// SIMATIC STEP 7 (V5.x) project PC1_NEW_01_08_2014
// CPU: CPU 315-2 DP
// station: P_ADR_BUS
// station: Hardware
// station: SIMATIC 300 - BEC
// program: S7 Program(1)

SYMBOL_TABLE
"MAIN_POWER_DB"	DB 1	DB 1	// MAIN POWER DATA BLOCK
"HYDRAULIC_FUNCTIONS_DB"	DB 2	DB 2	// HYDRAULIC FUNCTIONS DB
"TRAVEL_DRIVE_DB"	DB 3	DB 3	// TRAVEL DRIVE DATA BLOCK
"PUSHER_RAM_DB"	DB 4	DB 4	// PUSHER RAM DRIVE MECHANISH DATA BLOCK
"LEVEL_RAM_DB"	DB 5	DB 5	// LEVELER RAM DRIVE MECHANISH DATA BLOCK
"AIR_COMPRESSOR_DB"	DB 6	DB 6	// AIR COMPRESSOR DATA BLOCK
"DOOR_AND_JAMB_DB"	DB 7	DB 7	// DOOR AND JAMB CLEANER VIBRATOR DATA BLOCK
"LEVELER_BLOWER_DB"	DB 8	DB 8	// LEVELER BLOWER DATA BLOCK
"LIFTING_PLATFORM_DB"	DB 9	DB 9	// LIFTING PLATFORM DATA BLOCK
"LEVELER_DOOR_DB"	DB 10	DB 10	// LEVELER DOOR MECHANISM DATA BLOCK
"LEVELER_MUFF_DB"	DB 11	DB 11	// LEVELER MUFF MECHANISM DATA BLOCK
"DOOR_EXTRACTOR_DB"	DB 12	DB 12	// DOOR EXTRACTOR MECHANISH DATA BLOCK
"DOOR_CLEANER_DB"	DB 13	DB 13	// DOOR CLEANER MECHANISM DATA BLOCK
"JAMB_CLEANER_DB"	DB 14	DB 14	// JAMB CLEANER MECHANISM DATA BLOCK
"COUNTER_THRUST_WEDGE_DB"	DB 15	DB 15	// COUNTER THRUST WEDGE DATA BLOCK
"COAL_SPILLAGE_SYSTEM_DB"	DB 16	DB 16	// COAL SPILLAGE SYSTEM DATA BLOCK
"TATA_COMMUNICATION_DB"	DB 17	DB 17	// TATA COMMUNICATION THROUGH PROFIBUS
"WINCC_DB"	DB 18	DB 18
"DB_FOR_FM350"	DB 19	UDT 2
"FB_TO_TATA"	DB 20	DB 20	// FEEDBACK TO TATA ONBOARD PLC THROUGH PROFIBUS
"CMD_FROM_TATA"	DB 21	DB 21	// COMMAND FROM TATA ONBOARD PLC THROUGH PROFIBUS
"INPUT_MAPPING"	FC 1	FC 1	// INPUT MAPPING TO DATA BLOCK
"OUTPUT_MAPPING"	FC 2	FC 2	// OUTPUT MAPPING FROM DATA BLOCK
"MAIN_POWER"	FC 3	FC 3	// MAIN POWER CONTROL LOGIC
"HYDRAULIC_SYSTEM"	FC 4	FC 4	// HYDRAULIC SYSTEM OPERATIONS
"LEVELLER_RAM"	FC 5	FC 5	// LEVELLER RAM MECHANISH FUNCTION
"LEVELER_DOOR"	FC 6	FC 6	// LEVELLER DOOR MECHANISM
"TRAVEL_DRIVE"	FC 7	FC 7	// TRAVEL_DRIVE_MECHANISM
"PUSHER_RAM"	FC 8	FC 8	// PUSHER RAM MECHANISM
"AIR_COMPRESSOR"	FC 9	FC 9	// AIR COMPRESSOR FUNCTION
"DOOR_AND_JAMB"	FC 10	FC 10	// DOOR AND JAMB CLEANER MECHANISM
"LEVELER_BLOWER"	FC 11	FC 11	// LEVELER BLOWER FUNCTIONS
"LIFTING_PLATFORM"	FC 12	FC 12	// LIFTING PLATFORM FUNCTIONS
"LEVELER_MUFF"	FC 13	FC 13	// LEVELER MUFF MECHANISM
"DOOR_EXTRACTOR"	FC 14	FC 14	// DOOR EXTRACTOR MECHANISM
"DOOR_CLEANER"	FC 15	FC 15	// DOOR CLEANER MECHANISM
"JAMB_CLEANER"	FC 16	FC 16	// JAMB CLEANER MECHANISM
"COUNTER_THRUST_WEDGE"	FC 17	FC 17	// COUNTER THRUST WEDGE MECHANISM
"COAL_SPILLAGE_SYSTEM"	FC 18	FC 18	// COAL SPILLAGE SYSTEM
"PROFIBUS_COMMUNICATION"	FC 19	FC 19	// PROFIBUS COMMUNICATION
"TATA_COMMUNICATION"	FC 20	FC 20	// TATA COMMUNICATION FOR AUTO POSITIONING
"Clock Generator"	FC 69	FC 69	// Clock generator
"SCALE"	FC 105	FC 105	// Scaling Values
"UNSCALE"	FC 106	FC 106	// Unscaling Values
"MAIN_PWR_RDY_FOR_ON"	I 0.0	BOOL	// MAIN POWER READY FOR ON
"MAIN_PWR_ON_PB"	I 0.1	BOOL	// MAIN POWER ON PUSH BUTTON
"MAIN_PWR_OFF_PB"	I 0.2	BOOL	// MAIN POWER OFF PUSH BUTTON
"MAIN_PWR_ON_FB"	I 0.3	BOOL	// MAIN POWER ON FEED BACK
"CTRL_PWR_ON_FB"	I 0.4	BOOL	// CONTROL POWER ON FEEDBACK
"LAMP_TEST_PB"	I 0.5	BOOL	// LAMP TEST PUSH BUTTON
"ALARM_ACK_PB"	I 0.6	BOOL	// ALARM ACKNOWLEDGE PUSH BUTTON
"TRA_ILK_BYPAS"	I 0.7	BOOL	// TRAVEL INTERLOCK BYPASS INPUT
"PUSH_RAM_ILK_BYPASS"	I 1.0	BOOL	// PUSHER RAM INTERLOCK BYPASS
"LEV_ILK_BYPASS"	I 1.1	BOOL	// LEVELER RAM INTERLOCK BYPASS INPUT
"LEV_DRV_PROF_HARD_SEL"	I 1.2	BOOL	// LEVELER DRIVE PROFIBUS / HARD WIRE CONNECTION
"LEV_DRV_ON_FB"	I 1.3	BOOL	// LEVELER DRIVE ON FEED BACK
"PUMP_1_RDY_FOR_STA"	I 1.4	BOOL	// PUMP 1 READY FOR START
"PUMP_1_RUN_FB"	I 1.5	BOOL	// PUMP 1 RUNNING FEEDBACK
"PUMP_1_OVR_LD_TRIP"	I 1.6	BOOL	// PUMP 1 OVER LOAD TRIPPED
"LEV_DRV_RDY_FOR_STA"	I 1.7	BOOL	// LEVELER DRIVE READY FOR START
"PUMP_2_RDY_FOR_STA"	I 2.0	BOOL	// PUMP 2 READY FOR START
"PUMP_2_RUN_FB"	I 2.1	BOOL	// PUMP 2 RUNNING FEEDBACK
"PUMP_2_OVR_LD_TRIP"	I 2.2	BOOL	// PUMP 2 OVER LOAD TRIPPED
"CIR_PUMP_RDY_FOR_STA"	I 2.3	BOOL	// CIRCULATION PUMP READY FOR START
"CIR_PUMP_RUN_FB"	I 2.4	BOOL	// CIRCULATION PUMP RUNNING FEEDBACK
"CIR_PUMP_OVR_LD_TRIP"	I 2.5	BOOL	// CIRCULATION PUMP OVER LOAD TRIPPED
"COLR_FAN_RDY_FOR_STA"	I 2.6	BOOL	// COOLER FAN READY FOR START
"LEV_DRV_TRP_FB"	I 2.7	BOOL	// LEVELER DRIVE TRIP FEED BACK
"COLR_FAN_RUN_FB"	I 3.0	BOOL	// COOLER FAN RUNNING FEEDBACK
"COLR_FAN_OVR_LD_TRIP"	I 3.1	BOOL	// COOLER FAN OVER LOAD TRIPPED
"CD_LCS_SS"	I 3.2	BOOL	// CONTROL DESK / LOCAL CONTROL SELECTOR SWITCH
"PUMP_1_2_SS"	I 3.3	BOOL	// PUMP 1 OR 2 SELECTOR SWITCH
"PUMP_1_STA_PB"	I 3.4	BOOL	// PUMP 1 START PUSH BUTTON
"PUMP_1_STP_PB"	I 3.5	BOOL	// PUMP 1 STOP PUSH BUTTON
"PUMP_2_STA_PB"	I 3.6	BOOL	// PUMP 2 START PUSH BUTTON
"GRV_SCRPR_2_FWD_LS"	I 3.7	BOOL	// DOOR CLEANER GROOVE SCRAPPER 2 FORWARD LIMIT SWITCH
"PUMP_2_STP_PB"	I 4.0	BOOL	// PUMP 2 STOP PUSH BUTTON
"EMERGENCY_STOP_PB_LCS_41"	I 4.1	BOOL	// EMERGENCY STOP PUSH BUTTON LCS 41
"PUMP_1_2_SS_LCS"	I 4.2	BOOL	// PUMP 1 OR 2 SELECTOR SWITCH LCS
"PUMP_1_STA_PB_LCS"	I 4.3	BOOL	// PUMP 1 START PUSH BUTTON LCS
"PUMP_1_STP_PB_LCS"	I 4.4	BOOL	// PUMP 1 STOP PUSH BUTTON LCS
"PUMP_2_STA_PB_LCS"	I 4.5	BOOL	// PUMP 2 START PUSH BUTTON LCS
"PUMP_2_STP_PB_LCS"	I 4.6	BOOL	// PUMP 2 STOP PUSH BUTTON LCS
"GRV_SCRPR_2_RET_LS"	I 4.7	BOOL	// DOOR CLEANER GROOVE SCRAPPER 2 RETRACT LIMIT SWITCH
"CIR_PUMP_STA_PB_LCS"	I 5.0	BOOL	// CIRCULATION PUMP START PUSH BUTTON LCS
"CIR_PUMP_STP_PB_LCS"	I 5.1	BOOL	// CIRCULATION PUMP STOP PUSH BUTTON LCS
"COLR_FAN_STA_PB_LCS"	I 5.2	BOOL	// COOLER FAN START PUSH BUTTON LCS
"COLR_FAN_STP_PB_LCS"	I 5.3	BOOL	// COOLER FAN STOP PUSH BUTTON LCS
"LAMP_TEST_PB_LCS_41"	I 5.4	BOOL	// LAMP TEST PUSH BUTTON LCS
"SHT_OF_VLV_LIN_1_FUL_OPN"	I 5.5	BOOL	// SHUT OFF VALVE IN LINE 1 - FULLY OPEN
"SHT_OF_VLV_LIN_2_FUL_OPN"	I 5.6	BOOL	// SHUT OFF VALVE IN LINE 2 - FULLY OPEN
"DOOR_FIX_LOC_FB_PR_SWT"	I 5.7	BOOL	// DOOR FIX LOCKED FEEDBACK PRESSURE SWITCH
"LOW_OIL_TEMP"	I 6.0	BOOL	// LOW OIL TEMPERATURE - THERMOSTAT
"HIGH_OIL_TEMP"	I 6.1	BOOL	// HIGH OIL TEMPERATURE - THERMOSTAT
"MAX_OIL_TEMP"	I 6.2	BOOL	// MAXIMUM OIL TEMPERATURE - THERMOSTAT
"LOW_OIL_LEVEL"	I 6.3	BOOL	// LOW OIL LEVEL - FLOAT SWITCH
"MIN_OIL_LEVEL"	I 6.4	BOOL	// MINIMUM OIL LEVEL - FLOAT SWITCH
"RET_LIN_FLTR_CKD"	I 6.5	BOOL	// RETURN LINE FILTER CHOKED
"LOW_OIL_PRESS"	I 6.6	BOOL	// LOW OIL PRESSURE - PRESSURE SWITCH
"DOOR_FIX_REL_FB"	I 6.7	BOOL	// DOOR FIXRELEASED FEEDBACK
"HIGH_OIL_PRESS"	I 7.0	BOOL	// HIGH OIL PRESSURE - PRESSURE SWITCH
"EMG_ACCM_STA_PB_LCS"	I 7.1	BOOL	// EMERGENCY ACCUMULATOR START PB LCS
"EMG_ACCM_STP_PB_LCS"	I 7.2	BOOL	// EMERGENCY ACCUMULATOR STOP PB LCS
"HTR_STA_PB_LCS"	I 7.3	BOOL	// HEATER START PUSH BUTTON LCS
"HTR_STP_PB_LCS"	I 7.4	BOOL	// HEATER STOP PUSH BUTTON LCS
"TRA_GRP_1_RDY_FOR_STA"	I 7.6	BOOL	// TRAVEL GROUP 1 READY FOR START
"TATA_PUSH_PERM_BYPASS"	I 7.7	BOOL	// TATA PUSHING PERMISION BYPASS
"TRA_GRP_2_RDY_FOR_STA"	I 8.0	BOOL	// TRAVEL GROUP 2 READY FOR START
"TRA_GRP_2_RUN_FB"	I 8.1	BOOL	// TRAVEL GROUP 2 RUNNING FEEDBACK
"TRA_MTR_3_OVLD_TRIP"	I 8.2	BOOL	// TRAVEL MOTOR 3 OVER LOAD TRIP
"TRA_MTR_4_OVLD_TRIP"	I 8.3	BOOL	// TRAVEL MOTOR 4 OVER LOAD TRIP
"TRA_GRP_1_BRK_RDY_FOR_ST"	I 8.4	BOOL	// TRAVEL GROUP 1 BREAK READY FOR START
"TRA_GRP_1_BRK_ON_FB"	I 8.5	BOOL	// TRAVEL GROUP 1 BREAK ON FEEDBACK
"TRA_GRP_1_RUN_FB"	I 8.6	BOOL	// TRAVEL GROUP 1 RUNNING FEEDBACK
"USE_JOY_STICK_FOR_PUSH"	I 8.7	BOOL	// USER TRAVEL JOY STICK FOR PUSHER
"TRA_MTR_1_OVLD_TRIP"	I 9.0	BOOL	// TRAVEL MOTOR 1 OVER LOAD TRIP
"TRA_MTR_2_OVLD_TRIP"	I 9.1	BOOL	// TRAVEL MOTOR 2 OVER LOAD TRIP
"TRA_MTR_1_ISO_ON_FB"	I 9.2	BOOL	// TRAVEL MOTOR 1 ISOLATOR ON FEEDBACK
"TRA_MTR_2_ISO_ON_FB"	I 9.3	BOOL	// TRAVEL MOTOR 2 ISOLATOR ON FEEDBACK
"TRA_MTR_3_ISO_ON_FB"	I 9.4	BOOL	// TRAVEL MOTOR 3 ISOLATOR ON FEEDBACK
"TRA_MTR_4_ISO_ON_FB"	I 9.5	BOOL	// TRAVEL MOTOR 4 ISOLATOR ON FEEDBACK
"SIR_RDY_FOR_STA"	I 9.6	BOOL	// SIREN READY FOR START
"USE_JOY_STICK_FOR_LEV"	I 9.7	BOOL	// USE TRAVEL JPY STICK FOR LEVELER
"SIR_ON_FB"	I 10.0	BOOL	// SIREN ON FEED BACK
"TRA_GRP_2_BRK_RDY_FOR_ST"	I 10.1	BOOL	// TRAVEL GROUP 2 BREAK READY FOR START
"TRA_GRP_2_BRK_ON_FB"	I 10.2	BOOL	// TRAVEL GROUP 2 BREAK ON FEEDBACK
"SIR_OLR_TRIP"	I 10.3	BOOL	// SIREN ON OVER LOAD TRIP
"TRA_JOY_STK_REV_POS"	I 10.4	BOOL	// TRAVEL JOY STICK REVERSE POSITION
"TRA_JOY_STK_DED_MAN_BTN"	I 10.5	BOOL	// TRAVEL JOY DEAD MAN BUTTON
"TRA_JOY_STK_HME_POS"	I 10.6	BOOL	// TRAVEL JOY STICK HOME POSITION
"PUSH_JS_FWD_POS"	I 10.7	BOOL	// PUSHER RAM JOY STICK FORWARD POSITION
"TRA_JOY_STK_FWD_POS"	I 11.0	BOOL	// TRAVEL JOYSTICK FORWARD POSITION
"TRA_DRV_1_PROF_HARD_SS"	I 11.1	BOOL	// TRAVEL DRIVE 1 PROFIBUS/HARD WIRE SELECTRO SWITCH
"TRA_DRV_1_ON_FB"	I 11.2	BOOL	// TRAVEL DRIVE 1 ON FEEDBACK
"TRA_DRV_1_RDY_FOR_STA"	I 11.3	BOOL	// TRAVEL DRIVE 1 READY FOR START
"TRA_DRV_1_TRP_FB"	I 11.4	BOOL	// TRAVEL DRIVE 1 TRIP FEEDBACK
"TRA_DRV_2_PROF_HARD_SS"	I 11.5	BOOL	// TRAVEL DRIVE 2 PROFIBUS/HARD WIRE SELECTRO SWITCH
"TRA_DRV_2_ON_FB"	I 11.6	BOOL	// TRAVEL DRIVE 2 ON FEEDBACK
"PUSH_JS_HME_POS"	I 11.7	BOOL	// PUSHER JOY STICK HOME POSITION
"TRA_DRV_2_RDY_FOR_STA"	I 12.0	BOOL	// TRAVEL DRIVE 2 READY FOR START
"TRA_DRV_2_TRP_FB"	I 12.1	BOOL	// TRAVEL DRIVE 2 TRIP FEEDBACK
"LIMIT_SW_END_FWD_FB"	I 12.2	BOOL	// LIMIT SWITCH END FORWARD FEEDBACK
"LIMIT_SW_END_REV_FB"	I 12.4	BOOL	// LIMIT SWITCH END REVERSE FEEDBACK
"PUSH_BRK_RDY_FOR_STA"	I 12.6	BOOL	// PUSHER BRAKE READY FOR START
"PUSH_JS_REV_POS"	I 12.7	BOOL	// PUSHER JOY STICK REVERSE POSITION
"PUSH_MTR_BRK_ON_FB"	I 13.0	BOOL	// PUSHER MOTOR BRAKE ON FEEDBCAK
"PUSH_RAM_STP_PB"	I 13.1	BOOL	// PUSHER RAM STOP PUSH BUTTON
"PUSH_MAN_SS"	I 13.2	BOOL	// PUSHER MANUAL SELECTOR SWTICH
"PUSH_AUTO_SS"	I 13.3	BOOL	// PUSHER AUTO SELECTOR SWITCH
"PUSH_DRV_PROF_HDWR_SS"	I 13.4	BOOL	// PUSHER DRIVE PROFIBUS/HARDWIRE SELECTOR SWITCH
"PUSH_DRV_ON_FB"	I 13.5	BOOL	// PUSHER DRIVE ON FEED BACK
"PUSH_DRV_RDY_FOR_STA"	I 13.6	BOOL	// PUSHER DRIVE READY FOR START
"PUSH_JS_DEAD_MAN_BTN"	I 13.7	BOOL	// PUSHER JOY STICK DEAD MAN BUTTON
"PUSH_DRV_TRP_FB"	I 14.0	BOOL	// PUSHER DRIVE TRIP FEED BACK
"PUSH_RLS_OVN_FACE_RCHD"	I 14.1	BOOL	// PUSHER RLS OVEN FACE REACHED
"PUSH_RLS_GUIDE_ENT"	I 14.2	BOOL	// PUSHER RLS GUIDE ENTRY
"PUSH_RLS_FWD_END"	I 14.3	BOOL	// PUSHER RLS FORWARD END
"PUSH_RLS_STND_PIPE"	I 14.4	BOOL	// PUSHER RLS STAND PIPE
"PUSH_RLS_REV_END"	I 14.5	BOOL	// PUSHER RLS REVERSE END
"AUTO_POS_ACK"	I 14.6	BOOL	// AUTO PISITION ACKNOWLEDGE
"TRA_MODE_AUTO_MAN_SS"	I 14.7	BOOL	// TRAVEL MODE AUTO MANUAL SELECTOR SWITCH
"CDL_EMERGENCY_PB"	I 15.0	BOOL	// CONTROL DESK LEFT EMERGENCY PUSH BUTTON
"LIFT_LDT_TMR_SS"	I 15.1	BOOL	// LIFTING LDT TIMER SELECTOR
"RAM_EMG_DRV_DIS_ENG"	I 15.2	BOOL	// RAM EMERGENCY DRIVE DISENGAGE
"RAM_END_FWD_LS"	I 15.3	BOOL	// RAM END FORWARD LIMIT SWITCH
"RAM_END_RET_LS"	I 15.4	BOOL	// RAM END RETRACT LIMIT SWITCH
"LEV_BRK_RDY_FOR_STA"	I 15.5	BOOL	// LEVELER BRAKE READY FOR START
"MTR_BRK_ON_FB"	I 15.6	BOOL	// MOTOR BRAKE ON FEED BACK
"LEV_STP_PB"	I 16.0	BOOL	// LEVELER BRAKE STOP PUSH BUTTON
"MANUAL_SS"	I 16.1	BOOL	// MANUAL SELECTOR SWITCH
"AUTO_SS"	I 16.2	BOOL	// AUTOMATIC SELECTOR SWITCH
"LEV_JS_FWD_POS"	I 16.3	BOOL	// LEVELER JOYSTICK FORWARD POSITION
"LEV_JS_HME_POS"	I 16.4	BOOL	// LEVELER JOYSTICK HOME POSITION
"LEV_JS_REV_POS"	I 16.5	BOOL	// LEVELER JOY STICK REVERSE POSITION
"LEV_JS_DEAD_MAN_BUTTON"	I 16.6	BOOL	// LEVELER JOY STICK DEAD MAN BUTTON
"LEV_RLS_OVN_FAC_RCHD"	I 17.4	BOOL	// LEVELER RLS OVEN FACE REACHED
"LEV_RLS_FWD_END"	I 17.5	BOOL	// LEVELER RLS FORWARD END
"LEV_RLS_REV_STK_FB"	I 17.6	BOOL	// LEVELER RLS REVERSE STROKE FEED BACK
"LEV_RLS_REV_END"	I 18.0	BOOL	// LEVELER RLS REVERSE END
"EMG_PB_LCS_16"	I 18.1	BOOL	// EMERGENCY PUSH BUTTON LCS 16
"LEV_EM_DRV_ENG_LCS"	I 18.2	BOOL	// LEVELER EMERGENCY DRIVE ENGAGE LCS
"LEV_EM_DRV_DIS_ENG_LCS"	I 18.3	BOOL	// LEVELER EMERGENCY DRIVE DISENGAGE LCS
"LEV_EM_DRV_DIS_ENG"	I 18.4	BOOL	// LEVELER EMERGENCY DRIVE DISENGAGE
"LEV_END_FWD_LS"	I 18.5	BOOL	// LEVELER END FORWARD LIMIT SWITCH
"LEV_END_RET_LS"	I 18.6	BOOL	// LEVELER END RETRACT LIMIT SWITCH
"SPRING_PRESS"	I 19.1	BOOL	// SPRING PRESS
"LEV_BLOW_RDY_FOR_STA"	I 19.2	BOOL	// LEVELER BLOWER READY FOR START
"LEV_BLOW_RUN_FB"	I 19.3	BOOL	// LEVELER BLOWER RUNNING FEED BACK
"LEV_BLOW_OLR_TRP"	I 19.4	BOOL	// LEVELER BLOWER TRIP FEED BACK
"LEV_BLOW_STA_PB"	I 19.5	BOOL	// LEVELER BLOWER START PUSH BUTTON
"LEV_BLOW_STP_PB"	I 19.6	BOOL	// LEVELER BLOWER STOP PUSH BUTTON
"LEV_BLOW_STA_PB_LCS"	I 20.0	BOOL	// LEVELER BLOWER START PUSH BUTTON LCS
"LEV_BLOW_STP_PB_LCS"	I 20.1	BOOL	// LEVELER BLOWER STOP PUSH BUTTON LCS
"LIFT_PF_RDY_FOR_STA"	I 20.2	BOOL	// LIFT PLATFORM READY FOR START
"LIFT_PF_UP_ON_FB"	I 20.3	BOOL	// LIFT PLATFORM UP ON FEEDBCAK
"LIFT_PF_DN_ON_FB"	I 20.4	BOOL	// LIFT PLATFORM DOWN ON FEEDBCAK
"LIFT_MTR_OLR_TRP"	I 20.5	BOOL	// LIFT MOTOR OVERLOAD TRIP
"LIFT_PF_UP_PB"	I 20.6	BOOL	// LIFT PLATFORM UP PUSH BUTTON
"LIFT_PF_DN_PB"	I 21.0	BOOL	// LIFT PLATFORM DOWN PUSH BUTTON
"EMERGENCY_PB_LCS_19"	I 21.2	BOOL	// LCS-19 EMERGENCY PUSH BUTTON
"LIFT_PF_UP_LS"	I 21.3	BOOL	// LIFT PLATFORM UP LIMIT SWITCH
"LIFT_PF_DN_LS"	I 21.4	BOOL	// LIFT PLATFORM DOWN LIMIT SWITCH
"LEV_DOOR_LOCAL_SS"	I 22.3	BOOL	// LEVELER DOOR LOCAL SELECTOR SWITCH
"LEV_DOOR_MAN_SS"	I 22.4	BOOL	// LEVELER DOOR MANUAL SELECTOR SWITCH
"LEV_DOOR_AUTO_SS"	I 22.5	BOOL	// LEVELER DOOR AUTO SELECTOR SWITCH
"LEV_DOOR_STP_PB"	I 22.6	BOOL	// LEVELER DOOR STOP PUSH BUTTON
"ACT_GRP_FWD_STA_PB"	I 23.0	BOOL	// ACTUATING GRIP FORWARD START PUSH BUTTON
"ACT_GRP_RET_STA_PB"	I 23.1	BOOL	// ACTUATING GRIP RETRACT START PUSH BUTTON
"SLW_RK_SP_1_FWD_STA"	I 23.2	BOOL	// SLEAVING RACK STEP 1 FORWARD START PUSH BUTTON
"SLW_RK_SP_1_RET_STA"	I 23.3	BOOL	// SLEAVING RACK STEP 1 RETRACT START PUSH BUTTON
"SLW_RK_SP_2_FWD_STA"	I 23.4	BOOL	// SLEAVING RACK STEP 2 FORWARD START PUSH BUTTON
"SLW_RK_SP_2_RET_STA"	I 23.5	BOOL	// SLEAVING RACK STEP 2 RETRACT START PUSH BUTTON
"LEV_WN_FM_CR_UP_STA"	I 23.6	BOOL	// LEVELER WINDOW FRAME CLEANER UP START PUSH BUTTON
"LEV_WN_FM_CR_DN_STA"	I 24.0	BOOL	// LEVELER WINDOW FRAME CLEANER DOWN START PUSH BUTTON
"SMK_SLVE_FWD_STA_PB"	I 24.1	BOOL	// SMOKE SLEEVE FORWARD START PUSH BUTTON
"SMK_SLVE_RET_STA_PB"	I 24.2	BOOL	// SMOKE SLEEVE RETRACT START PUSH BUTTON
"EMG_STOP_PB_LCS_61"	I 24.3	BOOL	// EMERGENCY STOP PUSH BUTTON LCS 61
"ACT_GRP_FWD_STA_PB_LCS"	I 24.4	BOOL	// ACTUATING GRIP FORWARD START PUSH BUTTON LCS
"ACT_GRP_RET_STA_PB_LCS"	I 24.5	BOOL	// ACTUATING GRIP RETRACT START PUSH BUTTON LCS
"SLW_RK_SP_1_FWD_STA_LCS"	I 24.6	BOOL	// SLEAVING RACK STEP 1 FORWARD START PUSH BUTTON LCS
"SLW_RK_SP_1_RET_STA_LCS"	I 25.0	BOOL	// SLEAVING RACK STEP 1 RETRACT START PUSH BUTTON LCS
"SLW_RK_SP_2_FWD_STA_LCS"	I 25.1	BOOL	// SLEAVING RACK STEP 2 FORWARD START PUSH BUTTON LCS
"SLW_RK_SP_2_RET_STA_LCS"	I 25.2	BOOL	// SLEAVING RACK STEP 2 RETRACT START PUSH BUTTON LCS
"LEV_WN_FM_CR_UP_STA_LCS"	I 25.3	BOOL	// LEVELER WINDOW FRAME CLEANER UP START PUSH BUTTON LCS
"LEV_WN_FM_CR_DN_STA_LCS"	I 25.4	BOOL	// LEVELER WINDOW FRAME CLEANER DOWN START PUSH BUTTON LCS
"SMK_SLVE_FWD_STA_PB_LCS"	I 25.5	BOOL	// SMOKE SLEEVE FORWARD START PUSH BUTTON LCS
"SMK_SLVE_RET_STA_PB_LCS"	I 25.6	BOOL	// SMOKE SLEEVE RETRACT START PUSH BUTTON LCS
"TEST_LAMP_PB_LCS_61"	I 26.0	BOOL	// TEST LAMP PUSH BUTTON LCS 61
"SLW_RK_SP_1_FWD_LS"	I 26.5	BOOL	// SLEAVING RACK STEP 1 FORWARD LIMIT SWITCH
"SLW_RK_SP_1_RET_LS"	I 26.6	BOOL	// SLEAVING RACK STEP 1 RETRACT LIMIT SWITCH
"SLW_RK_SP_2_FWD_LS"	I 27.0	BOOL	// SLEAVING RACK STEP 2 FORWARD LIMIT SWITCH
"SLW_RK_SP_2_RET_LS"	I 27.1	BOOL	// SLEAVING RACK STEP 2 RETRACT LIMIT SWITCH
"LEV_WN_FM_CR_UP_LS"	I 27.2	BOOL	// LEVELER WINDOW FRAME CLEANER UP LIMIT SWITCH
"LEV_WN_FM_CR_DN_LS"	I 27.3	BOOL	// LEVELER WINDOW FRAME CLEANER DOWN LIMIT SWITCH
"SMK_SLVE_FWD_LS"	I 27.4	BOOL	// SMOKE SLEEVE FORWARD LIMIT SWITCH
"SMK_SLVE_SLOW_FWD_LS"	I 27.5	BOOL	// SMOKE SLEEVE SLOW FORWARD LIMIT SWITCH
"SMK_SLVE_REV_LS"	I 27.6	BOOL	// SMOKE SLEEVE RETRACT LIMIT SWITCH
"VIB_JMB_CLNR_STA_PB_LCS"	I 27.7	BOOL	// VIBRATOR - JAMB CLEANER START PUSH BUTTON LCS
"ACT_GRP_FWD_LS"	I 28.0	BOOL	// ACTUATING GRIP FORWARD START LIMIT SWITCH
"ACT_GRP_RET_LS"	I 28.1	BOOL	// ACTUATING GRIP RETRACT START LIMIT SWITCH
"VIB_JMB_CLNR_STP_PB_LCS"	I 28.2	BOOL	// VIBRATOR - JAMB CLEANER STOP PUSH BUTTON LCS
"AIR_COMP_PRESSURE_SW_FB"	I 28.5	BOOL	// PRESSURE SWITCH FEEDBACK
"DOOR_EXT_LOC_SS"	I 28.6	BOOL	// DOOR EXTRACTOR LOCAL SELECTOR SWITCH
"DOOR_EXT_MAN_SS"	I 29.0	BOOL	// DOOR EXTRACTOR MANUAL SELECTOR SWITCH
"DOOR_EXT_AUTO_SS"	I 29.1	BOOL	// DOOR EXTRACTOR AUTO SELECTOR SWITCH
"DOOR_EXT_STP_PB"	I 29.2	BOOL	// DOOR EXTRACTOR STOP PUSH BUTTON
"SLEW_FWD_STA_PB"	I 29.3	BOOL	// SLEW FORWARD START PUSH BUTTON
"SLEW_RET_STA_PB"	I 29.4	BOOL	// SLEW RETRACT START
"VER_COMP_FWD_STA"	I 29.5	BOOL	// VERTICAL COMPENSATION FORWARD START PUSHBUTTON
"VER_COMP_RET_STA"	I 29.6	BOOL	// VERTICAL COMPENSATION RETRACT START PUSHBUTTON
"TRA_FWD_STA"	I 30.0	BOOL	// TRAVEL FORWARD START PUSHBUTTON
"TRA_RET_STA"	I 30.1	BOOL	// TRAVEL RETRACT START PUSHBUTTON
"MAN_STK_UP_STA_PB"	I 30.2	BOOL	// MAIN STROKE UP START PUSH BUTTON
"MAN_STK_UP_DN_PB"	I 30.3	BOOL	// MAIN STROKE DOWN START PUSH BUTTON
"FNL_STK_UP_STA_PB"	I 30.4	BOOL	// FINAL STROKE UP START PUSH BUTTON
"FNL_STK_UP_DN_PB"	I 30.5	BOOL	// FINAL STROKE DOWN START PUSH BUTTON
"PRE_STK_UP_STA_PB"	I 30.6	BOOL	// PRE STROKE UP START PUSH BUTTON
"PRE_STK_UP_DN_PB"	I 31.0	BOOL	// PRE STROKE DOWN START PUSH BUTTON
"DOOR_SPRG_PRS_STA_PB"	I 31.1	BOOL	// DOOR SPRING PRESS START PUSH BUTTON
"DOOR_SPRG_RLES_STA_PB"	I 31.2	BOOL	// DOOR SPRING RELEASE START PUSH BUTTON
"DOOR_LCH_TURN_LOCK"	I 31.3	BOOL	// DOOR LATCH TURNING LOCK
"DOOR_LCH_TURN_UNLOC"	I 31.4	BOOL	// DOOR LATCH TURNING UNLOCK
"EMERGENCY_PB_LCS_73"	I 31.5	BOOL	// EMERGENCY PUSHBUTTON LCS-73
"SLEW_FWD_STA_LCS"	I 31.6	BOOL	// SLEW_FORWARD_START_PUSHBUTTON_LCS
"SLEW_RET_STA_LCS"	I 32.0	BOOL	// SLEW_RETRACT_START_PUSHBUTTON_LCS
"VER_COMP_FWD_STA_LCS"	I 32.1	BOOL	// VERTICAL COMPENSATION FORWARD START LCS PUSH BUTTON
"VER_COMP_RET_STA_LCS"	I 32.2	BOOL	// VERTICAL COMPENSATION RETRACT START LCS PUSH BUTTON
"TRA_FWD_STA_LCS"	I 32.3	BOOL	// TRAVEL FORWARD START LCS  PUSH BUTTON
"TRA_BACK_STA_LCS"	I 32.4	BOOL	// TRAVEL BACK START LCS  PUSH BUTTON
"MAIN_STK_UP_STA_LCS"	I 32.5	BOOL	// MAIN STROKE UP START LCS PUSH BUTTON
"MAIN_STK_DN_STA_LCS"	I 32.6	BOOL	// MAIN STROKE DN START LCS PUSH BUTTON
"FNL_STK_UP_STA_LCS"	I 33.0	BOOL	// FINAL STROKE UP START LCS  PUSH BUTTON
"FNL_STK_DN_STA_LCS"	I 33.1	BOOL	// FINAL STROKE DOWN START LCS PUSH BUTTON
"PRE_STK_UP_STA_LCS"	I 33.2	BOOL	// PREE STROKE UP START LCS PUSH BUTTON
"PRE_STK_DN_STA_LCS"	I 33.3	BOOL	// PREE STROKE DN START LCS PUSH BUTTON
"DOOR_SPRG_PRS_LK_STA_LCS"	I 33.4	BOOL	// DOOR SPRING LOCK START PUSH BUTTON LCS
"DOOR_SPRG_RLES_UNLSTA_LC"	I 33.5	BOOL	// DOOR SPRING UNLOCK  START PUSH BUTTON LCS
"LAMP_TEST_PB_LCS_73"	I 34.1	BOOL	// LAMP_TEST_PUSHBUTTON_LCS-73
"SLEW_SLOW_FWD_LS"	I 34.2	BOOL	// SLEW SLOW FORWARD LIMIT SWITCH
"SLEW_SLOW_RET_LS"	I 34.3	BOOL	// SLEW SLOW RETRACT LIMIT SWITCH
"SLEW_NOR_FWD_LS"	I 34.4	BOOL	// SLEW NORMAL FORWARD LIMIT SWITCH
"SLEW_NOR_RET_LS"	I 34.5	BOOL	// SLEW NORMAL RETRACT LIMIT SWITCH
"TRA_SLOW_FWD_LS"	I 34.6	BOOL	// TRAVEL SLOW FORWARD LIMIT  SWITCH
"TRA_SLOW_RET_LS"	I 35.0	BOOL	// TRAVEL SLOW RETRACT LIMIT  SWITCH
"TRA_FWD_LS"	I 35.1	BOOL	// TRAVEL FORWARD LIMIT SWIITCH
"TRA_RET_LS"	I 35.2	BOOL	// TRAVEL RETRACT LIMIT SWIITCH
"FOR_LS_TRAVEL"	I 35.3	BOOL	// FORWARD LIMIT SWITCH TRAVEL
"DOOR_ON_HOOK_LS"	I 35.4	BOOL	// DOOR ON HOOK LIMITSWTCH
"DOOR_LAT_TUR_UP_LS"	I 36.0	BOOL	// DOOR_LATCH_TURNING_UP_LIMIT SWICH
"DOOR_LAT_TUR_DN_LS"	I 36.1	BOOL	// DOOR_LATCH_TURNING_DN_LIMIT SWICH
"DOOR_LAT_LOCK_PB_LCS"	I 36.4	BOOL	// DOOR LATCH LOCK PUSHBUTTON LCS
"DOOR_LAT_UNLOCK_PB_LCS1"	I 36.5	BOOL	// DOOR LATCH UNLOCK PUSHBUTTON LCS
"DOOR_LAT_HOME_PB_LCS"	I 36.6	BOOL	// DOOR LATCH HOME PUSHBUTTON LCS
"LOCAL_SEL_SW"	I 37.0	BOOL	// DOOR CLEANER LOCAL SELECTOR SWITCH
"MAN_SEL_SW"	I 37.1	BOOL	// DOOR CLEANER MANUAL SELECTOR SWITCH
"AUTO_SEL_SW1"	I 37.2	BOOL	// DOOR CLEANER AUTO SELECTOR SWITCH
"STOP_PB"	I 37.3	BOOL	// DOOR CLEANER STOP PUSH BUTTON
"CAR_TRV_FWD_STA_PB"	I 37.4	BOOL	// DOOR CLEANER CARRIAGE TRAVEL FORWARD START PUSH BUTTON
"CAR_TRV_RET_STA_PB"	I 37.5	BOOL	// DOOR CLEANER CARRIAGE TRAVEL RETURN START PUSH BUTTON
"VER_CLNR_UP_STA_PB"	I 37.6	BOOL	// DOOR CLEANER VERTICAL CLEANER UP START PUSH BUTTON
"VER_CLNR_DOWN_STA_PB"	I 38.0	BOOL	// DOOR CLEANER VERTICAL CLEANER DOWN START PUSH BUTTON
"GRV_SCRP_FWD_STA"	I 38.1	BOOL	// DOOR CLEANER GROOVE SCRAPPER FORWARD START PUSH BUTTON
"GRV_SCRP_RET_STA"	I 38.2	BOOL	// DOOR CLEANER GROOVE SCRAPPER REVERSE START PUSH BUTTON
"TOP_SCRP_FWD_STA"	I 38.3	BOOL	// DOOR CLEANER TOP SCRAPPER FORWARD START PUSH BUTTON
"TOP_SCRP_REV_STA"	I 38.4	BOOL	// DOOR CLEANER TOP SCRAPPER REVERSE START PUSH BUTTON
"BTM_SCRP_FWD_STA"	I 38.5	BOOL	// DOOR CLEANER BOTTOM SCRAPPER FORWARD START PUSH BUTTON
"BTM_SCRP_REV_STA"	I 38.6	BOOL	// DOOR CLEANER BOTTOM SCRAPPER REVERSE START PUSH BUTTON
"GRV_SCRPR_ON_LCS"	I 38.7	BOOL	// DOOR CLEANER GROOVE SCRAPPER ON PUSH BUTTON LCS
"LCS_85_EMG_STP"	I 39.0	BOOL	// DOOR CLEANER LCS_85 EMERGENCY STOP PUSH BUTTON
"CAR_TRV_FWD_STA_PB_LCS"	I 39.1	BOOL	// DOOR CLEANER CARRIAGE TRAVEL FORWARD START PUSH BUTTON IN LCS
"CAR_TRV_RET_STA_PB_LCS"	I 39.2	BOOL	// DOOR CLEANER CARRIAGE TRAVEL RETURN START PUSH BUTTON IN LCS
"VER_CLNR_UP_STA_PB_LCS"	I 39.3	BOOL	// DOOR CLEANER VERTICAL CLEANER UP START PUSH BUTTON IN LCS
"VER_CLR_DWN_STA_PB_LCS"	I 39.4	BOOL	// DOOR CLEANER VERTICAL CLEANER DOWN START PUSH BUTTON IN LCS
"BTM_BRK_HLDR_FWD_STA_LCS"	I 39.5	BOOL	// DOOR CLEANER BOTTOM BRICK HOLDER FORWARD START PUSH BUTTON IN LCS
"BTM_BRK_HLDR_REV_STA_LCS"	I 39.6	BOOL	// DOOR CLEANER BOTTOM BRICK HOLDER REVERSE START PUSH BUTTON IN LCS
"LAMP_TEST"	I 39.7	BOOL	// DOOR CLEANER LAMP TEST PB IN LCS
"TOP_SCRPR_FWD_STA_LCS"	I 40.0	BOOL	// DOOR CLEANER TOP SCRAPPER FORWARD START PUSH BUTTON IN LCS
"TOP_SCRPR_REV_STA_LCS"	I 40.1	BOOL	// DOOR CLEANER TOP SCRAPPER REVERSE START PUSH BUTTON IN LCS
"BTM_SCRPR_FWD_STA_LCS"	I 40.2	BOOL	// DOOR CLEANER BOTTOM SCRAPPER FORWARD START PUSH BUTTON IN LCS
"BTM_SCRPR_REV_STA_LCS"	I 40.3	BOOL	// DOOR CLEANER BOTTOM SCRAPPER REVERSE START PUSH BUTTON IN LCS
"CAR_TRV_FWD_LS"	I 40.4	BOOL	// DOOR CLEANER CARRIAGE TRAVEL FORWARD LIMIT SWITCH
"CAR_TRV_RET_LS"	I 40.5	BOOL	// DOOR CLEANER CARRIAGE TRAVEL RETURN LIMIT SWITCH
"VER_CLNR_UP_LS"	I 40.6	BOOL	// DOOR CLEANER VERTICAL CLEANER UP LIMIT SWITCH
"GRV_SCRPR_OFF_LCS"	I 40.7	BOOL	// DOOR CLEANER GROOVE SCRAPPER OFF PUSH BUTTON LCS
"VER_CLNR_DOWN_LS"	I 41.0	BOOL	// DOOR CLEANER VERTICAL CLEANER DOWN LIMIT SWITCH
"GRV_SCRPR_1_FWD_LS"	I 41.1	BOOL	// DOOR CLEANER GROOVE SCRAPPER 1 FORWARD LIMIT SWITCH
"GRV_SCRPR_1_RET_LS"	I 41.2	BOOL	// DOOR CLEANER GROOVE SCRAPPER 1 REVERSE LIMIT SWITCH
"TOP_SCRP_FWD_LS"	I 41.3	BOOL	// DOOR CLEANER TOP SCRAPPER FORWARD LIMIT SWITCH
"TOP_SCRP_REV_LS"	I 41.4	BOOL	// DOOR CLEANER TOP SCRAPPER REVERSE LIMIT SWITCH
"BTM_SCRP_FWD_LS"	I 41.5	BOOL	// DOOR CLEANER BOTTOM SCRAPPER FORWARD LIMIT SWITCH
"BTM_SCRP_REV_LS"	I 41.6	BOOL	// DOOR CLEANER BOTTOM SCRAPPER REVERSE LIMIT SWITCH
"JC_LOC_SS"	I 42.0	BOOL	// JAMP CLEANER LOCAL SELECTOR SWITCH
"JC_MAN_SS"	I 42.1	BOOL	// JAMP CLEANER MANUAL SELECTOR SWITCH
"JC_AUTO_SS"	I 42.2	BOOL	// JAMP CLEANER AUTO SELECTOR SWITCH
"JC_STOP_PB"	I 42.3	BOOL	// JAMP CLEANER STOP PUSH BUTTON
"JC_SLEW_FWD_STA_PB"	I 42.4	BOOL	// JAMP CLEANER SLEW FORWARD START PUSH BUTTON
"JC_SLEW_RET_STA_PB"	I 42.5	BOOL	// JAMP CLEANER SLEW RETRACT START PUSH BUTTON
"TRA_FWD_STA_PB"	I 42.6	BOOL	// TRAVEL FORWARD START PUSH BUTTON
"TRA_RET_STA_PB"	I 43.0	BOOL	// TRAVEL RETRACT START PUSH BUTTON
"VER_CLE_UP_STA_PB"	I 43.1	BOOL	// VERTICAL CLEANER UP  START PUSH BUTTON
"VER_CLE_DN_STA_PB"	I 43.2	BOOL	// VERTICAL CLEANER DN START PUSH BUTTON
"LCS_90_EMERGENCY_PB"	I 43.3	BOOL	// LCS-90 EMERGENCY PUSH BUTTON
"SLEW_FWD_STA_PB_LCS"	I 43.4	BOOL	// SLEW FORWARD START PUSH BUTTON LCS
"SLEW_RET_STA_PB_LCS"	I 43.5	BOOL	// SLEW RETRACT START PUSH BUTTON LCS
"TRA_FWD_STA_PB_LCS"	I 43.6	BOOL	// TRAVEL FORWARD START PUSH BUTTON LCS
"TRA_RET_STA_PB_LCS"	I 44.0	BOOL	// TRAVEL RETRACT START PUSH BUTTON LCS
"VER_CLE_UP_STA_PB_LCS"	I 44.1	BOOL	// VERTICAL CLEANER UP  START PUSH BUTTON LCS
"VER_CLE_DN_STA_PB_LCS"	I 44.2	BOOL	// VERTICAL CLEANER DN START PUSH BUTTON LCS
"LCS_90_EMERGENCY_TEST_PB"	I 44.3	BOOL	// LCS-90 EMERGENCY TEST PUSH BUTTON
"JC_SLEW_SLOW_FWD_LS"	I 44.4	BOOL	// JAMP CLEANER SLEW SLOW FORWARD LIMIT SWITCH
"JC_SLEW_SLOW_RET_LS"	I 44.5	BOOL	// JAMP CLEANER  SLEW SLOW RETRACT LIMIT SWITCH
"SLEW_NORMAL_FWD_LS"	I 44.6	BOOL	// SLEW NORMAL FORWARD LIMIT SWITCH
"SLEW_NORMAL_RET_LS"	I 45.0	BOOL	// SLEW NORMAL RETRACT LIMIT SWITCH
"JC_TRA_SLOW_FWD_LS"	I 45.1	BOOL	// JAMP CLEANER TRAVEL SLOW FORWARD LIMIT  SWITCH
"JC_TRA_SLOW_RET_LS"	I 45.2	BOOL	// JAMP CLEANER TRAVEL SLOW RETRACT LIMIT  SWITCH
"TRA_NORMAL_FWD_LS"	I 45.3	BOOL	// TRAVEL NORMAL FORWARD LIMIT  SWITCH
"TRA_NORMAL_RET_LS"	I 45.4	BOOL	// TRAVEL NORMAL RETRACT LIMIT  SWITCH
"VER_CLE_UP_LS"	I 45.5	BOOL	// VERTICAL CLEANER UP LIMIIT SWITCH
"VER_CLE_DN_LS"	I 45.6	BOOL	// VERTICAL CLEANER DN LIMIIT SWITCH
"CNT_TH_WED_LOC_SS"	I 46.0	BOOL	// COUNTER  THRUST WEDGE LOCAL SELECTOR SWITCH
"CNT_TH_WED_MAN_SS"	I 46.1	BOOL	// COUNTER  THRUST WEDGE MAUAL SELECTOR SWITCH
"CNT_TH_WED_AUTO_SS"	I 46.2	BOOL	// COUNTER  THRUST WEDGE AUTO SELECTOR SWITCH
"CNT_TH_WED_STOP_PB"	I 46.3	BOOL	// COUNTER  THRUST WEDGE STOP PUSH BUTTON
"CNT_TH_WED_DN_STA_PB"	I 46.4	BOOL	// COUNTER  THRUST WEDGE DOWN START PUSH BUTTON
"CNT_TH_WED_UP_STA_PB"	I 46.5	BOOL	// COUNTER  THRUST WEDGE UP START PUSH BUTTON
"CNT_TH_WED_DN_STA_PB_LCS"	I 46.6	BOOL	// COUNTER  THRUST WEDGE DN START PUSH BUTTON LCS
"CNT_TH_WED_UP_STA_PB_LCS"	I 47.0	BOOL	// COUNTER  THRUST WEDGE UP START PUSH BUTTON LCS
"EMEG_STOP_PB_LCS_72"	I 47.1	BOOL	// EMERGENCY STOP PUSH BUTTON LCS-72
"CNT_TH_WED1_DN_STA_LS"	I 47.2	BOOL	// COUNTER  THRUST WEDGE-1 DN START LIMIT SWITCH
"CNT_TH_WED1_UP_STA_LS"	I 47.3	BOOL	// COUNTER  THRUST WEDGE-1 UP START LIMIT SWITCH
"CNT_TH_WED2_DN_STA_LS"	I 47.4	BOOL	// COUNTER  THRUST WEDGE-2 DN START LIMIT SWITCH
"CNT_TH_WED2_UP_STA_LS"	I 47.5	BOOL	// COUNTER  THRUST WEDGE-2 UP START LIMIT SWITCH
"CO_SPI_CHU_DN_STA"	I 47.6	BOOL	// COAL SPILLAGE CHUTE DOWN START
"CO_SPI_CHU_UP_STA"	I 48.0	BOOL	// COAL SPILLAGE CHUTE UP START
"CO_SPI_CHU_DN_STA_LCS"	I 48.1	BOOL	// COAL SPILLAGE CHUTE DOWN START LCS
"CO_SPI_CHU_UP_STA_LCS"	I 48.2	BOOL	// COAL SPILLAGE CHUTE UP START LCS
"CO_SPI_HOP_GT_OP_STA_LCS"	I 48.3	BOOL	// COAL SPILLAGE HOPPER GATE OPEN START LCS
"CO_SPI_HOP_GT_CL_STA_LCS"	I 48.4	BOOL	// COAL SPILLAGE HOPPER GATE CLOSE START LCS
"CO_SP_CHT_DN_LS"	I 48.5	BOOL	// COAL SPILLAGE CHUTE DOWN LIMIT SWITCH
"CO_SP_CHT_UP_LS"	I 48.6	BOOL	// COAL SPILLAGE CHUTE UP LIMIT SWITCH
"CO_SPI_HOP_GT_OP_LS"	I 49.0	BOOL	// COAL SPILLAGE HOPPER GATE OPEN LIMIT SWITCH
"CO_SPI_HOP_GT_CL_LS"	I 49.1	BOOL	// COAL SPILLAGE HOPPER GATE CLOSE LIMIT SWITCH
"CTRL_SELECTION_CD"	I 49.3	BOOL	// CONTROL SELECTRION CD
"PREP_DOOR_FUNC_STA"	I 49.4	BOOL	// COUNTER THRUST WEDGE PREPARE DOOR FUNCTION START PUSH BITTON
"PREP_DOOR_FUNC_STP"	I 49.5	BOOL	// COUNTER THRUST WEDGE PREPARE DOOR FUNCTION STO
"FIN_DOOR_FUNC_STA"	I 49.6	BOOL	// COUNTER THRUST WEDGE FINISH DOOR FUNCTION START
"EXT_OVEN_DOR_AUTO_STA_PB"	I 50.0	BOOL	// EXTRACT OVEN DOOR AUTO START PUSH BUTTON
"DR_EXT_RPL_AUTO_STP_PB"	I 50.1	BOOL	// DOOR EXTRACT/REPLACE OVEN DOOR AUTO STOP PUSH BUTTON
"RPL_OVEN_DOR_AUTO_STA_PB"	I 50.2	BOOL	// REPLACE OVEN DOOR AUTO START PUSH BUTTON
"CLEAN_OVN_DR_STA"	I 50.3	BOOL	// CLEAN OVEN DOOR START PUSH BUTTON
"CLEAN_OVN_DR_STP"	I 50.4	BOOL	// CLEAN OVEN DOOR STOP PUSH BUTTON
"PUSH_AUTO_STA_PB"	I 50.5	BOOL	// PUSHER RAM AUTO START PUSH BUTTON
"PUSH_AUTO_STP_RET_PB"	I 50.6	BOOL	// PUSHER RAM AUTO STOP AND RETRACT PUSH BUTTON
"JAMB_CLNR_AUTO_STA_PB"	I 51.0	BOOL	// CLEAN OVEN DOOR AUTO START PUSH BUTTON
"JAMB_CLNR_AUTO_STP_PB"	I 51.1	BOOL	// CLEAN OVEN DOOR AUTO STOP PUSH BUTTON
"PREP_FOR_LEV_STA_PB"	I 51.2	BOOL	// PREPARE FOR LEVELING START PUSH BUTTON
"PREP_FOR_LEV_STP_PB"	I 51.3	BOOL	// PREPARE FOR LEVELING STOP PUSH BUTTON
"FIN_LEV_DOOR_OPER_STA"	I 51.4	BOOL	// FINISH LEVELING OPERATION START PUSH BUTTON
"LEV_AUTO_STA_PB"	I 51.5	BOOL	// LEVELER AUTO START PUSH BUTTON
"LEV_AUTO_STP_RET_PB"	I 51.6	BOOL	// LEVELER AUTO STOP AND RETRACT PUSH BUTTON
"TRA_SIREN_ON_PB"	I 52.0	BOOL	// TRAVEL SIREN ON PUSH BUTTON
"EMERGENCY_LCS_15"	I 52.1	BOOL	// LCS-15 EMERGENCY PUSH BUTTON
"RAM_EM_DRV_ENG_LCS_15"	I 52.2	BOOL	// RAM EMERGENCY DRIVE ENGAGE LCS-15
"RAM_EM_DRV_DENG_LCS_15"	I 52.3	BOOL	// RAM EMERGENCY DRIVE DISENGAGE LCS - 15
"EMERGENCY_PB_LCS_16"	I 52.4	BOOL	// LCS-16 EMERGENCY PUSH BUTTON
"LEV_EM_DRV_ENG_LCS_16"	I 52.5	BOOL	// LEVELER EMERGENCY DRIVE ENGAGE LCS-16
"COK_SP_SH_SLE_FWD_STA_PB"	I 52.6	BOOL	// COKE SPILLAGE SHOVEL  SLEW FORWARD START PUSH BUTTON
"VIB_DOR_CLNR_RDY_FOR_STA"	I 53.0	BOOL	// VIBRATOR - DOOR CLEANER READY FOR START
"VIB_DOR_CLNR_RUN_FB"	I 53.1	BOOL	// VIBRATOR - DOOR CLEANER RUN FEEDBACK
"VIB_DOR_CLNR_OLR_TRP"	I 53.2	BOOL	// VIBRATOR - DOOR CLEANER OVERLOAD TRIP
"VIB_JMB_CLNR_RDY_FOR_STA"	I 53.3	BOOL	// VIBRATOR - JAMB CLEANER READY FOR START
"VIB_JMB_CLNR_RUN_FB"	I 53.4	BOOL	// VIBRATOR - JAMB CLEANER RUN FEEDBACK
"VIB_JMB_CLNR_OLR_TRP"	I 53.5	BOOL	// VIBRATOR - JAMB CLEANER OVERLOAD TRIP
"VIB_DOR_CLNR_STA_PB"	I 53.6	BOOL	// VIBRATOR - DOOR CLEANER START PUSH BUTTON
"COK_SP_SH_SLE_RET_STA_PB"	I 53.7	BOOL	// COKE SPILLAGE SHOVEL  SLEW RETRACT START PUSH BUTTON
"DR_CL_SP_SH_SL_FWD_LCS"	I 54.0	BOOL	// DOOR CLEANER SPILLAGE SHOWEL SLEW FORWARD START LCS
"DR_CL_SP_SH_SL_RET_LCS"	I 54.1	BOOL	// DOOR CLEANER SPILLAGE SHOWEL SLEW RETRACT START LCS
"DR_CL_SP_HO_FWD_STA_LCS"	I 54.2	BOOL	// DOOR  CLEANER SPILLAGE HOPPER FORWARD START LCS
"DR_CL_SP_HO_RET_STA_LCS"	I 54.3	BOOL	// DOOR  CLEANER SPILLAGE HOPPER RETRACT START LCS
"VIB_DOR_CLNR_STP_PB"	I 54.4	BOOL	// VIBRATOR - DOOR CLEANER STOP PUSH BUTTON
"VIB_JMB_CLNR_STA_PB"	I 54.5	BOOL	// VIBRATOR - JAMB CLEANER START PUSH BUTTON
"VIB_JMB_CLNR_STP_PB"	I 54.6	BOOL	// VIBRATOR - JAMB CLEANER STOP PUSH BUTTON
"MRT_1_RDY_FOR_STA"	I 55.0	BOOL	// MOTOR 1 READY FOR START
"MTR_1_RUN_FB"	I 55.1	BOOL	// MOTOR 1 RUN FEEDBACK
"MTR_1_OLR_TRP"	I 55.2	BOOL	// MOTOR 1 OVER LOAD TRIP
"MRT_2_RDY_FOR_STA"	I 55.3	BOOL	// MOTOR 2 READY FOR START
"MTR_2_RUN_FB"	I 55.4	BOOL	// MOTOR 2 RUN FEEDBACK
"MTR_2_OLR_TRP"	I 55.5	BOOL	// MOTOR 2 OVER LOAD TRIP
"CD_LCS_SS_AIR_COMP"	I 55.6	BOOL	// CONTROL DESK/LOCAL CONTROL SELECTOR SWITCH
"MTR_1_2_SS"	I 56.0	BOOL	// MOTOR 1/2 SELECTION
"MTR_1_STA_PB"	I 56.1	BOOL	// MOTOR 1 START PUSH BUTTON
"MTR_1_STP_PB"	I 56.2	BOOL	// MOTOR 1 STOP PUSH BUTTON
"MTR_2_STA_PB"	I 56.3	BOOL	// MOTOR 2 START PUSH BUTTON
"MTR_2_STP_PB"	I 56.4	BOOL	// MOTOR 2 STOP PUSH BUTTON
"MTR_1_2_SS_LCS"	I 56.5	BOOL	// MOTOR 1/2 SELECTION LCS
"MTR_1_STA_PB_LCS"	I 56.6	BOOL	// MOTOR 1 START PUSH BUTTON LCS
"MTR_1_STP_PB_LCS"	I 57.0	BOOL	// MOTOR 1 STOP PUSH BUTTON LCS
"MTR_2_STA_PB_LCS"	I 57.1	BOOL	// MOTOR 2 START PUSH BUTTON LCS
"MTR_2_STP_PB_LCS"	I 57.2	BOOL	// MOTOR 2 STOP PUSH BUTTON LCS
"LCS_24_EMERGENCY_STOP_PB"	I 57.3	BOOL	// LCS-24 EMERGENCY STOP PUSH BUTTON
"CK_SPI_SH_SL_RT_STA_PB"	I 57.4	BOOL	// COKE SPILLAGE SHOVEL  SLEW RETRACT START PUSH BUTTON LCS
"VIB_DOR_CLNR_STA_PB_LCS"	I 57.5	BOOL	// VIBRATOR - DOOR CLEANER START PUSH BUTTON LCS
"VIB_DOR_CLNR_STP_PB_LCS"	I 57.6	BOOL	// VIBRATOR - DOOR CLEANER STOP PUSH BUTTON LCS
"LEV_EM_DRV_DENG_LCS_16"	I 58.0	BOOL	// LEVELER EMERGENCY DRIVE DISENGAGE LCS-16
"COK_SP_SH_SLE_FWD_STA_LC"	I 58.1	BOOL	// COKE SPILLAGE SHOVEL  SLEW FORWARD START PUSH BUTTON LCS
"COK_SP_SH_SLE_RET_STA_LC"	I 58.2	BOOL	// COKE SPILLAGE SHOVEL  SLEW RETRACT START PUSH BUTTON LCS
"COK_SP_SH_SLE_FWD_ST_LCS"	I 58.3	BOOL	// COKE SPILLAGE SHOVEL  SLEW FORWARD START PUSH BUTTON LCS1
"COK_SP_SH_SLE_RET_ST_LCS"	I 58.4	BOOL	// COKE SPILLAGE SHOVEL  SLEW RETRACT START PUSH BUTTON LCS1
"DR_CL_SP_SH_SL_FWD_STA"	I 58.5	BOOL	// DOOR CLEANER SPILLAGE SHOWEL SLEW FORWARD START
"DR_CL_SP_SH_SL_RET_STA"	I 58.6	BOOL	// DOOR CLEANER SPILLAGE SHOWEL SLEW RETRACT START
"DR_CL_SP_SH_SL_FWD_FB"	I 59.0	BOOL	// DOOR CLEANER SPILLAGE SHOWEL SLEW FORWARD FEED BACK
"DR_CL_SP_SH_SL_RET_FB"	I 59.1	BOOL	// DOOR CLEANER SPILLAGE SHOWEL SLEW RETRACT FEED BACK
"DR_CL_SP_HO_FWD_FB"	I 59.2	BOOL	// DOOR  CLEANER SPILLAGE HOPPER FORWARD FEED BACK
"DR_CL_SP_HO_RET_FB"	I 59.3	BOOL	// DOOR  CLEANER SPILLAGE HOPPER RETRACT FEED BACK
"ALWAYS_OFF"	M 0.0	BOOL	// THIS BIT WILL BE ALWAYS OFF
"ALWAYS_ON"	M 0.1	BOOL	// THIS BIT WILL BE ALWAYS ON
"HALF_SECOND_PULSE_TRAIN"	M 0.2	BOOL	// ONE SECOND PULSE - THIS BIT WILL BE ON FOR 500MS AND OFF FOR 500MS
"ONE_SECOND_PULSE"	M 0.3	BOOL	// ONE RAINSING EGDGE PULE WILL BE GENERATED PER SECOND
"EMERGENCY"	M 0.4	BOOL	// EMERGENCY PUSH BUTTON PRESSED
"PULSE_GENERATION_BIT"	M 0.5	BOOL	// PULSE GENERATION BIT
"TEST_FWD_LEV"	M 11.0	BOOL	// TEST FORWARD LEVELER
"TEST_REV_LEV"	M 11.1	BOOL	// TEST REVERSE LEVELER
"TEST_HOME_LEV"	M 11.2	BOOL	// TEST HOME BIT LEVELER
"TEST_DEAD_MAN_LEV"	M 11.3	BOOL	// TEST DEAD MAN PUSH BUTTON LEVELER
"TEST_FWD_PUSH"	M 11.4	BOOL	// TEST FORWARD PUSHER
"TEST_REV_PUSH"	M 11.5	BOOL	// TEST REVERSE PUSHER
"TEST_HOME_PUSH"	M 11.6	BOOL	// TEST HOME BIT PUSHER
"TEST_DEAD_MAN_PUSH"	M 11.7	BOOL	// TEST DEAD MAN PUSH BUTTON PUSHER
"TEST_SPEED_LEV"	MW 10	INT	// TEST SPEED LEVELER
"TEST_SPEED_PUSH"	MW 12	INT	// TEST SPEED PUSHER
"MAIN_PROGRAM"	OB 1	OB 1	// MAIN ROUTINE
"I/O_FLT1"	OB 82	OB 82	// I/O Point Fault 1
"OBNL_FLT"	OB 85	OB 85	// OB Not Loaded Fault
"RACK_FLT"	OB 86	OB 86	// Loss of Rack Fault
"PROG_ERR"	OB 121	OB 121	// Programming Error
"MOD_ERR"	OB 122	OB 122	// Module Access Error
"LEV_ENC_POS"	PID 288	DINT	// LEVELER ENCODER POSITION THROUGH PROFIBUS
"PUSH_ENC_POS"	PID 292	DINT	// PUSHER ENCODER POSITION FEEDBACK THROUGH PROFIBUS
"TRA_DRV_JS_SPD_REF"	PIW 254	INT	// TRAVEL DRIVE SPEED REFERENCE INPUT FROM JOY STICK
"PUSH_DRV_JS_SPD_REF_1"	PIW 256	WORD	// PUSHER DRIVE JOY STICK SPEED REFERENCE
"PUSH_DRV_JS_SPD_REF"	PIW 258	INT	// PUSHER DRIVE JOY STICK SPEED REFERENCE
"LEV_DRV_JS_SPD_REF"	PIW 260	WORD
"VER_COMP_LDT_IN"	PIW 262	INT	// VERTICAL COMPENSATION LDT INPUT VALUE
"DR_LIFT_LDT_VAL_IN"	PIW 264	INT	// DOOR LIFTING LDT VALUE INPUT
"TRA_DRV_1_SPD_REF"	PQW 258	WORD	// TRAVEL DRIVE 1 SPEED REFERENCE
"TRA_DRV_2_SPD_REF"	PQW 260	WORD	// TRAVEL DRIVE 2 SPEED REFERENCE
"LEV_DRV_SPD_REF"	PQW 264	INT	// LEVELER DRIVE SPEED REFERENCE OUTPUT
"LEV_ENC_CTRL_WORD"	PQW 266	INT	// LEVELER ENCODER CONTROL WORD
"PUSH_ENC_CTRL_WORD"	PQW 288	INT	// PUSHER ENCODER CONTROL WORD
"MAIN_PWR_ON_CMD"	Q 0.0	BOOL	// MAIN POWER ON COMMAND
"MAIN_PWR_ON_IND"	Q 0.1	BOOL	// MAIN POWER ON INDICATOR
"CTRL_PWR_ON_IND"	Q 0.2	BOOL	// CONTROL POWER ON INDICATOR
"PUMP_1_ON_CMD"	Q 0.3	BOOL	// PUMP 1 ON COMMAND
"PUMP_2_ON_CMD"	Q 0.4	BOOL	// PUMP 2 ON COMMAND
"CIR_PUMP_ON_CMD"	Q 0.5	BOOL	// CIRCULATION PUMP ON COMMAND
"CLR_FAN_ON_CMD"	Q 0.6	BOOL	// COOLER FAN ON COMMAND
"SYSTEM_RDY_IND"	Q 1.0	BOOL	// SYSTEM READY INDICATOR
"PUMP_1_ON_IND"	Q 1.1	BOOL	// PUMP 1 ON INDICATOR
"PUMP_2_ON_IND"	Q 1.2	BOOL	// PUMP 2 ON INDICATOR LCS
"LCS_41_ON_IND_LCS"	Q 1.3	BOOL	// LCS 41 ON INDICATOR
"PUMP_1_ON_IND_LCS"	Q 1.4	BOOL	// PUMP 1 ON INDICATOR LCS
"PUMP_2_ON_IND_LCS"	Q 1.5	BOOL	// PUMP 2 ON INDICATOR LCS
"CIR_PUMP_ON_IND_LCS"	Q 1.6	BOOL	// CIRCULATION PUMP ON INDICATOR LCS
"CLR_FAN_ON_IND_LCS"	Q 2.0	BOOL	// COOLER FAN ON INDICATOR LCS
"LOW_OIL_LEVEL_IND_LCS"	Q 2.1	BOOL	// LOW OIL LEVEL INDICATOR LCS
"HIGH_OIL_TEMP_IND_LCS"	Q 2.2	BOOL	// HIGH OIL TEMPERATURE INDICATOR LCS
"LOW_OIL_TEMP_IND_LCS"	Q 2.3	BOOL	// LOW OIL TEMPERATURE INDICATOR LCS
"FLTR_CHK_IND_LCS"	Q 2.4	BOOL	// FILTER CHOKE INDICATOR LCS
"ACCM_IN_OPER_IND_LCS"	Q 2.5	BOOL	// ACCUMULATOR IN OPERATION INDICATOR
"HTR_ON_IND_LCS"	Q 2.6	BOOL	// HEATER ON INDICATOR LCS
"DR_CL_SP_SH_SL_FWD_CMD"	Q 2.7	BOOL	// DOOR CLEANER SPILLAGE SHOWEL SLEW FORWARD COMMAND
"TRA_GRP_1_ON_CMD"	Q 3.0	BOOL	// TRAVEL GROUP 1 ON COMMAND
"TRA_GRP_2_ON_CMD"	Q 3.1	BOOL	// TRAVEL GROUP 2 ON COMMAND
"TRA_GRP_1_BRK_ON_CMD"	Q 3.2	BOOL	// TRAVEL GROUP 1 BRAKE ON COMMAND
"SIREN_ON_CMD"	Q 3.3	BOOL	// SIREN ON COMMAND
"TRA_GRP_2_BRK_ON_CMD"	Q 3.4	BOOL	// TRAVEL GROUP 2 BRAKE ON COMMAND
"FLASHER_ON_CMD"	Q 3.5	BOOL	// FLASHER ON COMMAND
"TRA_PER_IND"	Q 3.6	BOOL	// TRAVEL PERMISSION INDICATOR
"PUSH_RAM_BRK_ON_CMD"	Q 4.2	BOOL	// PUSHER RAM BREAK ON COMMAND
"PREP_FOR_PUSH_IND"	Q 4.3	BOOL	// PREPARE FOR PUSHING INDICATOR
"LEV_LOC_IND_LCS_16"	Q 4.4	BOOL	// LEVELER LOCAL SELECTION INDICATION LCS-16
"TRA_DRV_1_FWD_CMD"	Q 4.5	BOOL	// TRAVEL DRIVE 1 FORWARD COMMAND
"DR_CL_SP_HO_FWD_COM"	Q 4.6	BOOL	// DOOR  CLEANER SPILLAGE HOPPER FORWARD COMMAND
"PRESS_REL_VLV_1_ON_CMD"	Q 4.7	BOOL	// PRESSURE RELIEF VALVE 1 ON COMMAND
"LEV_RAM_BRK_ON_CMD"	Q 5.2	BOOL	// LEVELER RAM BRAKE ON COMMAND
"LEV_PERM_IND"	Q 5.3	BOOL	// LEVELING PERMISSION INDICATION
"DR_CL_SP_HO_RET_COM"	Q 5.4	BOOL	// DOOR  CLEANER SPILLAGE HOPPER RETRACT COMMAND
"PUSH_RAM_DE_CARB_VALVE"	Q 5.5	BOOL	// PSUHER RAM DE CARBONISING VALVE
"PUSH_RAM_RACK_TEETH_VLV"	Q 5.6	BOOL	// PUSHER RAM RACK TEETH VALVE
"PRESS_REL_VLV_2_ON_CMD"	Q 5.7	BOOL	// PRESSURE RELIEF VALVE 2 ON COMMAND
"MTR_1_ON_CMD"	Q 6.0	BOOL	// MOTOR 1 ON COMMAND
"MTR_2_ON_CMD"	Q 6.1	BOOL	// MOTOR 2 ON COMMAND
"MTR_1_ON_IND"	Q 6.2	BOOL	// MOTOR 1 ON INDICATOR
"MTR_2_ON_IND"	Q 6.3	BOOL	// MOTOR 2 ON INDICATOR
"MTR_1_ON_IND_LCS"	Q 6.4	BOOL	// MOTOR 1 ON INDICATOR LCS
"MTR_2_ON_IND_LCS"	Q 6.5	BOOL	// MOTOR 2 ON INDICATOR LCS
"LCS_24_ON_IND_LCS"	Q 6.6	BOOL	// LCS-24 ON INDICATOR LCS
"VIB_DOR_CLNR_ON_CMD"	Q 7.0	BOOL	// VIBRATOR - DOOR CLEANER ON COMMAND
"VIB_JMB_CLNR_ON_CMD"	Q 7.1	BOOL	// VIBRATOR - JAMB CLEANER ON COMMAND
"VIB_DOR_CLNR_ON_IND"	Q 7.2	BOOL	// VIBRATOR - DOOR CLEANER ON INDICATOR
"VIB_JMB_CLNR_ON_IND"	Q 7.3	BOOL	// VIBRATOR - JAMB CLEANER ON INDICATOR
"VIB_DOR_CLNR_ON_IND_LCS"	Q 7.4	BOOL	// VIBRATOR - DOOR CLEANER ON INDICATOR LCS
"VIB_JMB_CLNR_ON_IND_LCS"	Q 7.5	BOOL	// VIBRATOR - JAMB CLEANER ON INDICATOR LCS
"LEV_BLOW_MTR_ON_CMD"	Q 7.6	BOOL	// LEVELER BLOWER MOTOR ON COMMAND
"DE_TRA_RELIVE_CMD"	Q 7.7	BOOL	// DOOR EXTRACTOR TRAVEL RELEVE VALVE
"LEV_BLOW_MTR_ON_IND"	Q 8.0	BOOL	// LEVELER BLOWER MOTOR ON INDICATOR
"LEV_BLOW_MTR_ON_IND_LCS"	Q 8.1	BOOL	// LEVELER BLOWER MOTOR ON INDICATOR
"LIFT_PF_UP_ON_CMD"	Q 8.2	BOOL	// LIFT PLATFORM UP ON COMMAND
"LIFT_PF_DN_ON_CMD"	Q 8.3	BOOL	// LIFT PLATFORM DOWN ON COMMAND
"DOOR_FIX_LOCK_IND"	Q 8.4	BOOL	// DOOR FIX LOCK INDICATOR
"DOOR_FIX_UNLK_IND"	Q 8.5	BOOL	// DOOR FIX UNLOCK INDICATOR
"DOOR_FIX_UNLK_IND1"	Q 8.6	BOOL	// DOOR FIX UNLOCK INDICATOR
"TRA_DRV_1_REV_CMD"	Q 8.7	BOOL	// TRAVEL DRIVE 1 REVERSE COMMAND
"ACT_GRP_FWD_CMD"	Q 9.0	BOOL	// ACTUATING GRIP FORWARD START COMMAND
"ACT_GRP_RET_CMD"	Q 9.1	BOOL	// ACTUATING GRIP RETRACT START COMMAND
"SLW_RK_SP_1_FWD_CMD"	Q 9.2	BOOL	// SLEAVING RACK STEP 1 FORWARD COMMAND
"SLW_RK_SP_1_RET_CMD"	Q 9.3	BOOL	// SLEAVING RACK STEP 1 RETRACT COMMAND
"SLW_RK_SP_2_FWD_CMD"	Q 9.4	BOOL	// SLEAVING RACK STEP 2 FORWARD COMMAND
"SLW_RK_SP_2_RET_CMD"	Q 9.5	BOOL	// SLEAVING RACK STEP 2 RETRACT COMMAND
"LEV_WN_FM_CR_UP_CMD"	Q 9.6	BOOL	// LEVELER WINDOW FRAME CLEANER UP COMMAND
"TRA_DRV_2_FWD_CMD"	Q 9.7	BOOL	// TRAVEL DRIVE 2 FORWARD COMMAND
"LEV_WN_FM_CR_DN_CMD"	Q 10.0	BOOL	// LEVELER WINDOW FRAME CLEANER DOWN COMMAND
"SMK_SLVE_SLOW_FWD_CMD"	Q 10.1	BOOL	// SMOKE SLEEVE SLOW FORWARD COMMAND
"SMK_SLVE_SLOW_RET_CMD"	Q 10.2	BOOL	// SMOKE SLEEVE SLOW RETRACT COMMAND
"SMK_SLVE_NORM_FWD_CMD"	Q 10.3	BOOL	// SMOKE SLEEVE NORMAL FORWARD COMMAND
"SMK_SLVE_NORM_REV_CMD"	Q 10.4	BOOL	// SMOKE SLEEVE NORMAL RETRACT COMMAND
"ACT_GRP_FWD_IND"	Q 10.5	BOOL	// ACTUATING GRIP FORWARD INDICATOR
"ACT_GRP_RET_IND"	Q 10.6	BOOL	// ACTUATING GRIP RETRACT INDICATOR
"TRA_DRV_2_REV_CMD"	Q 10.7	BOOL	// TRAVEL DRIVE 2 REVERSE COMMAND
"ACT_GRP_DOOR_ON_HOOK"	Q 11.0	BOOL	// ACTUATOR GRIP DOOR ON HOOK
"SLW_RK_SP_1_FWD_IND"	Q 11.1	BOOL	// SLEAVING RACK STEP 1 FORWARD INDICATOR
"SLW_RK_SP_1_RET_IND"	Q 11.2	BOOL	// SLEAVING RACK STEP 1 RETRACT INDICATOR
"SLW_RK_SP_2_FWD_IND"	Q 11.3	BOOL	// SLEAVING RACK STEP 2 FORWARD INDICATOR
"SLW_RK_SP_2_RET_IND"	Q 11.4	BOOL	// SLEAVING RACK STEP 2 RETRACT INDICATOR
"LEV_WN_FM_CR_UP_IND"	Q 11.5	BOOL	// LEVELER WINDOW FRAME CLEANER UP INDICATOR
"LEV_WN_FM_CR_DN_IND"	Q 11.6	BOOL	// LEVELER WINDOW FRAME CLEANER DOWN INDICATOR
"PUSH_RAM_FWD_CMD"	Q 11.7	BOOL	// PUSHER RAM FORWARD ON COMMAND
"SMK_SLVE_FWD_IND"	Q 12.0	BOOL	// SMOKE SLEEVE FORWARD INDICATOR
"SMK_SLVE_RET_IND"	Q 12.1	BOOL	// SMOKE SLEEVE RETRACT INDICATOR
"ACT_GRP_FWD_IND_LCS"	Q 12.2	BOOL	// ACTUATING GRIP FORWARD INDICATOR LCS
"ACT_GRP_RET_IND_LCS"	Q 12.3	BOOL	// ACTUATING GRIP RETRACT INDICATOR LCS
"ACT_GRP_DOOR_ON_HOOK_LCS"	Q 12.4	BOOL	// ACTUATOR GRIP DOOR ON HOOK LCS
"SLW_RK_SP_1_FWD_IND_LCS"	Q 12.5	BOOL	// SLEAVING RACK STEP 1 FORWARD INDICATOR LCS
"SLW_RK_SP_1_RET_IND_LCS"	Q 12.6	BOOL	// SLEAVING RACK STEP 1 RETRACT INDICATOR LCS
"PUSH_RAM_REV_CMD"	Q 12.7	BOOL	// PUSHER RAM REVERSE COMMAND
"SLW_RK_SP_2_FWD_IND_LCS"	Q 13.0	BOOL	// SLEAVING RACK STEP 2 FORWARD INDICATOR LCS
"SLW_RK_SP_2_RET_IND_LCS"	Q 13.1	BOOL	// SLEAVING RACK STEP 2 RETRACT INDICATOR LCS
"LEV_WN_FM_CR_UP_IND_LCS"	Q 13.2	BOOL	// LEVELER WINDOW FRAME CLEANER UP INDICATOR LCS
"LEV_WN_FM_CR_DN_IND_LCS"	Q 13.3	BOOL	// LEVELER WINDOW FRAME CLEANER DOWN INDICATOR LCS
"SMK_SLVE_FWD_IND_LCS"	Q 13.4	BOOL	// SMOKE SLEEVE FORWARD INDICATOR LCS
"SMK_SLVE_RET_IND_LCS"	Q 13.5	BOOL	// SMOKE SLEEVE RETRACT INDICATOR LCS
"LCS_61_ON_INDICATOR"	Q 13.6	BOOL	// LCS 61 ON INDICATOR
"LEV_DRV_FWD_CMD"	Q 13.7	BOOL	// LEVELER DRIVE FORWARD COMMAND
"LEV_DRV_ENG_UP_CMD"	Q 14.0	BOOL	// LEVELER PNEUMATIC EMERGENCY DRIVE LEVEL UP COMMAND
"LEV_ENG_DRV_DN_CMD"	Q 14.1	BOOL	// LEVELER EMERGENCY PNEUMATIC DRIVE LEVEL DOWN COMMAND
"RAMU_ENG_DRV_UP_CMD"	Q 14.2	BOOL	// RAM PNEUMATIC EMERGENCY DRIVE UP COMMAND
"RAM_ENG_DRV_DN_CMD"	Q 14.3	BOOL	// RAM PNEUMATIC EMERGENCY DRIVE DOWN COMMAND
"LEV_EM_DRV_ENG_IND_LC_15"	Q 14.4	BOOL	// LEVELER EMERGENCY DRIVE ENGAGE INDICATOR LCS-15
"COK_SPI_SH_SL_RET_CMD"	Q 14.5	BOOL	// COKE SPILLAGE SHOVEL SLEW RETRACT COMMAND
"COK_SPI_SH_SL_FWD_IND"	Q 14.6	BOOL	// COKE SPILLAGE SHOVEL SLEW FORWARD INDICATOR
"LEV_DRV_REV_CMD"	Q 14.7	BOOL	// LEVELER DRIVE REVERSE COMMAND
"TRA_SIR_ON_CMD"	Q 15.0	BOOL	// TRAVEL SIREN ON COMMAND
"PUSH_RAM_HOOT"	Q 15.1	BOOL	// PUSHER_RAM_HOOTER
"SLEW_NOR_FWD_COMMAND"	Q 15.2	BOOL	// SLEW NORMAL FORWARD COMMAND
"SLEW_NOR_RET_COMMAND"	Q 15.3	BOOL	// SLEW NORMAL RETRACT COMMAND
"VER_COMP_FWD_CMD"	Q 15.4	BOOL	// VERTICAL COMPENSATION FORWARD COMMAND
"VER_COMP_RET_CMD"	Q 15.5	BOOL	// VERTICAL COMPENSATION RETRACT COMMAND
"VER_COMP_RELIVE_CMD"	Q 15.6	BOOL	// VERTICAL COMPENSTAION RELIVE  COOMMAND
"DR_CL_SP_SH_SL_RET_CMD"	Q 15.7	BOOL	// DOOR CLEANER SPILLAGE SHOWEL SLEW RETRACT COMMAND
"TRA_SLOW_FWD_CMD"	Q 16.0	BOOL	// TRAVEL SLOW FORWARD COMMAND
"TRA_SLOW_RET_CMD"	Q 16.1	BOOL	// TRAVEL SLOW RETRACT COMMAND
"TRA_NORM_FWD_CMD"	Q 16.2	BOOL	// TRAVEL NORMAL FORWARD COMMAND
"TRA_NORM_RET_CMD"	Q 16.3	BOOL	// TRAVEL NORMAL RETRACT COMMAND
"MAN_FNL_STK_UP_CMD"	Q 16.4	BOOL	// MANUAL AND FINAL STROKE  UP COMMAND
"MAN_FNL_STK_DN_CMD"	Q 16.5	BOOL	// MANUAL AND FINAL STROKE  DN COMMAND
"PRE_STK_UP_CMD"	Q 16.6	BOOL	// PRE STROKE  UP COMMAND
"AUTO_POS_ON"	Q 16.7	BOOL	// AUTO POSITION ON
"PRE_STK_DN_CMD"	Q 17.0	BOOL	// PRE STROKE  DN COMMAND
"DOOR_SPRG_PRS_LOCK_CMD"	Q 17.1	BOOL	// DOOR SPRING PRESS LOCK COMMAND
"DOOR_SPRG_PRS_UNLK_CMD"	Q 17.2	BOOL	// DOOR SPRING PRESS UNLOCK COMMAND
"DOOR_LCH_TURN_UP_CMD"	Q 17.3	BOOL	// DOOR LATCH TURNING UP COMMAND
"DOOR_LCH_TURN_DOWN_CMD"	Q 17.4	BOOL	// DOOR LATCH TURNING DOWN COMMADN
"DE_SLEW_FWD_IND"	Q 17.5	BOOL	// SLEW FORWARD INDICATOR
"SLEW_SLOW_RET_IND"	Q 17.6	BOOL	// SLEW SLOW RETRACT INDICATOR
"SLEW_SLOW_FWD_IND"	Q 17.7	BOOL	// SLEW SLOW FORWARD INDICATOR
"VER_COMP_FWD_IND"	Q 18.0	BOOL	// VERTICAL COMPENSATION FORWARD INDICATOR
"VER_COMP_RET_IND"	Q 18.1	BOOL	// VERTICAL COMPENSATION RETRACT INDICATOR
"TRA_FWD_IND"	Q 18.2	BOOL	// TRAVEL FORWARD INDICATOR
"TRA_BACK_IND"	Q 18.3	BOOL	// TRAVEL BACK INDICATOR
"MAN_STK_UP_IND"	Q 18.4	BOOL	// FINAL STROKE  UP INDICATION
"MAN_STK_DN_IND"	Q 18.5	BOOL	// FINAL STROKE  DOWN  INDICATOR
"FNL_STK_UP_IND"	Q 18.6	BOOL	// FINAL STROKE  UP INDICATOR
"FNL_STK_DN_IND"	Q 19.0	BOOL	// FINAL STROKE  DOWN INDICATOR
"PRE_STK_UP_IND"	Q 19.1	BOOL	// PRE STROKE  UP INDICATION
"PRE_STK_DN_IND"	Q 19.2	BOOL	// PRE STROKE  DOWN INDICATOR
"DOOR_SPRG_PRS_LOCK_IND"	Q 19.3	BOOL	// DOOR SPRING PRESS LOCK INDICATOR
"DOOR_SPRG_PRS_UNLK_IND"	Q 19.4	BOOL	// DOOR SPRING PRESS UNLOCK INDICATOR
"DR_CL_SP_SH_SL_FWD_IND_L"	Q 19.5	BOOL	// DOOR CLEANER SPILLAGE SHOWEL SLEW FORWARD INDICATOR LCS
"DR_CL_SP_SH_SL_RET_IND_L"	Q 19.6	BOOL	// DOOR CLEANER SPILLAGE SHOWEL SLEW RETRACT INDICATOR LCS
"LCS_73_ON_IND"	Q 20.0	BOOL	// LCS-73_ON_INDICATOR
"SLEW_SLOW_FWD_IND_LCS"	Q 20.1	BOOL	// SLEW SLOW FORWARD INDICATOR LCS
"SLEW_SLOW_RET_IND_LCS"	Q 20.2	BOOL	// SLEW SLOW RETRACT INDICATOR LCS
"VER_COMP_FWD_IND_LCS"	Q 20.3	BOOL	// VERTICAL COMPENSATION FORWARD INDICATOR LCS
"VER_COMP_RET_IND_LCS"	Q 20.4	BOOL	// VERTICAL COMPENSATION RETRACT INDICATOR LCS
"TRA_FWD_IND_LCS"	Q 20.5	BOOL	// TRAVEL FORWARD INDICATOR
"TRA_BACK_IND_LCS"	Q 20.6	BOOL	// TRAVEL BACK INDICATOR LCS
"MAN_STK_UP_IND_LCS"	Q 21.0	BOOL	// FINAL STROKE  UP INDICATION LCS
"MAN_STK_DN_IND_LCS"	Q 21.1	BOOL	// FINAL STROKE  DOWN  INDICATOR LCS
"FNL_STK_UP_IND_LCS"	Q 21.2	BOOL	// FINAL STROKE  UP INDICATOR LCS
"FNL_STK_DN_IND_LCS"	Q 21.3	BOOL	// FINAL STROKE  DOWN INDICATOR LCS
"PRE_STK_UP_IND_LCS"	Q 21.4	BOOL	// PRE STROKE  UP INDICATION LCS
"PRE_STK_DN_IND_LCS"	Q 21.5	BOOL	// PRE STROKE  DOWN INDICATOR LCS
"DR_CL_SP_HO_FWD_IND_LCS"	Q 21.6	BOOL	// DOOR  CLEANER SPILLAGE HOPPER FORWARD INDICATOR
"DOOR_LAT_TUR_DN_IND_LCS"	Q 22.0	BOOL	// DOOR LATCH TURNING  DOWN  INDICATOR LCS
"DOOR_LAT_TUR_UP_IND_LCS"	Q 22.1	BOOL	// DOOR LATCH TURNING  UP INDICATOR LCS
"DR_CL_SP_HO_RET_IND_LCS"	Q 22.2	BOOL	// DOOR  CLEANER SPILLAGE HOPPER RETRACT INDICATOR
"DOOR_LAT_HOME"	Q 22.3	BOOL	// DOOR LATCH  HOME
"DR_SPNG_LK_IND_LCS"	Q 22.4	BOOL	// DOOR SPRING PRESSURE LOCK INDICATOR LCS
"DR_SPNG_UNLK_IND_LCS"	Q 22.5	BOOL	// DOOR SPRING PRESSURE UNLOCK INDICATOR LCS
"CAR_TRA_FWD_CMD"	Q 23.0	BOOL	// DOOR CLEANER CARRIAGE FORWARD TRAVEL COMMAND
"CAR_TRA_RET_CMD"	Q 23.1	BOOL	// DOOR CLEANER CARRIAGE RETRACT TRAVEL COMMAND
"VER_CLNR_UP_CMD"	Q 23.2	BOOL	// DOOR CLEANER VERTICAL CLEANER UP COMMAND
"VER_CLNR_DOWN_CMD"	Q 23.3	BOOL	// DOOR CLEANER VERTICAL CLEANER DOWN COMMAND
"GRV_SCRPR_1_FWD_CMD"	Q 23.4	BOOL	// DOOR CLEANER GROOVE SCRAPPER 1 FWD COMMAND
"GRV_SCRPR_1_RET_CMD"	Q 23.5	BOOL	// DOOR CLEANER GROOVE SCRAPPER 1 RET COMMAND
"TOP_SCRP_FWD_CMD"	Q 23.6	BOOL	// DOOR CLEANER TOP SCRAPPER FORWARD COMMAND
"TOP_SCRP_REV_CMD"	Q 24.0	BOOL	// DOOR CLEANER TOP SCRAPPER REVERSE COMMAND
"BTM_SCRP_FWD_CMD"	Q 24.1	BOOL	// DOOR CLEANER BOTTOM SCRAPPER FORWARD COMMAND
"BTM_SCRP_REV_CMD"	Q 24.2	BOOL	// DOOR CLEANER BOTTOM SCRAPPER REVERSE COMMAND
"CAR_TRA_FWD_IND_CD"	Q 24.3	BOOL	// DOOR CLEANER CARRIAGE FORWARD TRAVEL INDICATOR CONTROL DESK
"CAR_TRA_RET_IND_CD"	Q 24.4	BOOL	// DOOR CLEANER CARRIAGE RETRACT TRAVEL INDICATOR CONTROL DESK
"VER_CLNR_UP_IND_CD"	Q 24.5	BOOL	// DOOR CLEANER VERTICAL CLEANER UP INDICATOR CONTROL DESK
"VER_CLNR_DOWN_IND_CD"	Q 24.6	BOOL	// DOOR CLEANER VERTICAL CLEANER DOWN INDICATOR CONTROL DESK
"GRV_SRPR_FWD_IND_CD"	Q 25.0	BOOL	// DOOR CLEANER GROOVE SCRAPPER FORWARD INDICATOR CONTROL DESK
"GRV_SRPR_RET_IND_CD"	Q 25.1	BOOL	// DOOR CLEANER GROOVE SCRAPPER REVERSE INDICATOR CONTROL DESK
"TOP_SCRP_FWD_IND_CD"	Q 25.2	BOOL	// DOOR CLEANER TOP SCRAPPER FORWARD INDICATOR CONTROL DESK
"TOP_SCRP_REV_IND_CD"	Q 25.3	BOOL	// DOOR CLEANER TOP SCRAPPER REVERSE INDICATOR CONTROL DESK
"BTM_SCRP_FWD_IND_CD"	Q 25.4	BOOL	// DOOR CLEANER BOTTOM SCRAPPER FORWARD INDICATOR CONTROL DESK
"BTM_SCRP_REV_IND_CD"	Q 25.5	BOOL	// DOOR CLEANER BOTTOM SCRAPPER REVERSE INDICATOR CONTROL DESK
"CAR_TRA_FWD_IND_LCS"	Q 25.6	BOOL	// DOOR CLEANER CARRIAGE FORWARD TRAVEL INDICATOR LOCAL CONTROL PANEL
"CAR_TRA_RET_IND_LCS"	Q 26.0	BOOL	// DOOR CLEANER CARRIAGE RETRACT TRAVEL INDICATOR LOCAL CONTROL PANEL
"VER_CLNR_UP_IND_LCS"	Q 26.1	BOOL	// DOOR CLEANER VERTICAL CLEANER UP INDICATOR LOCAL CONTROL PANEL
"VER_CLNR_DOWN_IND_LCS"	Q 26.2	BOOL	// DOOR CLEANER VERTICAL CLEANER DOWN INDICATOR LOCAL CONTROL PANEL
"BRK_HLDR_FWD_IND_LCS"	Q 26.3	BOOL	// DOOR CLEANER BRICK HOLDER FORWARD INDICATOR LOCAL CONTROL PANEL
"BRK_HLDR_REV_IND_LCS"	Q 26.4	BOOL	// DOOR CLEANER BRICK HOLDER REVERSE INDICATOR LOCAL CONTROL PANEL
"TOP_SCRP_FWD_IND_LCS"	Q 26.5	BOOL	// DOOR CLEANER TOP SCRAPPER FORWARD INDICATOR LOCAL CONTROL PANEL
"TOP_SCRP_REV_IND_LCS"	Q 26.6	BOOL	// DOOR CLEANER TOP SCRAPPER REVERSE INDICATOR LOCAL CONTROL PANEL
"BTM_SCRP_FWD_IND_LCS"	Q 27.0	BOOL	// DOOR CLEANER BOTTOM SCRAPPER FORWARD INDICATOR LOCAL CONTROL PANEL
"BTM_SCRP_REV_IND_LCS"	Q 27.1	BOOL	// DOOR CLEANER BOTTOM SCRAPPER REVERSE INDICATOR LOCAL CONTROL PANEL
"LCS_85_ON_IND"	Q 27.2	BOOL	// LCS 85 ON INDICATION
"GRV_SCRPR_ON_IND"	Q 27.3	BOOL	// DOOR CLEANER GROOVE SCRAPPER ON INDICATOR LCS
"GRV_SCRPR_OFF_IND"	Q 27.4	BOOL	// DOOR CLEANER GROOVE SCRAPPER OFF INDICATOR LCS
"GRV_SCRPR_2_FWD_CMD"	Q 27.5	BOOL	// DOOR CLEANER GROOVE SCRAPPER 2 FWD COMMAND
"GRV_SCRPR_2_RET_CMD"	Q 27.6	BOOL	// DOOR CLEANER GROOVE SCRAPPER 2 RET COMMAND
"SLEW_NORMAL_RET_CMD"	Q 28.0	BOOL	// SLEW NORMAL RETRACT COMMAND
"JC_TRA_SLOW_FWD_CMD"	Q 28.1	BOOL	// JAMP CLEANER TRAVEL SLOW FORWARD COMMAND
"JC_TRA_SLOW_RET_CMD"	Q 28.2	BOOL	// JAMP CLEANER TRAVEL SLOW RETRACT COMMAND
"TRA_NORMAL_FWD_CMD"	Q 28.3	BOOL	// TRAVEL NORMAL FORWARD COMMAND
"TRA_NORMAL_RET_CMD"	Q 28.4	BOOL	// TRAVEL NORMAL RETRACT COMMAND
"VER_CLE_UP_CMD"	Q 28.5	BOOL	// VERTICAL CLEANER UP COMMAND
"VER_CLE_DN_CMD"	Q 28.6	BOOL	// VERTICAL CLEANER DN COMMAND
"JC_SLEW_FWD_IND"	Q 29.0	BOOL	// SLEW FORWARD INDICATOR
"SLEW_RET_IND"	Q 29.1	BOOL	// SLEW RETRACT INDICATOR
"JC_TRA_FWD_IND"	Q 29.2	BOOL	// TRAVEL FORWARD INDICATOR
"TRA_RET_IND"	Q 29.3	BOOL	// TRAVEL RETRACT INDICATOR
"VER_CLE_UP_IND"	Q 29.4	BOOL	// VERTICAL CLEANER UP INDICATOR
"VER_CLE_DN_IND"	Q 29.5	BOOL	// VERTICAL CLEANER DN INDICATOR
"SLEW_FWD_IND_LCS"	Q 29.7	BOOL	// SLEW FORWARD INDICATOR LCS
"SLEW_RET_IND_LCS"	Q 30.0	BOOL	// SLEW RETRACT INDICATOR LCS
"JC_TRA_FWD_IND_LCS"	Q 30.1	BOOL	// TRAVEL FORWARD INDICATOR LCS
"TRA_RET_IND_LCS"	Q 30.2	BOOL	// TRAVEL RETRACT INDICATOR LCS
"VER_CLE_UP_IND_LCS"	Q 30.3	BOOL	// VERTICAL CLEANER UP INDICATOR LCS
"VER_CLE_DN_IND_LCS"	Q 30.4	BOOL	// VERTICAL CLEANER DN INDICATOR
"LCS_90_ON_IND"	Q 30.5	BOOL	// LCS-90 ON INDICATOR
"SLEW_NORMAL_FWD_CMD"	Q 30.6	BOOL	// SLEW NORMAL FORWARD COMMAND
"CNT_TH_WED_UP_CMD"	Q 31.0	BOOL	// COUNTER  THRUST WEDGE UP COMMAND
"CNT_TH_WED_DN_CMD"	Q 31.1	BOOL	// COUNTER  THRUST WEDGE DN COMMAND
"CNT_TH_WED_UP_IND"	Q 31.2	BOOL	// COUNTER  THRUST WEDGE UP INDICATOR
"CNT_TH_WED_DN_IND"	Q 31.3	BOOL	// COUNTER  THRUST WEDGE DN INDICATOR
"CNT_TH_WED_UP_IND_LCS"	Q 31.4	BOOL	// COUNTER  THRUST WEDGE UP INDICATOR LCS
"CNT_TH_WED_DN_IND_LCS"	Q 31.5	BOOL	// COUNTER  THRUST WEDGE DN INDICATOR LCS
"CNT_WED_LOC_IND_LCS"	Q 31.6	BOOL	// COUNTER  THRUST WEDGE LOCAL INDICATOR LCS
"CO_SPI_CHU_UP_CMD"	Q 32.0	BOOL	// COAL SPILLAGE CHUTE UP COMMAND
"CO_SPI_CHU_DN_CMD"	Q 32.1	BOOL	// COAL SPILLAGE CHUTE DOWN COMMAND
"CO_SP_CHT_HO_GT_OP_CMD"	Q 32.2	BOOL	// COAL SPILLAGE CHUTE HOPPER GATE OPEN COMMAND
"CO_SP_CHT_HO_GT_CL_CMD"	Q 32.3	BOOL	// COAL SPILLAGE CHUTE HOPPER GATE CLOSE COMMAND
"CO_SP_CHT_UP_IND"	Q 32.4	BOOL	// COAL SPILLAGE CHUTE UP INDICATOR
"CO_SP_CHT_DN_IND"	Q 32.5	BOOL	// COAL SPILLAGE CHUTE DOWN INDICATOR
"CO_SP_CHT_DN_IND_LCS"	Q 32.6	BOOL	// COAL SPILLAGE CHUTE DOWN INDICATOR LCS
"CO_SP_CHT_UP_IND_LCS"	Q 33.0	BOOL	// COAL SPILLAGE CHUTE UP INDICATOR LCS
"CO_SPI_HOP_GT_OP_IND_LCS"	Q 33.1	BOOL	// COAL SPILLAGE HOPPER GATE OPEN INDICATOR LCS
"CO_SPI_HOP_GT_CL_IND_LCS"	Q 33.2	BOOL	// COAL SPILLAGE HOPPER GATE CLOSE INDICATOR LCS
"PREP_DOOR_FUNC_IND"	Q 33.3	BOOL	// PREPARE DOOR FUNCTION INDICATOR
"FIN_DOOR_FUNC_IND"	Q 33.4	BOOL	// FINISH DOOR FUNCTION INDICATOR
"EXT_OVEN_DOR_IND"	Q 33.5	BOOL	// EXTRACT OVEN DOOR INDICATOR
"RPL_OVEN_DOR_IND"	Q 33.6	BOOL	// REPLACE OVEN DOOR INDICATOR
"CLEAN_OVN_DR_IND"	Q 34.0	BOOL	// CLEAN OVEN DOOR AUTO INDICATION
"STA_PUSH_IND"	Q 34.1	BOOL	// START PUSHING INDICATION
"CLEAN_OVN_DOOR_IND"	Q 34.2	BOOL	// CLEAN OVEN DOOR INDICATION
"PREP_FOR_LEV_IND"	Q 34.3	BOOL	// PREPARE FOR LEVELING INDICATION
"FIN_LEV_PERM_IND"	Q 34.4	BOOL	// FINISH LEVELING PERMISION INDICATOR
"STA_LEV_IND"	Q 34.5	BOOL	// START LEVELING INDICATION
"PUSH_RAM_REV_END_IND"	Q 34.6	BOOL	// PUSHER RAM FULLY BACK INDICATION
"LEV_RAM_REV_END_IND"	Q 35.0	BOOL	// LEVELER BAR FULLY BACK INDICATOR
"COK_SPI_SH_SL_FWD_CMD"	Q 35.1	BOOL	// COKE SPILLAGE SHOVEL SLEW FORWARD COMMAND
"DR_CL_SP_SH_SL_FWD_IND"	Q 35.2	BOOL	// DOOR CLEANER SPILLAGE SHOWEL SLEW FORWARD INDICATOR
"DR_CL_SP_SH_SL_RET_IND"	Q 35.3	BOOL	// DOOR CLEANER SPILLAGE SHOWEL SLEW RETRACT INDICATOR
"COK_SPI_SH_SL_RET_IND"	Q 35.4	BOOL	// COKE SPILLAGE SHOVEL SLEW RETRACT INDICATOR
"COK_SPI_SH_SL_FWD_IND_LC"	Q 35.5	BOOL	// COKE SPILLAGE SHOVEL SLEW FORWARD INDICATOR LCS
"COK_SPI_SH_SL_RET_IND_L"	Q 35.6	BOOL	// COKE SPILLAGE SHOVEL SLEW RETRACT INDICATOR LCS
"EMG_ACCM_ON_CMD"	Q 36.5	BOOL	// EMERGENCY ACCUMULLATOR ON COMMAND
"PUSH_DRV_REV_CMD"	Q 37.1	BOOL	// PUSHER DRIVE REVERSE COMMAND
"DPRD_DAT"	SFC 14	SFC 14	// Read Consistent Data of a Standard DP Slave
"DPWR_DAT"	SFC 15	SFC 15	// Write Consistent Data to a Standard DP Slave
"PRE_STK_UP_CMD_TMR"	T 50	TIMER	// PRE STROKE UP COMMAND TIMER
"PRE_STK_DN_CMD_TMR"	T 51	TIMER	// PRE STROKE DOWN COMMAND TIMER
"MAIN_STK_UP_CMD_TMR"	T 52	TIMER	// MAIN STROKE UP COMMAND TIMER
"MAIN_STK_DN_CMD_TMR"	T 53	TIMER	// MAIN STROKE DOWN COMMAND TIMER
"FIN_STK_UP_CMD_TMR"	T 54	TIMER	// FINAL STROKE UP COMMAND TIMER
"FIN_STK_DN_CMD_TMR"	T 55	TIMER	// FINAL STROKE DOWN COMMAND TIMER
"COUNTER_MODULE_DATA_TYPE"	UDT 2	UDT 2
"ANALOG_VALUE"	VAT 1	
END_SYMBOL_TABLE

FUNCTION "INPUT_MAPPING" : VOID	// FC 1
AUTHOR : Kamillas
VERSION : 0.1
BEGIN
// (block stored without names or comments; labels and parameter names are numbered)
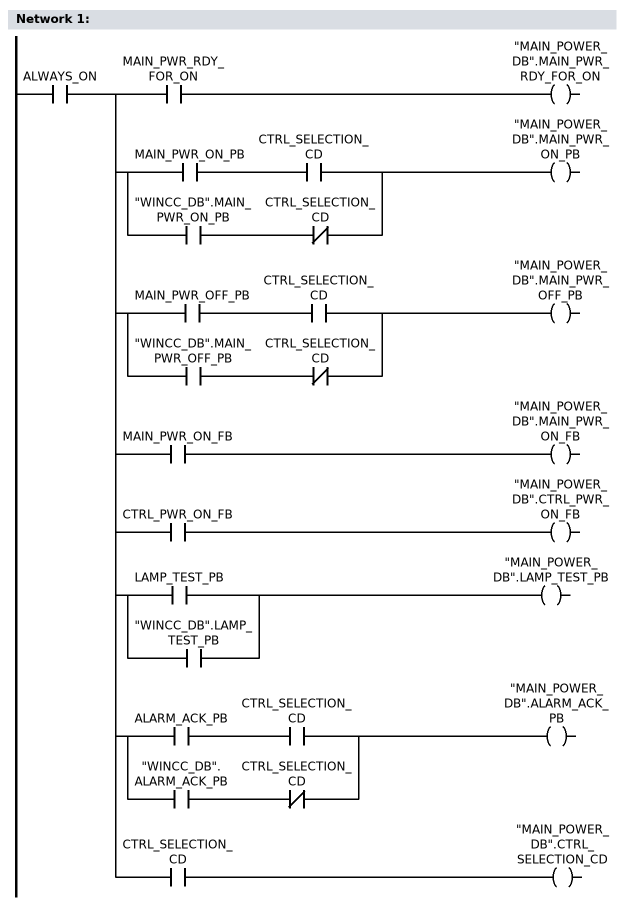
NETWORK
TITLE =
      A     "ALWAYS_ON";
      =     L 0.0;
      A     L 0.0;
      A     "MAIN_PWR_RDY_FOR_ON";
      =     "MAIN_POWER_DB".MAIN_PWR_RDY_FOR_ON;
      A     L 0.0;
      A(;
      A     "MAIN_PWR_ON_PB";
      A     "CTRL_SELECTION_CD";
      O;
      A     "WINCC_DB".MAIN_PWR_ON_PB;
      AN    "CTRL_SELECTION_CD";
      );
      =     "MAIN_POWER_DB".MAIN_PWR_ON_PB;
      A     L 0.0;
      A(;
      A     "MAIN_PWR_OFF_PB";
      A     "CTRL_SELECTION_CD";
      O;
      A     "WINCC_DB".MAIN_PWR_OFF_PB;
      AN    "CTRL_SELECTION_CD";
      );
      =     "MAIN_POWER_DB".MAIN_PWR_OFF_PB;
      A     L 0.0;
      A     "MAIN_PWR_ON_FB";
      =     "MAIN_POWER_DB".MAIN_PWR_ON_FB;
      A     L 0.0;
      A     "CTRL_PWR_ON_FB";
      =     "MAIN_POWER_DB".CTRL_PWR_ON_FB;
      A     L 0.0;
      A(;
      O     "LAMP_TEST_PB";
      O     "WINCC_DB".LAMP_TEST_PB;
      );
      =     "MAIN_POWER_DB".LAMP_TEST_PB;
      A     L 0.0;
      A(;
      A     "ALARM_ACK_PB";
      A     "CTRL_SELECTION_CD";
      O;
      A     "WINCC_DB".ALARM_ACK_PB;
      AN    "CTRL_SELECTION_CD";
      );
      =     "MAIN_POWER_DB".ALARM_ACK_PB;
      A     L 0.0;
      A     "CTRL_SELECTION_CD";
      =     "MAIN_POWER_DB".CTRL_SELECTION_CD;
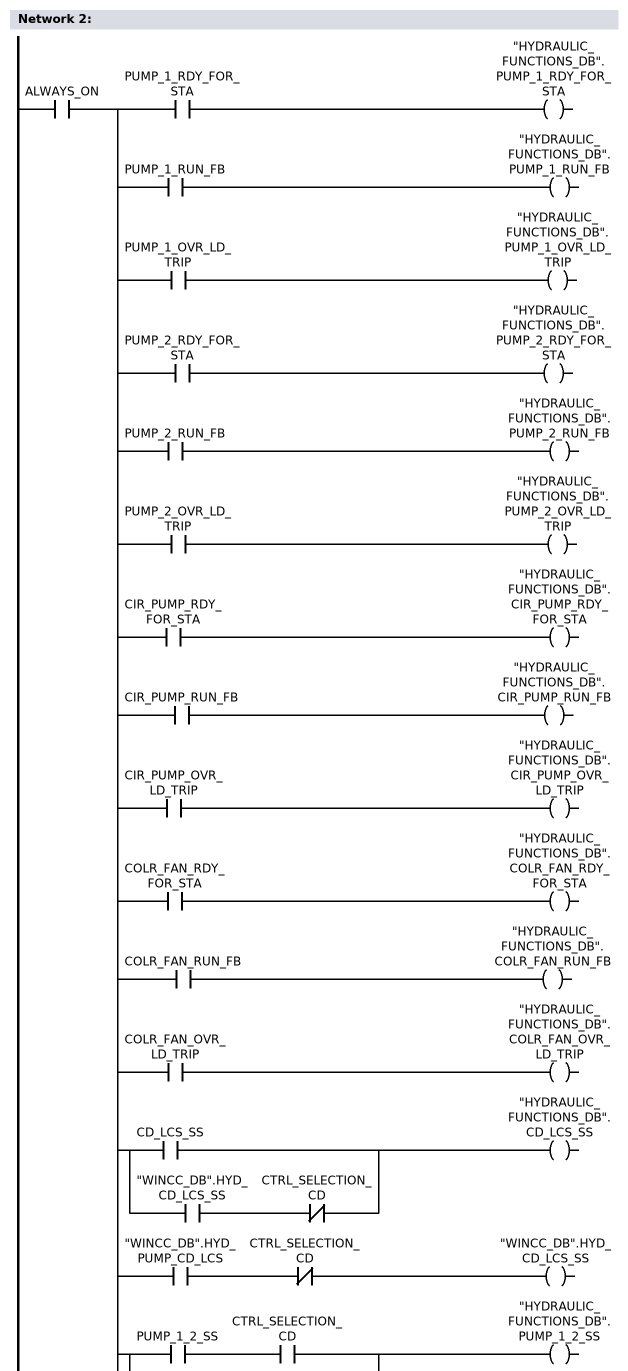
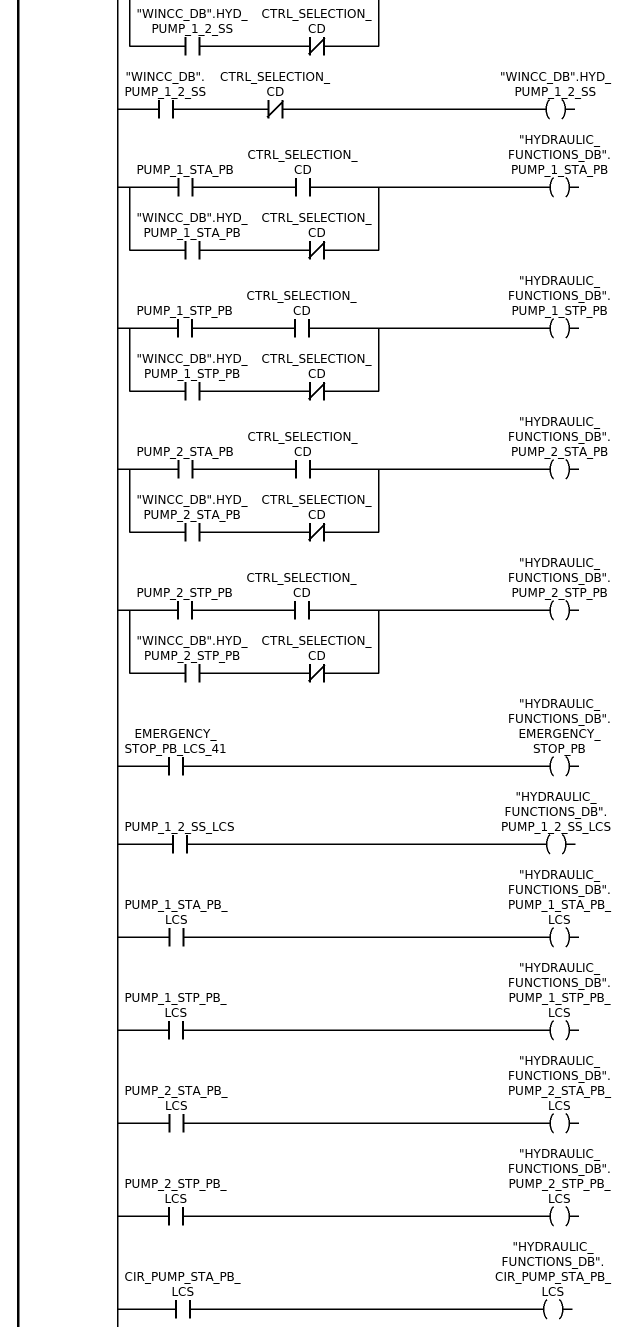
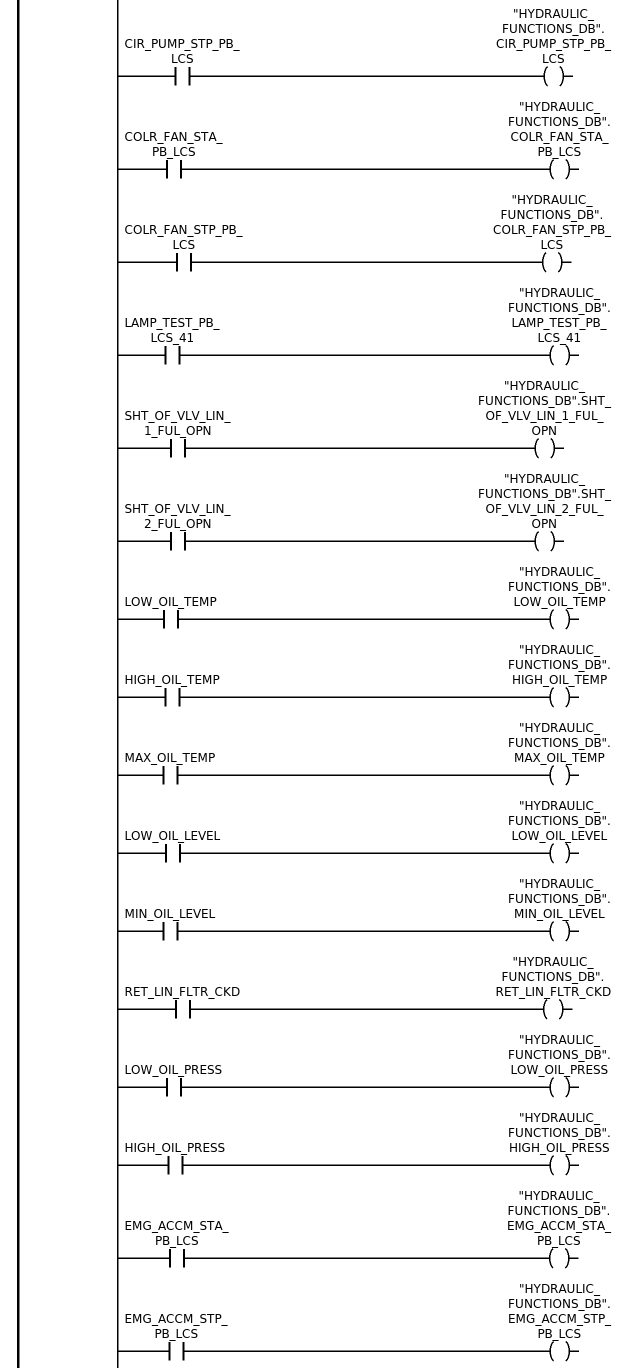
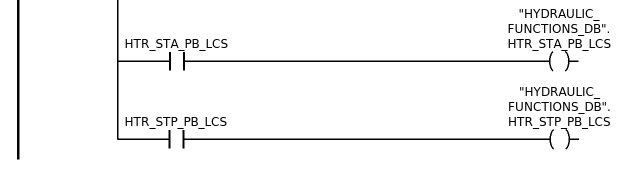
NETWORK
TITLE =
      A     "ALWAYS_ON";
      =     L 0.0;
      A     L 0.0;
      A     "PUMP_1_RDY_FOR_STA";
      =     "HYDRAULIC_FUNCTIONS_DB".PUMP_1_RDY_FOR_STA;
      A     L 0.0;
      A     "PUMP_1_RUN_FB";
      =     "HYDRAULIC_FUNCTIONS_DB".PUMP_1_RUN_FB;
      A     L 0.0;
      A     "PUMP_1_OVR_LD_TRIP";
      =     "HYDRAULIC_FUNCTIONS_DB".PUMP_1_OVR_LD_TRIP;
      A     L 0.0;
      A     "PUMP_2_RDY_FOR_STA";
      =     "HYDRAULIC_FUNCTIONS_DB".PUMP_2_RDY_FOR_STA;
      A     L 0.0;
      A     "PUMP_2_RUN_FB";
      =     "HYDRAULIC_FUNCTIONS_DB".PUMP_2_RUN_FB;
      A     L 0.0;
      A     "PUMP_2_OVR_LD_TRIP";
      =     "HYDRAULIC_FUNCTIONS_DB".PUMP_2_OVR_LD_TRIP;
      A     L 0.0;
      A     "CIR_PUMP_RDY_FOR_STA";
      =     "HYDRAULIC_FUNCTIONS_DB".CIR_PUMP_RDY_FOR_STA;
      A     L 0.0;
      A     "CIR_PUMP_RUN_FB";
      =     "HYDRAULIC_FUNCTIONS_DB".CIR_PUMP_RUN_FB;
      A     L 0.0;
      A     "CIR_PUMP_OVR_LD_TRIP";
      =     "HYDRAULIC_FUNCTIONS_DB".CIR_PUMP_OVR_LD_TRIP;
      A     L 0.0;
      A     "COLR_FAN_RDY_FOR_STA";
      =     "HYDRAULIC_FUNCTIONS_DB".COLR_FAN_RDY_FOR_STA;
      A     L 0.0;
      A     "COLR_FAN_RUN_FB";
      =     "HYDRAULIC_FUNCTIONS_DB".COLR_FAN_RUN_FB;
      A     L 0.0;
      A     "COLR_FAN_OVR_LD_TRIP";
      =     "HYDRAULIC_FUNCTIONS_DB".COLR_FAN_OVR_LD_TRIP;
      A     L 0.0;
      A(;
      O     "CD_LCS_SS";
      O;
      A     "WINCC_DB".HYD_CD_LCS_SS;
      AN    "CTRL_SELECTION_CD";
      );
      =     "HYDRAULIC_FUNCTIONS_DB".CD_LCS_SS;
      A     L 0.0;
      A     "WINCC_DB".HYD_PUMP_CD_LCS;
      AN    "CTRL_SELECTION_CD";
      =     "WINCC_DB".HYD_CD_LCS_SS;
      A     L 0.0;
      A(;
      A     "PUMP_1_2_SS";
      A     "CTRL_SELECTION_CD";
      O;
      A     "WINCC_DB".HYD_PUMP_1_2_SS;
      AN    "CTRL_SELECTION_CD";
      );
      =     "HYDRAULIC_FUNCTIONS_DB".PUMP_1_2_SS;
      A     L 0.0;
      A     "WINCC_DB".PUMP_1_2_SS;
      AN    "CTRL_SELECTION_CD";
      =     "WINCC_DB".HYD_PUMP_1_2_SS;
      A     L 0.0;
      A(;
      A     "PUMP_1_STA_PB";
      A     "CTRL_SELECTION_CD";
      O;
      A     "WINCC_DB".HYD_PUMP_1_STA_PB;
      AN    "CTRL_SELECTION_CD";
      );
      =     "HYDRAULIC_FUNCTIONS_DB".PUMP_1_STA_PB;
      A     L 0.0;
      A(;
      A     "PUMP_1_STP_PB";
      A     "CTRL_SELECTION_CD";
      O;
      A     "WINCC_DB".HYD_PUMP_1_STP_PB;
      AN    "CTRL_SELECTION_CD";
      );
      =     "HYDRAULIC_FUNCTIONS_DB".PUMP_1_STP_PB;
      A     L 0.0;
      A(;
      A     "PUMP_2_STA_PB";
      A     "CTRL_SELECTION_CD";
      O;
      A     "WINCC_DB".HYD_PUMP_2_STA_PB;
      AN    "CTRL_SELECTION_CD";
      );
      =     "HYDRAULIC_FUNCTIONS_DB".PUMP_2_STA_PB;
      A     L 0.0;
      A(;
      A     "PUMP_2_STP_PB";
      A     "CTRL_SELECTION_CD";
      O;
      A     "WINCC_DB".HYD_PUMP_2_STP_PB;
      AN    "CTRL_SELECTION_CD";
      );
      =     "HYDRAULIC_FUNCTIONS_DB".PUMP_2_STP_PB;
      A     L 0.0;
      A     "EMERGENCY_STOP_PB_LCS_41";
      =     "HYDRAULIC_FUNCTIONS_DB".EMERGENCY_STOP_PB;
      A     L 0.0;
      A     "PUMP_1_2_SS_LCS";
      =     "HYDRAULIC_FUNCTIONS_DB".PUMP_1_2_SS_LCS;
      A     L 0.0;
      A     "PUMP_1_STA_PB_LCS";
      =     "HYDRAULIC_FUNCTIONS_DB".PUMP_1_STA_PB_LCS;
      A     L 0.0;
      A     "PUMP_1_STP_PB_LCS";
      =     "HYDRAULIC_FUNCTIONS_DB".PUMP_1_STP_PB_LCS;
      A     L 0.0;
      A     "PUMP_2_STA_PB_LCS";
      =     "HYDRAULIC_FUNCTIONS_DB".PUMP_2_STA_PB_LCS;
      A     L 0.0;
      A     "PUMP_2_STP_PB_LCS";
      =     "HYDRAULIC_FUNCTIONS_DB".PUMP_2_STP_PB_LCS;
      A     L 0.0;
      A     "CIR_PUMP_STA_PB_LCS";
      =     "HYDRAULIC_FUNCTIONS_DB".CIR_PUMP_STA_PB_LCS;
      A     L 0.0;
      A     "CIR_PUMP_STP_PB_LCS";
      =     "HYDRAULIC_FUNCTIONS_DB".CIR_PUMP_STP_PB_LCS;
      A     L 0.0;
      A     "COLR_FAN_STA_PB_LCS";
      =     "HYDRAULIC_FUNCTIONS_DB".COLR_FAN_STA_PB_LCS;
      A     L 0.0;
      A     "COLR_FAN_STP_PB_LCS";
      =     "HYDRAULIC_FUNCTIONS_DB".COLR_FAN_STP_PB_LCS;
      A     L 0.0;
      A     "LAMP_TEST_PB_LCS_41";
      =     "HYDRAULIC_FUNCTIONS_DB".LAMP_TEST_PB_LCS_41;
      A     L 0.0;
      A     "SHT_OF_VLV_LIN_1_FUL_OPN";
      =     "HYDRAULIC_FUNCTIONS_DB".SHT_OF_VLV_LIN_1_FUL_OPN;
      A     L 0.0;
      A     "SHT_OF_VLV_LIN_2_FUL_OPN";
      =     "HYDRAULIC_FUNCTIONS_DB".SHT_OF_VLV_LIN_2_FUL_OPN;
      A     L 0.0;
      A     "LOW_OIL_TEMP";
      =     "HYDRAULIC_FUNCTIONS_DB".LOW_OIL_TEMP;
      A     L 0.0;
      A     "HIGH_OIL_TEMP";
      =     "HYDRAULIC_FUNCTIONS_DB".HIGH_OIL_TEMP;
      A     L 0.0;
      A     "MAX_OIL_TEMP";
      =     "HYDRAULIC_FUNCTIONS_DB".MAX_OIL_TEMP;
      A     L 0.0;
      A     "LOW_OIL_LEVEL";
      =     "HYDRAULIC_FUNCTIONS_DB".LOW_OIL_LEVEL;
      A     L 0.0;
      A     "MIN_OIL_LEVEL";
      =     "HYDRAULIC_FUNCTIONS_DB".MIN_OIL_LEVEL;
      A     L 0.0;
      A     "RET_LIN_FLTR_CKD";
      =     "HYDRAULIC_FUNCTIONS_DB".RET_LIN_FLTR_CKD;
      A     L 0.0;
      A     "LOW_OIL_PRESS";
      =     "HYDRAULIC_FUNCTIONS_DB".LOW_OIL_PRESS;
      A     L 0.0;
      A     "HIGH_OIL_PRESS";
      =     "HYDRAULIC_FUNCTIONS_DB".HIGH_OIL_PRESS;
      A     L 0.0;
      A     "EMG_ACCM_STA_PB_LCS";
      =     "HYDRAULIC_FUNCTIONS_DB".EMG_ACCM_STA_PB_LCS;
      A     L 0.0;
      A     "EMG_ACCM_STP_PB_LCS";
      =     "HYDRAULIC_FUNCTIONS_DB".EMG_ACCM_STP_PB_LCS;
      A     L 0.0;
      A     "HTR_STA_PB_LCS";
      =     "HYDRAULIC_FUNCTIONS_DB".HTR_STA_PB_LCS;
      A     L 0.0;
      A     "HTR_STP_PB_LCS";
      =     "HYDRAULIC_FUNCTIONS_DB".HTR_STP_PB_LCS;
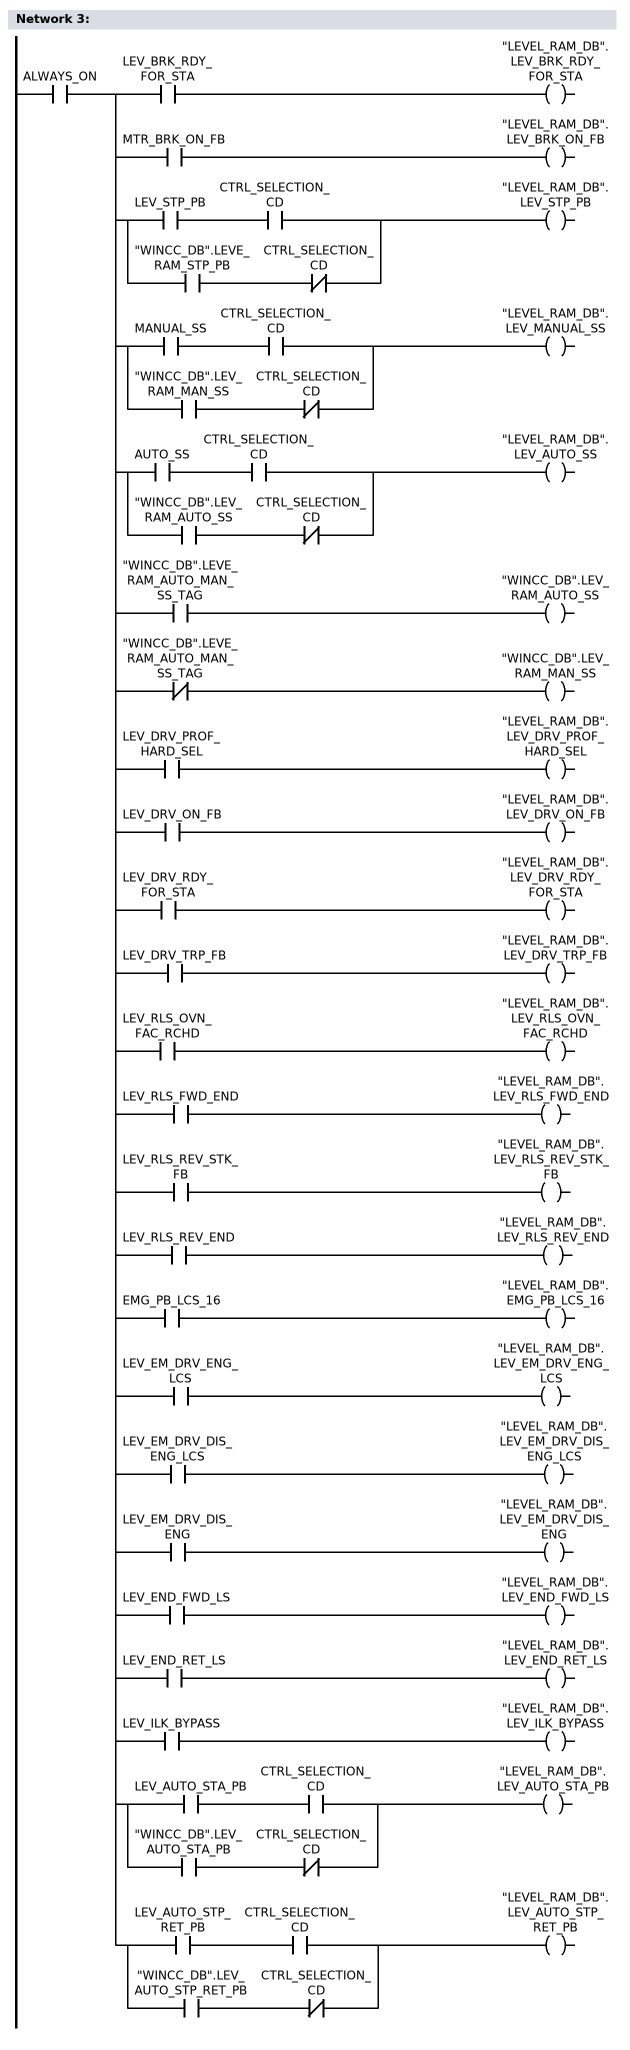
NETWORK
TITLE =
      A     "ALWAYS_ON";
      =     L 0.0;
      A     L 0.0;
      A     "LEV_BRK_RDY_FOR_STA";
      =     "LEVEL_RAM_DB".LEV_BRK_RDY_FOR_STA;
      A     L 0.0;
      A     "MTR_BRK_ON_FB";
      =     "LEVEL_RAM_DB".LEV_BRK_ON_FB;
      A     L 0.0;
      A(;
      A     "LEV_STP_PB";
      A     "CTRL_SELECTION_CD";
      O;
      A     "WINCC_DB".LEVE_RAM_STP_PB;
      AN    "CTRL_SELECTION_CD";
      );
      =     "LEVEL_RAM_DB".LEV_STP_PB;
      A     L 0.0;
      A(;
      A     "MANUAL_SS";
      A     "CTRL_SELECTION_CD";
      O;
      A     "WINCC_DB".LEV_RAM_MAN_SS;
      AN    "CTRL_SELECTION_CD";
      );
      =     "LEVEL_RAM_DB".LEV_MANUAL_SS;
      A     L 0.0;
      A(;
      A     "AUTO_SS";
      A     "CTRL_SELECTION_CD";
      O;
      A     "WINCC_DB".LEV_RAM_AUTO_SS;
      AN    "CTRL_SELECTION_CD";
      );
      =     "LEVEL_RAM_DB".LEV_AUTO_SS;
      A     L 0.0;
      A     "WINCC_DB".LEVE_RAM_AUTO_MAN_SS_TAG;
      =     "WINCC_DB".LEV_RAM_AUTO_SS;
      A     L 0.0;
      AN    "WINCC_DB".LEVE_RAM_AUTO_MAN_SS_TAG;
      =     "WINCC_DB".LEV_RAM_MAN_SS;
      A     L 0.0;
      A     "LEV_DRV_PROF_HARD_SEL";
      =     "LEVEL_RAM_DB".LEV_DRV_PROF_HARD_SEL;
      A     L 0.0;
      A     "LEV_DRV_ON_FB";
      =     "LEVEL_RAM_DB".LEV_DRV_ON_FB;
      A     L 0.0;
      A     "LEV_DRV_RDY_FOR_STA";
      =     "LEVEL_RAM_DB".LEV_DRV_RDY_FOR_STA;
      A     L 0.0;
      A     "LEV_DRV_TRP_FB";
      =     "LEVEL_RAM_DB".LEV_DRV_TRP_FB;
      A     L 0.0;
      A     "LEV_RLS_OVN_FAC_RCHD";
      =     "LEVEL_RAM_DB".LEV_RLS_OVN_FAC_RCHD;
      A     L 0.0;
      A     "LEV_RLS_FWD_END";
      =     "LEVEL_RAM_DB".LEV_RLS_FWD_END;
      A     L 0.0;
      A     "LEV_RLS_REV_STK_FB";
      =     "LEVEL_RAM_DB".LEV_RLS_REV_STK_FB;
      A     L 0.0;
      A     "LEV_RLS_REV_END";
      =     "LEVEL_RAM_DB".LEV_RLS_REV_END;
      A     L 0.0;
      A     "EMG_PB_LCS_16";
      =     "LEVEL_RAM_DB".EMG_PB_LCS_16;
      A     L 0.0;
      A     "LEV_EM_DRV_ENG_LCS";
      =     "LEVEL_RAM_DB".LEV_EM_DRV_ENG_LCS;
      A     L 0.0;
      A     "LEV_EM_DRV_DIS_ENG_LCS";
      =     "LEVEL_RAM_DB".LEV_EM_DRV_DIS_ENG_LCS;
      A     L 0.0;
      A     "LEV_EM_DRV_DIS_ENG";
      =     "LEVEL_RAM_DB".LEV_EM_DRV_DIS_ENG;
      A     L 0.0;
      A     "LEV_END_FWD_LS";
      =     "LEVEL_RAM_DB".LEV_END_FWD_LS;
      A     L 0.0;
      A     "LEV_END_RET_LS";
      =     "LEVEL_RAM_DB".LEV_END_RET_LS;
      A     L 0.0;
      A     "LEV_ILK_BYPASS";
      =     "LEVEL_RAM_DB".LEV_ILK_BYPASS;
      A     L 0.0;
      A(;
      A     "LEV_AUTO_STA_PB";
      A     "CTRL_SELECTION_CD";
      O;
      A     "WINCC_DB".LEV_AUTO_STA_PB;
      AN    "CTRL_SELECTION_CD";
      );
      =     "LEVEL_RAM_DB".LEV_AUTO_STA_PB;
      A     L 0.0;
      A(;
      A     "LEV_AUTO_STP_RET_PB";
      A     "CTRL_SELECTION_CD";
      O;
      A     "WINCC_DB".LEV_AUTO_STP_RET_PB;
      AN    "CTRL_SELECTION_CD";
      );
      =     "LEVEL_RAM_DB".LEV_AUTO_STP_RET_PB;
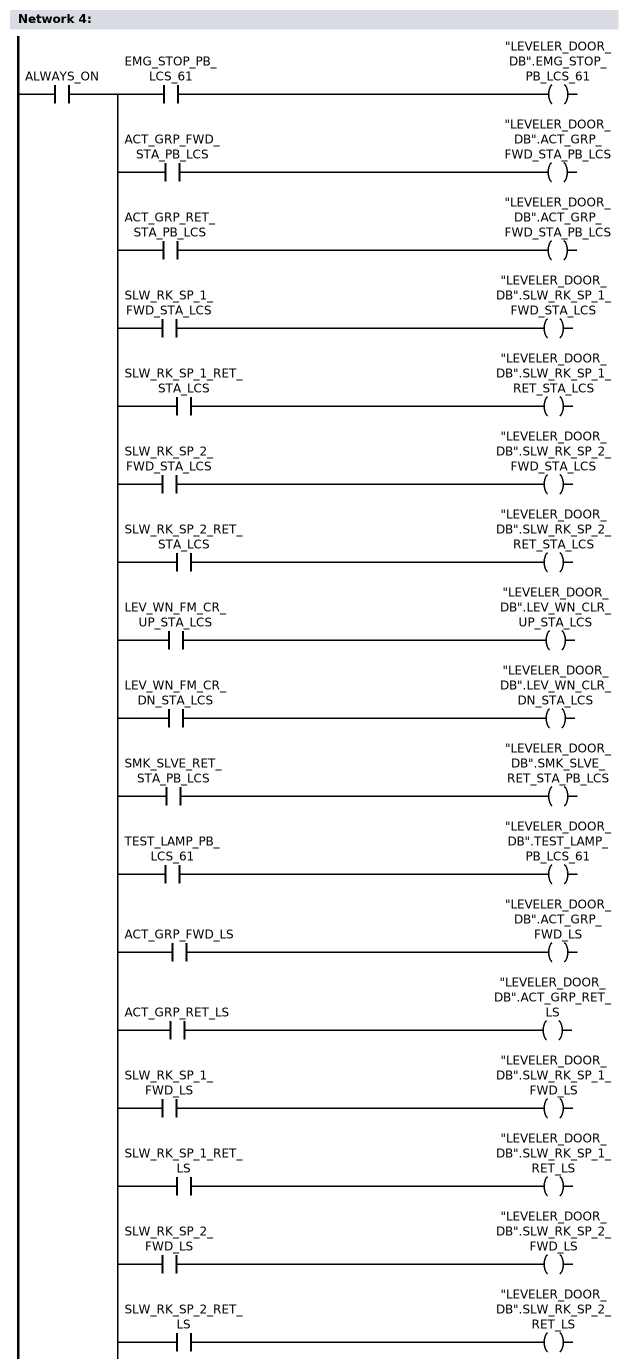
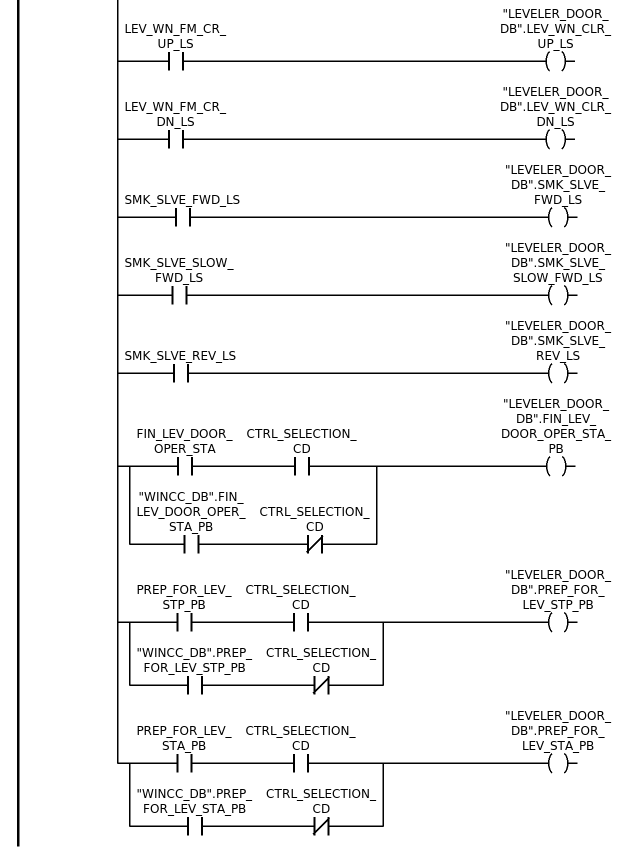
NETWORK
TITLE =
      A     "ALWAYS_ON";
      =     L 0.0;
      A     L 0.0;
      A     "EMG_STOP_PB_LCS_61";
      =     "LEVELER_DOOR_DB".EMG_STOP_PB_LCS_61;
      A     L 0.0;
      A     "ACT_GRP_FWD_STA_PB_LCS";
      =     "LEVELER_DOOR_DB".ACT_GRP_FWD_STA_PB_LCS;
      A     L 0.0;
      A     "ACT_GRP_RET_STA_PB_LCS";
      =     "LEVELER_DOOR_DB".ACT_GRP_FWD_STA_PB_LCS;
      A     L 0.0;
      A     "SLW_RK_SP_1_FWD_STA_LCS";
      =     "LEVELER_DOOR_DB".SLW_RK_SP_1_FWD_STA_LCS;
      A     L 0.0;
      A     "SLW_RK_SP_1_RET_STA_LCS";
      =     "LEVELER_DOOR_DB".SLW_RK_SP_1_RET_STA_LCS;
      A     L 0.0;
      A     "SLW_RK_SP_2_FWD_STA_LCS";
      =     "LEVELER_DOOR_DB".SLW_RK_SP_2_FWD_STA_LCS;
      A     L 0.0;
      A     "SLW_RK_SP_2_RET_STA_LCS";
      =     "LEVELER_DOOR_DB".SLW_RK_SP_2_RET_STA_LCS;
      A     L 0.0;
      A     "LEV_WN_FM_CR_UP_STA_LCS";
      =     "LEVELER_DOOR_DB".LEV_WN_CLR_UP_STA_LCS;
      A     L 0.0;
      A     "LEV_WN_FM_CR_DN_STA_LCS";
      =     "LEVELER_DOOR_DB".LEV_WN_CLR_DN_STA_LCS;
      A     L 0.0;
      A     "SMK_SLVE_RET_STA_PB_LCS";
      =     "LEVELER_DOOR_DB".SMK_SLVE_RET_STA_PB_LCS;
      A     L 0.0;
      A     "TEST_LAMP_PB_LCS_61";
      =     "LEVELER_DOOR_DB".TEST_LAMP_PB_LCS_61;
      A     L 0.0;
      A     "ACT_GRP_FWD_LS";
      =     "LEVELER_DOOR_DB".ACT_GRP_FWD_LS;
      A     L 0.0;
      A     "ACT_GRP_RET_LS";
      =     "LEVELER_DOOR_DB".ACT_GRP_RET_LS;
      A     L 0.0;
      A     "SLW_RK_SP_1_FWD_LS";
      =     "LEVELER_DOOR_DB".SLW_RK_SP_1_FWD_LS;
      A     L 0.0;
      A     "SLW_RK_SP_1_RET_LS";
      =     "LEVELER_DOOR_DB".SLW_RK_SP_1_RET_LS;
      A     L 0.0;
      A     "SLW_RK_SP_2_FWD_LS";
      =     "LEVELER_DOOR_DB".SLW_RK_SP_2_FWD_LS;
      A     L 0.0;
      A     "SLW_RK_SP_2_RET_LS";
      =     "LEVELER_DOOR_DB".SLW_RK_SP_2_RET_LS;
      A     L 0.0;
      A     "LEV_WN_FM_CR_UP_LS";
      =     "LEVELER_DOOR_DB".LEV_WN_CLR_UP_LS;
      A     L 0.0;
      A     "LEV_WN_FM_CR_DN_LS";
      =     "LEVELER_DOOR_DB".LEV_WN_CLR_DN_LS;
      A     L 0.0;
      A     "SMK_SLVE_FWD_LS";
      =     "LEVELER_DOOR_DB".SMK_SLVE_FWD_LS;
      A     L 0.0;
      A     "SMK_SLVE_SLOW_FWD_LS";
      =     "LEVELER_DOOR_DB".SMK_SLVE_SLOW_FWD_LS;
      A     L 0.0;
      A     "SMK_SLVE_REV_LS";
      =     "LEVELER_DOOR_DB".SMK_SLVE_REV_LS;
      A     L 0.0;
      A(;
      A     "FIN_LEV_DOOR_OPER_STA";
      A     "CTRL_SELECTION_CD";
      O;
      A     "WINCC_DB".FIN_LEV_DOOR_OPER_STA_PB;
      AN    "CTRL_SELECTION_CD";
      );
      =     "LEVELER_DOOR_DB".FIN_LEV_DOOR_OPER_STA_PB;
      A     L 0.0;
      A(;
      A     "PREP_FOR_LEV_STP_PB";
      A     "CTRL_SELECTION_CD";
      O;
      A     "WINCC_DB".PREP_FOR_LEV_STP_PB;
      AN    "CTRL_SELECTION_CD";
      );
      =     "LEVELER_DOOR_DB".PREP_FOR_LEV_STP_PB;
      A     L 0.0;
      A(;
      A     "PREP_FOR_LEV_STA_PB";
      A     "CTRL_SELECTION_CD";
      O;
      A     "WINCC_DB".PREP_FOR_LEV_STA_PB;
      AN    "CTRL_SELECTION_CD";
      );
      =     "LEVELER_DOOR_DB".PREP_FOR_LEV_STA_PB;
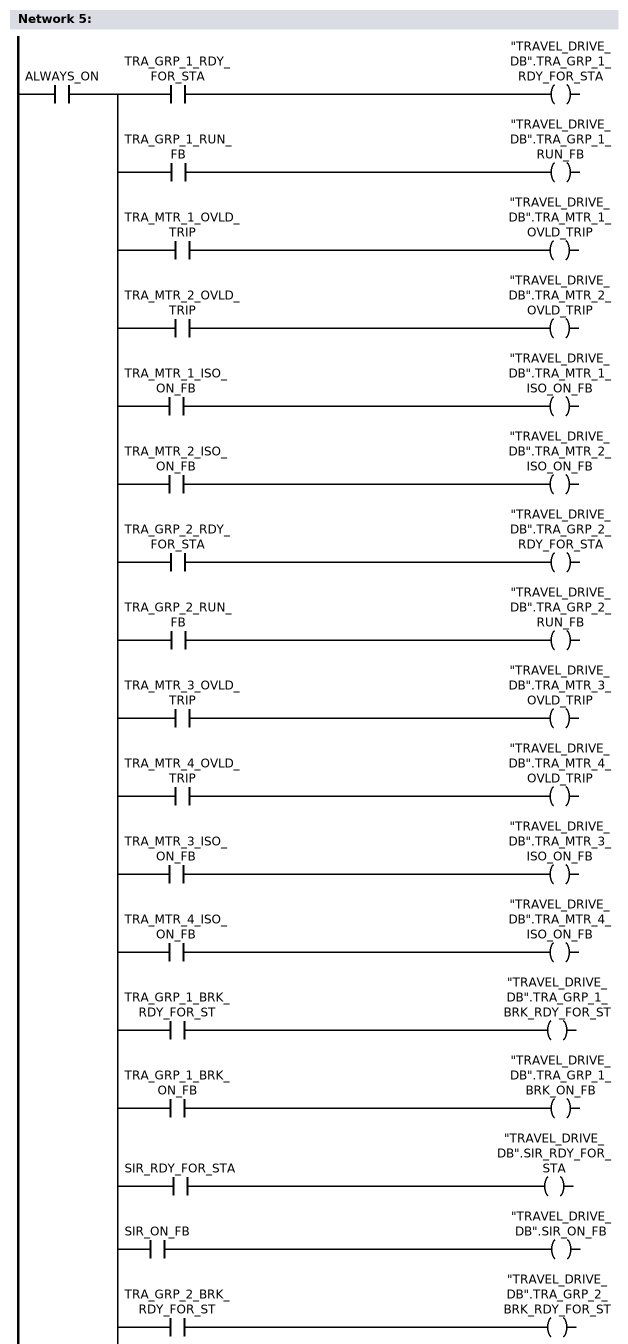
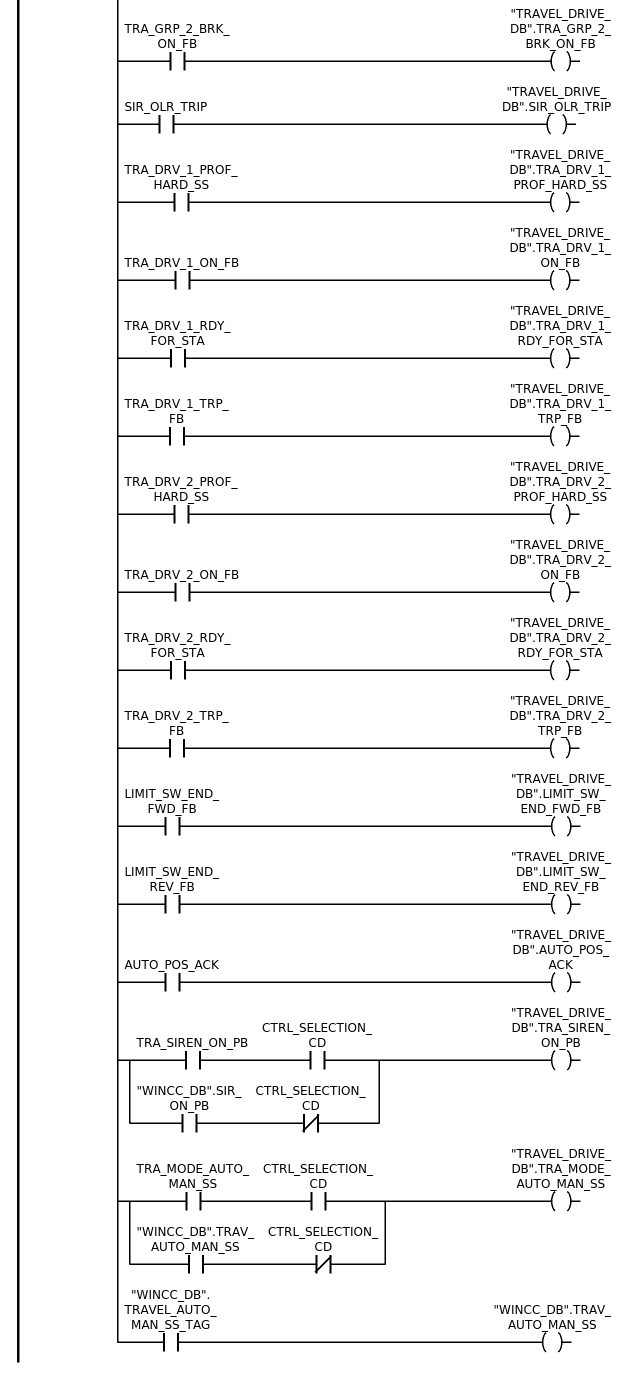
NETWORK
TITLE =
      A     "ALWAYS_ON";
      =     L 0.0;
      A     L 0.0;
      A     "TRA_GRP_1_RDY_FOR_STA";
      =     "TRAVEL_DRIVE_DB".TRA_GRP_1_RDY_FOR_STA;
      A     L 0.0;
      A     "TRA_GRP_1_RUN_FB";
      =     "TRAVEL_DRIVE_DB".TRA_GRP_1_RUN_FB;
      A     L 0.0;
      A     "TRA_MTR_1_OVLD_TRIP";
      =     "TRAVEL_DRIVE_DB".TRA_MTR_1_OVLD_TRIP;
      A     L 0.0;
      A     "TRA_MTR_2_OVLD_TRIP";
      =     "TRAVEL_DRIVE_DB".TRA_MTR_2_OVLD_TRIP;
      A     L 0.0;
      A     "TRA_MTR_1_ISO_ON_FB";
      =     "TRAVEL_DRIVE_DB".TRA_MTR_1_ISO_ON_FB;
      A     L 0.0;
      A     "TRA_MTR_2_ISO_ON_FB";
      =     "TRAVEL_DRIVE_DB".TRA_MTR_2_ISO_ON_FB;
      A     L 0.0;
      A     "TRA_GRP_2_RDY_FOR_STA";
      =     "TRAVEL_DRIVE_DB".TRA_GRP_2_RDY_FOR_STA;
      A     L 0.0;
      A     "TRA_GRP_2_RUN_FB";
      =     "TRAVEL_DRIVE_DB".TRA_GRP_2_RUN_FB;
      A     L 0.0;
      A     "TRA_MTR_3_OVLD_TRIP";
      =     "TRAVEL_DRIVE_DB".TRA_MTR_3_OVLD_TRIP;
      A     L 0.0;
      A     "TRA_MTR_4_OVLD_TRIP";
      =     "TRAVEL_DRIVE_DB".TRA_MTR_4_OVLD_TRIP;
      A     L 0.0;
      A     "TRA_MTR_3_ISO_ON_FB";
      =     "TRAVEL_DRIVE_DB".TRA_MTR_3_ISO_ON_FB;
      A     L 0.0;
      A     "TRA_MTR_4_ISO_ON_FB";
      =     "TRAVEL_DRIVE_DB".TRA_MTR_4_ISO_ON_FB;
      A     L 0.0;
      A     "TRA_GRP_1_BRK_RDY_FOR_ST";
      =     "TRAVEL_DRIVE_DB".TRA_GRP_1_BRK_RDY_FOR_ST;
      A     L 0.0;
      A     "TRA_GRP_1_BRK_ON_FB";
      =     "TRAVEL_DRIVE_DB".TRA_GRP_1_BRK_ON_FB;
      A     L 0.0;
      A     "SIR_RDY_FOR_STA";
      =     "TRAVEL_DRIVE_DB".SIR_RDY_FOR_STA;
      A     L 0.0;
      A     "SIR_ON_FB";
      =     "TRAVEL_DRIVE_DB".SIR_ON_FB;
      A     L 0.0;
      A     "TRA_GRP_2_BRK_RDY_FOR_ST";
      =     "TRAVEL_DRIVE_DB".TRA_GRP_2_BRK_RDY_FOR_ST;
      A     L 0.0;
      A     "TRA_GRP_2_BRK_ON_FB";
      =     "TRAVEL_DRIVE_DB".TRA_GRP_2_BRK_ON_FB;
      A     L 0.0;
      A     "SIR_OLR_TRIP";
      =     "TRAVEL_DRIVE_DB".SIR_OLR_TRIP;
      A     L 0.0;
      A     "TRA_DRV_1_PROF_HARD_SS";
      =     "TRAVEL_DRIVE_DB".TRA_DRV_1_PROF_HARD_SS;
      A     L 0.0;
      A     "TRA_DRV_1_ON_FB";
      =     "TRAVEL_DRIVE_DB".TRA_DRV_1_ON_FB;
      A     L 0.0;
      A     "TRA_DRV_1_RDY_FOR_STA";
      =     "TRAVEL_DRIVE_DB".TRA_DRV_1_RDY_FOR_STA;
      A     L 0.0;
      A     "TRA_DRV_1_TRP_FB";
      =     "TRAVEL_DRIVE_DB".TRA_DRV_1_TRP_FB;
      A     L 0.0;
      A     "TRA_DRV_2_PROF_HARD_SS";
      =     "TRAVEL_DRIVE_DB".TRA_DRV_2_PROF_HARD_SS;
      A     L 0.0;
      A     "TRA_DRV_2_ON_FB";
      =     "TRAVEL_DRIVE_DB".TRA_DRV_2_ON_FB;
      A     L 0.0;
      A     "TRA_DRV_2_RDY_FOR_STA";
      =     "TRAVEL_DRIVE_DB".TRA_DRV_2_RDY_FOR_STA;
      A     L 0.0;
      A     "TRA_DRV_2_TRP_FB";
      =     "TRAVEL_DRIVE_DB".TRA_DRV_2_TRP_FB;
      A     L 0.0;
      A     "LIMIT_SW_END_FWD_FB";
      =     "TRAVEL_DRIVE_DB".LIMIT_SW_END_FWD_FB;
      A     L 0.0;
      A     "LIMIT_SW_END_REV_FB";
      =     "TRAVEL_DRIVE_DB".LIMIT_SW_END_REV_FB;
      A     L 0.0;
      A     "AUTO_POS_ACK";
      =     "TRAVEL_DRIVE_DB".AUTO_POS_ACK;
      A     L 0.0;
      A(;
      A     "TRA_SIREN_ON_PB";
      A     "CTRL_SELECTION_CD";
      O;
      A     "WINCC_DB".SIR_ON_PB;
      AN    "CTRL_SELECTION_CD";
      );
      =     "TRAVEL_DRIVE_DB".TRA_SIREN_ON_PB;
      A     L 0.0;
      A(;
      A     "TRA_MODE_AUTO_MAN_SS";
      A     "CTRL_SELECTION_CD";
      O;
      A     "WINCC_DB".TRAV_AUTO_MAN_SS;
      AN    "CTRL_SELECTION_CD";
      );
      =     "TRAVEL_DRIVE_DB".TRA_MODE_AUTO_MAN_SS;
      A     L 0.0;
      A     "WINCC_DB".TRAVEL_AUTO_MAN_SS_TAG;
      =     "WINCC_DB".TRAV_AUTO_MAN_SS;
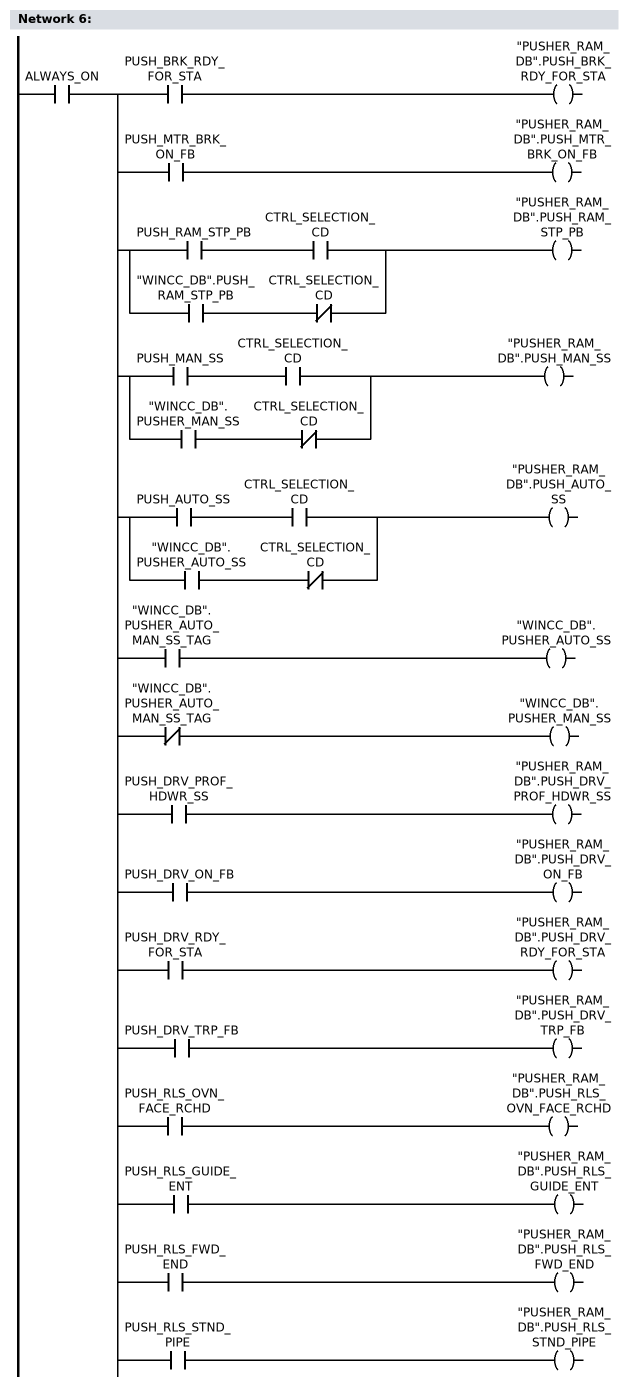
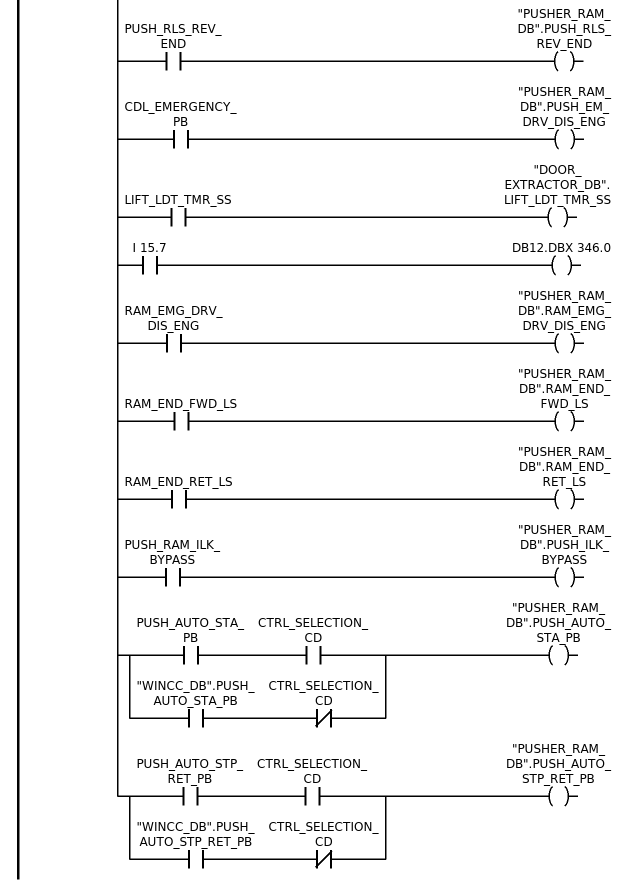
NETWORK
TITLE =
      A     "ALWAYS_ON";
      =     L 0.0;
      A     L 0.0;
      A     "PUSH_BRK_RDY_FOR_STA";
      =     "PUSHER_RAM_DB".PUSH_BRK_RDY_FOR_STA;
      A     L 0.0;
      A     "PUSH_MTR_BRK_ON_FB";
      =     "PUSHER_RAM_DB".PUSH_MTR_BRK_ON_FB;
      A     L 0.0;
      A(;
      A     "PUSH_RAM_STP_PB";
      A     "CTRL_SELECTION_CD";
      O;
      A     "WINCC_DB".PUSH_RAM_STP_PB;
      AN    "CTRL_SELECTION_CD";
      );
      =     "PUSHER_RAM_DB".PUSH_RAM_STP_PB;
      A     L 0.0;
      A(;
      A     "PUSH_MAN_SS";
      A     "CTRL_SELECTION_CD";
      O;
      A     "WINCC_DB".PUSHER_MAN_SS;
      AN    "CTRL_SELECTION_CD";
      );
      =     "PUSHER_RAM_DB".PUSH_MAN_SS;
      A     L 0.0;
      A(;
      A     "PUSH_AUTO_SS";
      A     "CTRL_SELECTION_CD";
      O;
      A     "WINCC_DB".PUSHER_AUTO_SS;
      AN    "CTRL_SELECTION_CD";
      );
      =     "PUSHER_RAM_DB".PUSH_AUTO_SS;
      A     L 0.0;
      A     "WINCC_DB".PUSHER_AUTO_MAN_SS_TAG;
      =     "WINCC_DB".PUSHER_AUTO_SS;
      A     L 0.0;
      AN    "WINCC_DB".PUSHER_AUTO_MAN_SS_TAG;
      =     "WINCC_DB".PUSHER_MAN_SS;
      A     L 0.0;
      A     "PUSH_DRV_PROF_HDWR_SS";
      =     "PUSHER_RAM_DB".PUSH_DRV_PROF_HDWR_SS;
      A     L 0.0;
      A     "PUSH_DRV_ON_FB";
      =     "PUSHER_RAM_DB".PUSH_DRV_ON_FB;
      A     L 0.0;
      A     "PUSH_DRV_RDY_FOR_STA";
      =     "PUSHER_RAM_DB".PUSH_DRV_RDY_FOR_STA;
      A     L 0.0;
      A     "PUSH_DRV_TRP_FB";
      =     "PUSHER_RAM_DB".PUSH_DRV_TRP_FB;
      A     L 0.0;
      A     "PUSH_RLS_OVN_FACE_RCHD";
      =     "PUSHER_RAM_DB".PUSH_RLS_OVN_FACE_RCHD;
      A     L 0.0;
      A     "PUSH_RLS_GUIDE_ENT";
      =     "PUSHER_RAM_DB".PUSH_RLS_GUIDE_ENT;
      A     L 0.0;
      A     "PUSH_RLS_FWD_END";
      =     "PUSHER_RAM_DB".PUSH_RLS_FWD_END;
      A     L 0.0;
      A     "PUSH_RLS_STND_PIPE";
      =     "PUSHER_RAM_DB".PUSH_RLS_STND_PIPE;
      A     L 0.0;
      A     "PUSH_RLS_REV_END";
      =     "PUSHER_RAM_DB".PUSH_RLS_REV_END;
      A     L 0.0;
      A     "CDL_EMERGENCY_PB";
      =     "PUSHER_RAM_DB".PUSH_EM_DRV_DIS_ENG;
      A     L 0.0;
      A     "LIFT_LDT_TMR_SS";
      =     "DOOR_EXTRACTOR_DB".LIFT_LDT_TMR_SS;
      A     L 0.0;
      A     I 15.7;
      =     DB12.DBX 346.0;
      A     L 0.0;
      A     "RAM_EMG_DRV_DIS_ENG";
      =     "PUSHER_RAM_DB".RAM_EMG_DRV_DIS_ENG;
      A     L 0.0;
      A     "RAM_END_FWD_LS";
      =     "PUSHER_RAM_DB".RAM_END_FWD_LS;
      A     L 0.0;
      A     "RAM_END_RET_LS";
      =     "PUSHER_RAM_DB".RAM_END_RET_LS;
      A     L 0.0;
      A     "PUSH_RAM_ILK_BYPASS";
      =     "PUSHER_RAM_DB".PUSH_ILK_BYPASS;
      A     L 0.0;
      A(;
      A     "PUSH_AUTO_STA_PB";
      A     "CTRL_SELECTION_CD";
      O;
      A     "WINCC_DB".PUSH_AUTO_STA_PB;
      AN    "CTRL_SELECTION_CD";
      );
      =     "PUSHER_RAM_DB".PUSH_AUTO_STA_PB;
      A     L 0.0;
      A(;
      A     "PUSH_AUTO_STP_RET_PB";
      A     "CTRL_SELECTION_CD";
      O;
      A     "WINCC_DB".PUSH_AUTO_STP_RET_PB;
      AN    "CTRL_SELECTION_CD";
      );
      =     "PUSHER_RAM_DB".PUSH_AUTO_STP_RET_PB;
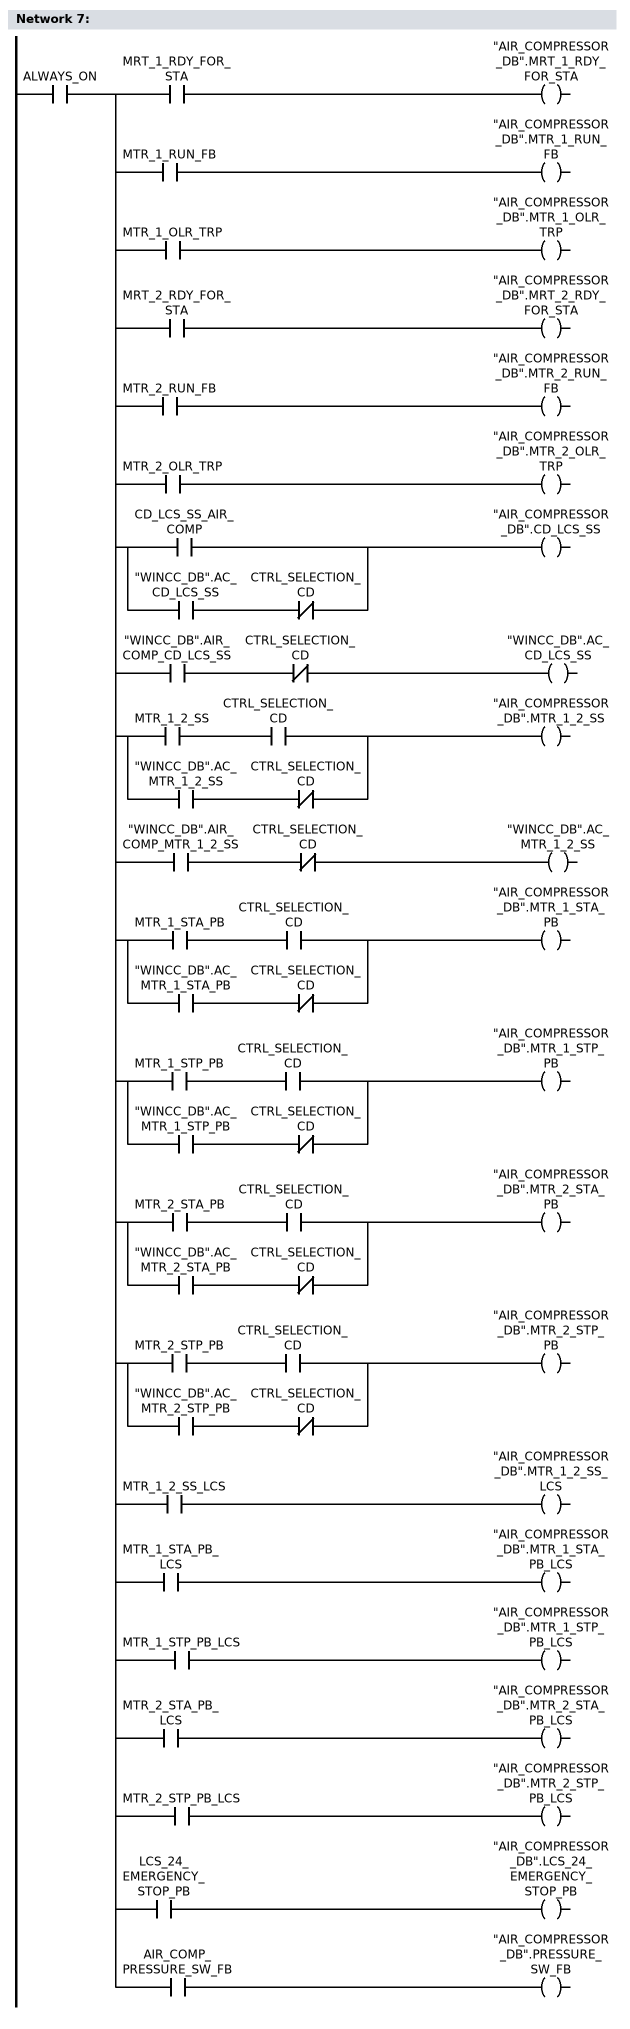
NETWORK
TITLE =
      A     "ALWAYS_ON";
      =     L 0.0;
      A     L 0.0;
      A     "MRT_1_RDY_FOR_STA";
      =     "AIR_COMPRESSOR_DB".MRT_1_RDY_FOR_STA;
      A     L 0.0;
      A     "MTR_1_RUN_FB";
      =     "AIR_COMPRESSOR_DB".MTR_1_RUN_FB;
      A     L 0.0;
      A     "MTR_1_OLR_TRP";
      =     "AIR_COMPRESSOR_DB".MTR_1_OLR_TRP;
      A     L 0.0;
      A     "MRT_2_RDY_FOR_STA";
      =     "AIR_COMPRESSOR_DB".MRT_2_RDY_FOR_STA;
      A     L 0.0;
      A     "MTR_2_RUN_FB";
      =     "AIR_COMPRESSOR_DB".MTR_2_RUN_FB;
      A     L 0.0;
      A     "MTR_2_OLR_TRP";
      =     "AIR_COMPRESSOR_DB".MTR_2_OLR_TRP;
      A     L 0.0;
      A(;
      O     "CD_LCS_SS_AIR_COMP";
      O;
      A     "WINCC_DB".AC_CD_LCS_SS;
      AN    "CTRL_SELECTION_CD";
      );
      =     "AIR_COMPRESSOR_DB".CD_LCS_SS;
      A     L 0.0;
      A     "WINCC_DB".AIR_COMP_CD_LCS_SS;
      AN    "CTRL_SELECTION_CD";
      =     "WINCC_DB".AC_CD_LCS_SS;
      A     L 0.0;
      A(;
      A     "MTR_1_2_SS";
      A     "CTRL_SELECTION_CD";
      O;
      A     "WINCC_DB".AC_MTR_1_2_SS;
      AN    "CTRL_SELECTION_CD";
      );
      =     "AIR_COMPRESSOR_DB".MTR_1_2_SS;
      A     L 0.0;
      A     "WINCC_DB".AIR_COMP_MTR_1_2_SS;
      AN    "CTRL_SELECTION_CD";
      =     "WINCC_DB".AC_MTR_1_2_SS;
      A     L 0.0;
      A(;
      A     "MTR_1_STA_PB";
      A     "CTRL_SELECTION_CD";
      O;
      A     "WINCC_DB".AC_MTR_1_STA_PB;
      AN    "CTRL_SELECTION_CD";
      );
      =     "AIR_COMPRESSOR_DB".MTR_1_STA_PB;
      A     L 0.0;
      A(;
      A     "MTR_1_STP_PB";
      A     "CTRL_SELECTION_CD";
      O;
      A     "WINCC_DB".AC_MTR_1_STP_PB;
      AN    "CTRL_SELECTION_CD";
      );
      =     "AIR_COMPRESSOR_DB".MTR_1_STP_PB;
      A     L 0.0;
      A(;
      A     "MTR_2_STA_PB";
      A     "CTRL_SELECTION_CD";
      O;
      A     "WINCC_DB".AC_MTR_2_STA_PB;
      AN    "CTRL_SELECTION_CD";
      );
      =     "AIR_COMPRESSOR_DB".MTR_2_STA_PB;
      A     L 0.0;
      A(;
      A     "MTR_2_STP_PB";
      A     "CTRL_SELECTION_CD";
      O;
      A     "WINCC_DB".AC_MTR_2_STP_PB;
      AN    "CTRL_SELECTION_CD";
      );
      =     "AIR_COMPRESSOR_DB".MTR_2_STP_PB;
      A     L 0.0;
      A     "MTR_1_2_SS_LCS";
      =     "AIR_COMPRESSOR_DB".MTR_1_2_SS_LCS;
      A     L 0.0;
      A     "MTR_1_STA_PB_LCS";
      =     "AIR_COMPRESSOR_DB".MTR_1_STA_PB_LCS;
      A     L 0.0;
      A     "MTR_1_STP_PB_LCS";
      =     "AIR_COMPRESSOR_DB".MTR_1_STP_PB_LCS;
      A     L 0.0;
      A     "MTR_2_STA_PB_LCS";
      =     "AIR_COMPRESSOR_DB".MTR_2_STA_PB_LCS;
      A     L 0.0;
      A     "MTR_2_STP_PB_LCS";
      =     "AIR_COMPRESSOR_DB".MTR_2_STP_PB_LCS;
      A     L 0.0;
      A     "LCS_24_EMERGENCY_STOP_PB";
      =     "AIR_COMPRESSOR_DB".LCS_24_EMERGENCY_STOP_PB;
      A     L 0.0;
      A     "AIR_COMP_PRESSURE_SW_FB";
      =     "AIR_COMPRESSOR_DB".PRESSURE_SW_FB;
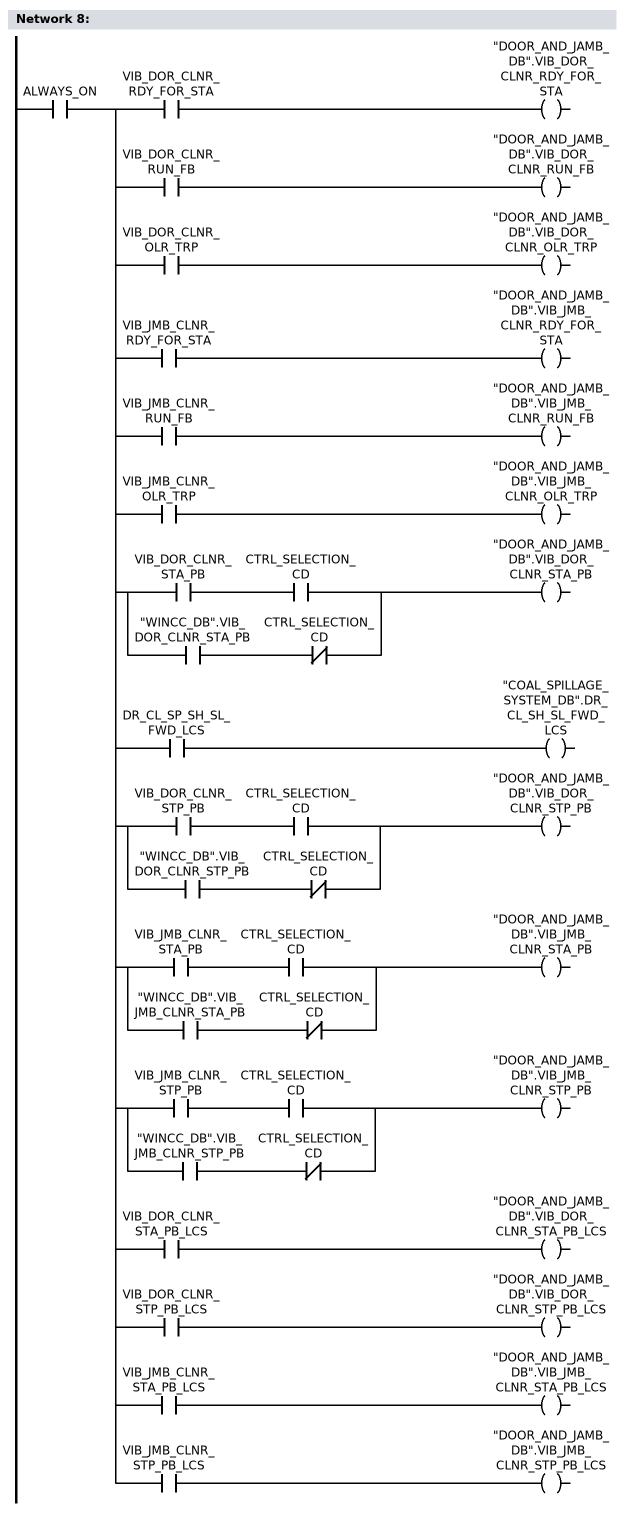
NETWORK
TITLE =
      A     "ALWAYS_ON";
      =     L 0.0;
      A     L 0.0;
      A     "VIB_DOR_CLNR_RDY_FOR_STA";
      =     "DOOR_AND_JAMB_DB".VIB_DOR_CLNR_RDY_FOR_STA;
      A     L 0.0;
      A     "VIB_DOR_CLNR_RUN_FB";
      =     "DOOR_AND_JAMB_DB".VIB_DOR_CLNR_RUN_FB;
      A     L 0.0;
      A     "VIB_DOR_CLNR_OLR_TRP";
      =     "DOOR_AND_JAMB_DB".VIB_DOR_CLNR_OLR_TRP;
      A     L 0.0;
      A     "VIB_JMB_CLNR_RDY_FOR_STA";
      =     "DOOR_AND_JAMB_DB".VIB_JMB_CLNR_RDY_FOR_STA;
      A     L 0.0;
      A     "VIB_JMB_CLNR_RUN_FB";
      =     "DOOR_AND_JAMB_DB".VIB_JMB_CLNR_RUN_FB;
      A     L 0.0;
      A     "VIB_JMB_CLNR_OLR_TRP";
      =     "DOOR_AND_JAMB_DB".VIB_JMB_CLNR_OLR_TRP;
      A     L 0.0;
      A(;
      A     "VIB_DOR_CLNR_STA_PB";
      A     "CTRL_SELECTION_CD";
      O;
      A     "WINCC_DB".VIB_DOR_CLNR_STA_PB;
      AN    "CTRL_SELECTION_CD";
      );
      =     "DOOR_AND_JAMB_DB".VIB_DOR_CLNR_STA_PB;
      A     L 0.0;
      A     "DR_CL_SP_SH_SL_FWD_LCS";
      =     "COAL_SPILLAGE_SYSTEM_DB".DR_CL_SH_SL_FWD_LCS;
      A     L 0.0;
      A(;
      A     "VIB_DOR_CLNR_STP_PB";
      A     "CTRL_SELECTION_CD";
      O;
      A     "WINCC_DB".VIB_DOR_CLNR_STP_PB;
      AN    "CTRL_SELECTION_CD";
      );
      =     "DOOR_AND_JAMB_DB".VIB_DOR_CLNR_STP_PB;
      A     L 0.0;
      A(;
      A     "VIB_JMB_CLNR_STA_PB";
      A     "CTRL_SELECTION_CD";
      O;
      A     "WINCC_DB".VIB_JMB_CLNR_STA_PB;
      AN    "CTRL_SELECTION_CD";
      );
      =     "DOOR_AND_JAMB_DB".VIB_JMB_CLNR_STA_PB;
      A     L 0.0;
      A(;
      A     "VIB_JMB_CLNR_STP_PB";
      A     "CTRL_SELECTION_CD";
      O;
      A     "WINCC_DB".VIB_JMB_CLNR_STP_PB;
      AN    "CTRL_SELECTION_CD";
      );
      =     "DOOR_AND_JAMB_DB".VIB_JMB_CLNR_STP_PB;
      A     L 0.0;
      A     "VIB_DOR_CLNR_STA_PB_LCS";
      =     "DOOR_AND_JAMB_DB".VIB_DOR_CLNR_STA_PB_LCS;
      A     L 0.0;
      A     "VIB_DOR_CLNR_STP_PB_LCS";
      =     "DOOR_AND_JAMB_DB".VIB_DOR_CLNR_STP_PB_LCS;
      A     L 0.0;
      A     "VIB_JMB_CLNR_STA_PB_LCS";
      =     "DOOR_AND_JAMB_DB".VIB_JMB_CLNR_STA_PB_LCS;
      A     L 0.0;
      A     "VIB_JMB_CLNR_STP_PB_LCS";
      =     "DOOR_AND_JAMB_DB".VIB_JMB_CLNR_STP_PB_LCS;
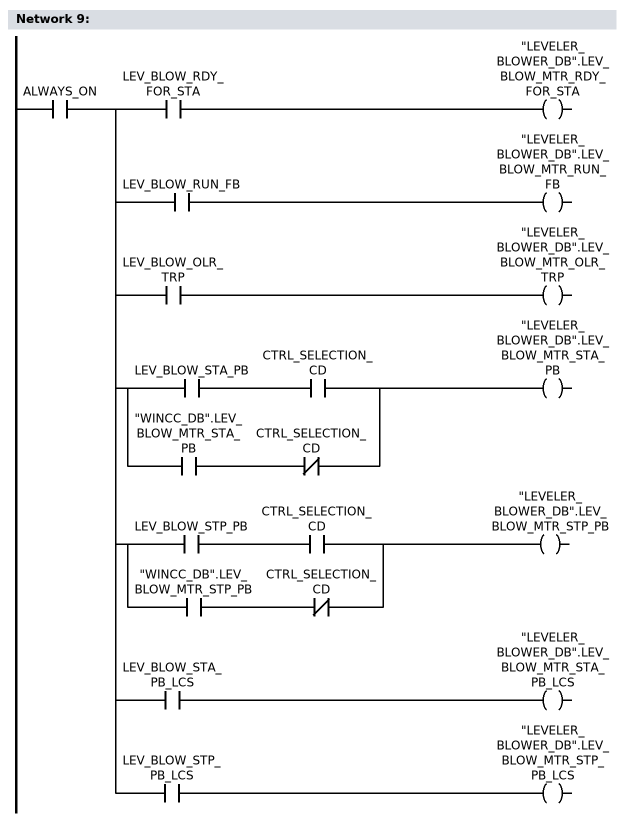
NETWORK
TITLE =
      A     "ALWAYS_ON";
      =     L 0.0;
      A     L 0.0;
      A     "LEV_BLOW_RDY_FOR_STA";
      =     "LEVELER_BLOWER_DB".LEV_BLOW_MTR_RDY_FOR_STA;
      A     L 0.0;
      A     "LEV_BLOW_RUN_FB";
      =     "LEVELER_BLOWER_DB".LEV_BLOW_MTR_RUN_FB;
      A     L 0.0;
      A     "LEV_BLOW_OLR_TRP";
      =     "LEVELER_BLOWER_DB".LEV_BLOW_MTR_OLR_TRP;
      A     L 0.0;
      A(;
      A     "LEV_BLOW_STA_PB";
      A     "CTRL_SELECTION_CD";
      O;
      A     "WINCC_DB".LEV_BLOW_MTR_STA_PB;
      AN    "CTRL_SELECTION_CD";
      );
      =     "LEVELER_BLOWER_DB".LEV_BLOW_MTR_STA_PB;
      A     L 0.0;
      A(;
      A     "LEV_BLOW_STP_PB";
      A     "CTRL_SELECTION_CD";
      O;
      A     "WINCC_DB".LEV_BLOW_MTR_STP_PB;
      AN    "CTRL_SELECTION_CD";
      );
      =     "LEVELER_BLOWER_DB".LEV_BLOW_MTR_STP_PB;
      A     L 0.0;
      A     "LEV_BLOW_STA_PB_LCS";
      =     "LEVELER_BLOWER_DB".LEV_BLOW_MTR_STA_PB_LCS;
      A     L 0.0;
      A     "LEV_BLOW_STP_PB_LCS";
      =     "LEVELER_BLOWER_DB".LEV_BLOW_MTR_STP_PB_LCS;
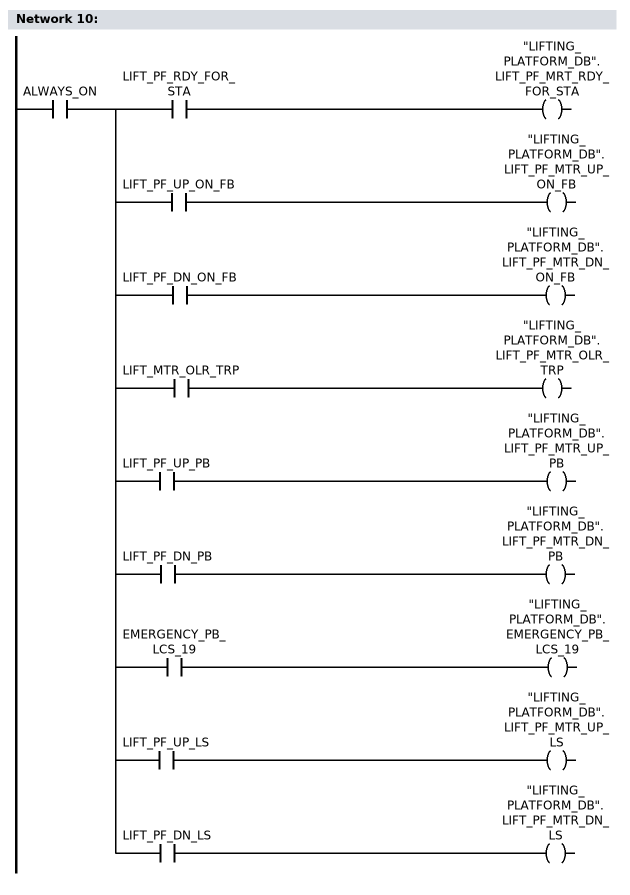
NETWORK
TITLE =
      A     "ALWAYS_ON";
      =     L 0.0;
      A     L 0.0;
      A     "LIFT_PF_RDY_FOR_STA";
      =     "LIFTING_PLATFORM_DB".LIFT_PF_MRT_RDY_FOR_STA;
      A     L 0.0;
      A     "LIFT_PF_UP_ON_FB";
      =     "LIFTING_PLATFORM_DB".LIFT_PF_MTR_UP_ON_FB;
      A     L 0.0;
      A     "LIFT_PF_DN_ON_FB";
      =     "LIFTING_PLATFORM_DB".LIFT_PF_MTR_DN_ON_FB;
      A     L 0.0;
      A     "LIFT_MTR_OLR_TRP";
      =     "LIFTING_PLATFORM_DB".LIFT_PF_MTR_OLR_TRP;
      A     L 0.0;
      A     "LIFT_PF_UP_PB";
      =     "LIFTING_PLATFORM_DB".LIFT_PF_MTR_UP_PB;
      A     L 0.0;
      A     "LIFT_PF_DN_PB";
      =     "LIFTING_PLATFORM_DB".LIFT_PF_MTR_DN_PB;
      A     L 0.0;
      A     "EMERGENCY_PB_LCS_19";
      =     "LIFTING_PLATFORM_DB".EMERGENCY_PB_LCS_19;
      A     L 0.0;
      A     "LIFT_PF_UP_LS";
      =     "LIFTING_PLATFORM_DB".LIFT_PF_MTR_UP_LS;
      A     L 0.0;
      A     "LIFT_PF_DN_LS";
      =     "LIFTING_PLATFORM_DB".LIFT_PF_MTR_DN_LS;
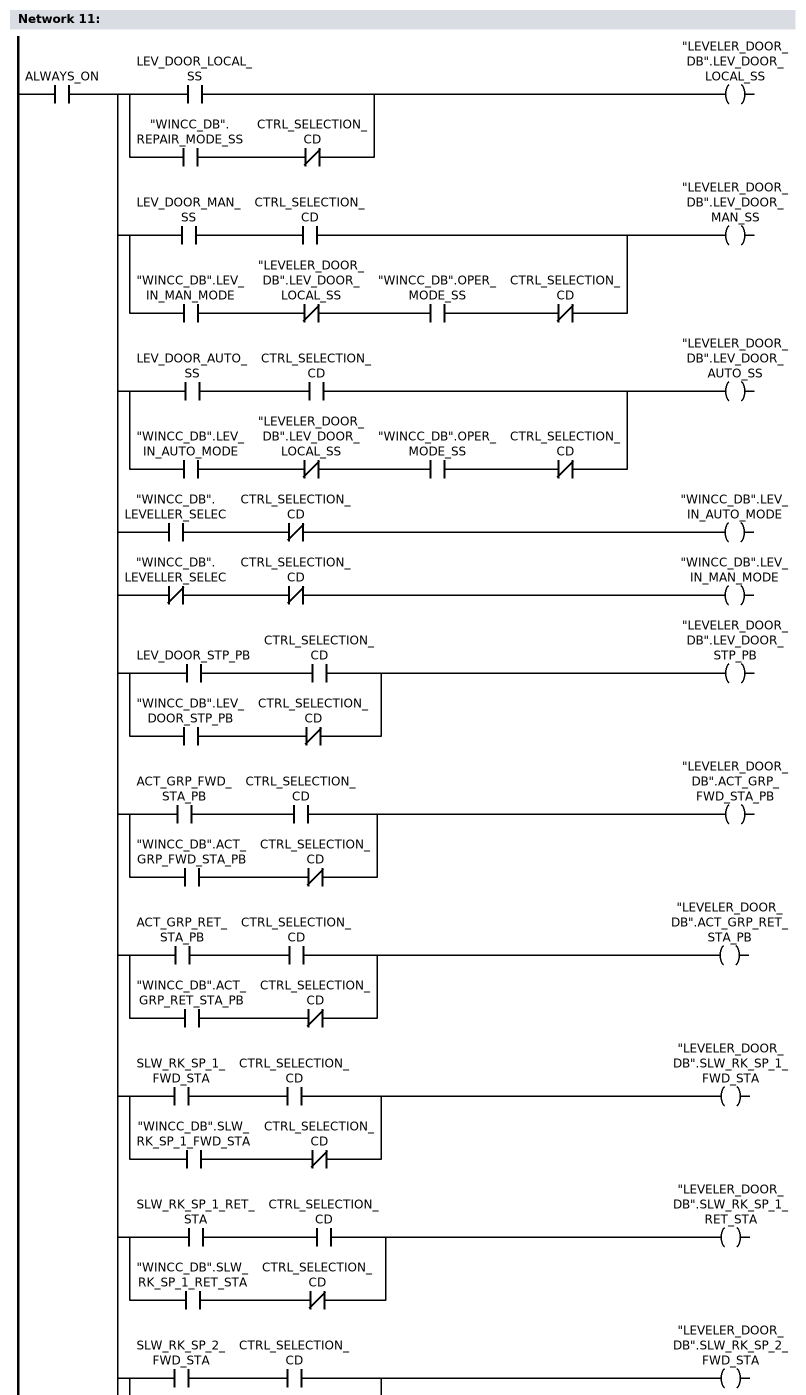
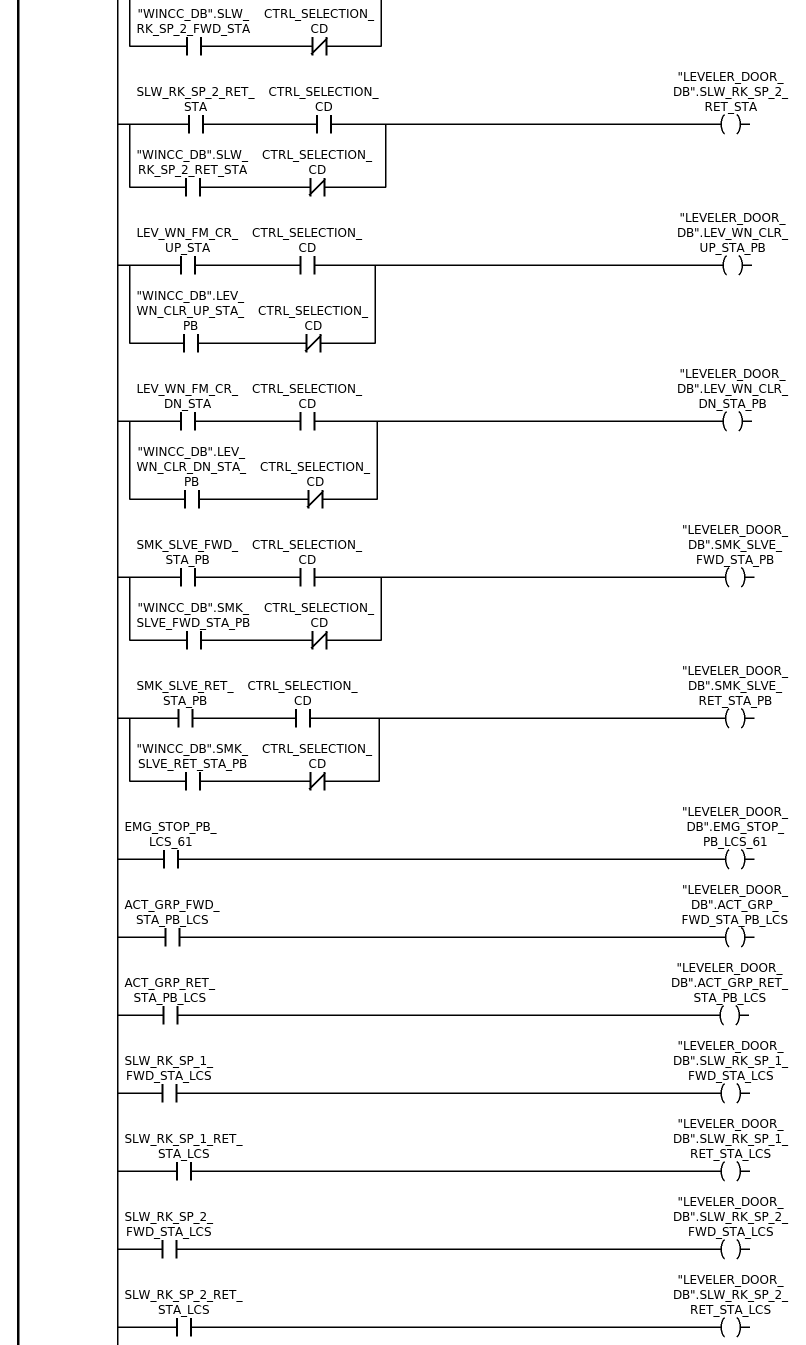
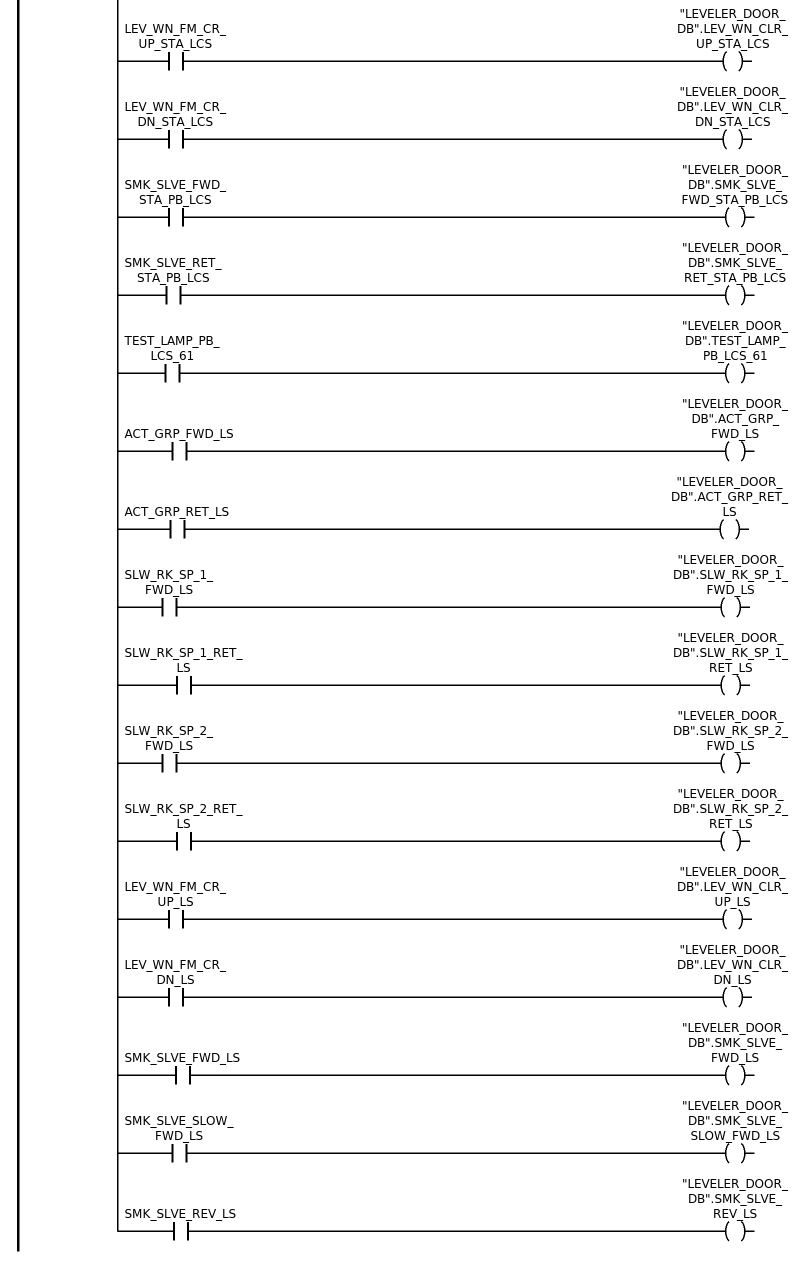
NETWORK
TITLE =
      A     "ALWAYS_ON";
      =     L 0.0;
      A     L 0.0;
      A(;
      O     "LEV_DOOR_LOCAL_SS";
      O;
      A     "WINCC_DB".REPAIR_MODE_SS;
      AN    "CTRL_SELECTION_CD";
      );
      =     "LEVELER_DOOR_DB".LEV_DOOR_LOCAL_SS;
      A     L 0.0;
      A(;
      A     "LEV_DOOR_MAN_SS";
      A     "CTRL_SELECTION_CD";
      O;
      A     "WINCC_DB".LEV_IN_MAN_MODE;
      AN    "LEVELER_DOOR_DB".LEV_DOOR_LOCAL_SS;
      A     "WINCC_DB".OPER_MODE_SS;
      AN    "CTRL_SELECTION_CD";
      );
      =     "LEVELER_DOOR_DB".LEV_DOOR_MAN_SS;
      A     L 0.0;
      A(;
      A     "LEV_DOOR_AUTO_SS";
      A     "CTRL_SELECTION_CD";
      O;
      A     "WINCC_DB".LEV_IN_AUTO_MODE;
      AN    "LEVELER_DOOR_DB".LEV_DOOR_LOCAL_SS;
      A     "WINCC_DB".OPER_MODE_SS;
      AN    "CTRL_SELECTION_CD";
      );
      =     "LEVELER_DOOR_DB".LEV_DOOR_AUTO_SS;
      A     L 0.0;
      A     "WINCC_DB".LEVELLER_SELEC;
      AN    "CTRL_SELECTION_CD";
      =     "WINCC_DB".LEV_IN_AUTO_MODE;
      A     L 0.0;
      AN    "WINCC_DB".LEVELLER_SELEC;
      AN    "CTRL_SELECTION_CD";
      =     "WINCC_DB".LEV_IN_MAN_MODE;
      A     L 0.0;
      A(;
      A     "LEV_DOOR_STP_PB";
      A     "CTRL_SELECTION_CD";
      O;
      A     "WINCC_DB".LEV_DOOR_STP_PB;
      AN    "CTRL_SELECTION_CD";
      );
      =     "LEVELER_DOOR_DB".LEV_DOOR_STP_PB;
      A     L 0.0;
      A(;
      A     "ACT_GRP_FWD_STA_PB";
      A     "CTRL_SELECTION_CD";
      O;
      A     "WINCC_DB".ACT_GRP_FWD_STA_PB;
      AN    "CTRL_SELECTION_CD";
      );
      =     "LEVELER_DOOR_DB".ACT_GRP_FWD_STA_PB;
      A     L 0.0;
      A(;
      A     "ACT_GRP_RET_STA_PB";
      A     "CTRL_SELECTION_CD";
      O;
      A     "WINCC_DB".ACT_GRP_RET_STA_PB;
      AN    "CTRL_SELECTION_CD";
      );
      =     "LEVELER_DOOR_DB".ACT_GRP_RET_STA_PB;
      A     L 0.0;
      A(;
      A     "SLW_RK_SP_1_FWD_STA";
      A     "CTRL_SELECTION_CD";
      O;
      A     "WINCC_DB".SLW_RK_SP_1_FWD_STA;
      AN    "CTRL_SELECTION_CD";
      );
      =     "LEVELER_DOOR_DB".SLW_RK_SP_1_FWD_STA;
      A     L 0.0;
      A(;
      A     "SLW_RK_SP_1_RET_STA";
      A     "CTRL_SELECTION_CD";
      O;
      A     "WINCC_DB".SLW_RK_SP_1_RET_STA;
      AN    "CTRL_SELECTION_CD";
      );
      =     "LEVELER_DOOR_DB".SLW_RK_SP_1_RET_STA;
      A     L 0.0;
      A(;
      A     "SLW_RK_SP_2_FWD_STA";
      A     "CTRL_SELECTION_CD";
      O;
      A     "WINCC_DB".SLW_RK_SP_2_FWD_STA;
      AN    "CTRL_SELECTION_CD";
      );
      =     "LEVELER_DOOR_DB".SLW_RK_SP_2_FWD_STA;
      A     L 0.0;
      A(;
      A     "SLW_RK_SP_2_RET_STA";
      A     "CTRL_SELECTION_CD";
      O;
      A     "WINCC_DB".SLW_RK_SP_2_RET_STA;
      AN    "CTRL_SELECTION_CD";
      );
      =     "LEVELER_DOOR_DB".SLW_RK_SP_2_RET_STA;
      A     L 0.0;
      A(;
      A     "LEV_WN_FM_CR_UP_STA";
      A     "CTRL_SELECTION_CD";
      O;
      A     "WINCC_DB".LEV_WN_CLR_UP_STA_PB;
      AN    "CTRL_SELECTION_CD";
      );
      =     "LEVELER_DOOR_DB".LEV_WN_CLR_UP_STA_PB;
      A     L 0.0;
      A(;
      A     "LEV_WN_FM_CR_DN_STA";
      A     "CTRL_SELECTION_CD";
      O;
      A     "WINCC_DB".LEV_WN_CLR_DN_STA_PB;
      AN    "CTRL_SELECTION_CD";
      );
      =     "LEVELER_DOOR_DB".LEV_WN_CLR_DN_STA_PB;
      A     L 0.0;
      A(;
      A     "SMK_SLVE_FWD_STA_PB";
      A     "CTRL_SELECTION_CD";
      O;
      A     "WINCC_DB".SMK_SLVE_FWD_STA_PB;
      AN    "CTRL_SELECTION_CD";
      );
      =     "LEVELER_DOOR_DB".SMK_SLVE_FWD_STA_PB;
      A     L 0.0;
      A(;
      A     "SMK_SLVE_RET_STA_PB";
      A     "CTRL_SELECTION_CD";
      O;
      A     "WINCC_DB".SMK_SLVE_RET_STA_PB;
      AN    "CTRL_SELECTION_CD";
      );
      =     "LEVELER_DOOR_DB".SMK_SLVE_RET_STA_PB;
      A     L 0.0;
      A     "EMG_STOP_PB_LCS_61";
      =     "LEVELER_DOOR_DB".EMG_STOP_PB_LCS_61;
      A     L 0.0;
      A     "ACT_GRP_FWD_STA_PB_LCS";
      =     "LEVELER_DOOR_DB".ACT_GRP_FWD_STA_PB_LCS;
      A     L 0.0;
      A     "ACT_GRP_RET_STA_PB_LCS";
      =     "LEVELER_DOOR_DB".ACT_GRP_RET_STA_PB_LCS;
      A     L 0.0;
      A     "SLW_RK_SP_1_FWD_STA_LCS";
      =     "LEVELER_DOOR_DB".SLW_RK_SP_1_FWD_STA_LCS;
      A     L 0.0;
      A     "SLW_RK_SP_1_RET_STA_LCS";
      =     "LEVELER_DOOR_DB".SLW_RK_SP_1_RET_STA_LCS;
      A     L 0.0;
      A     "SLW_RK_SP_2_FWD_STA_LCS";
      =     "LEVELER_DOOR_DB".SLW_RK_SP_2_FWD_STA_LCS;
      A     L 0.0;
      A     "SLW_RK_SP_2_RET_STA_LCS";
      =     "LEVELER_DOOR_DB".SLW_RK_SP_2_RET_STA_LCS;
      A     L 0.0;
      A     "LEV_WN_FM_CR_UP_STA_LCS";
      =     "LEVELER_DOOR_DB".LEV_WN_CLR_UP_STA_LCS;
      A     L 0.0;
      A     "LEV_WN_FM_CR_DN_STA_LCS";
      =     "LEVELER_DOOR_DB".LEV_WN_CLR_DN_STA_LCS;
      A     L 0.0;
      A     "SMK_SLVE_FWD_STA_PB_LCS";
      =     "LEVELER_DOOR_DB".SMK_SLVE_FWD_STA_PB_LCS;
      A     L 0.0;
      A     "SMK_SLVE_RET_STA_PB_LCS";
      =     "LEVELER_DOOR_DB".SMK_SLVE_RET_STA_PB_LCS;
      A     L 0.0;
      A     "TEST_LAMP_PB_LCS_61";
      =     "LEVELER_DOOR_DB".TEST_LAMP_PB_LCS_61;
      A     L 0.0;
      A     "ACT_GRP_FWD_LS";
      =     "LEVELER_DOOR_DB".ACT_GRP_FWD_LS;
      A     L 0.0;
      A     "ACT_GRP_RET_LS";
      =     "LEVELER_DOOR_DB".ACT_GRP_RET_LS;
      A     L 0.0;
      A     "SLW_RK_SP_1_FWD_LS";
      =     "LEVELER_DOOR_DB".SLW_RK_SP_1_FWD_LS;
      A     L 0.0;
      A     "SLW_RK_SP_1_RET_LS";
      =     "LEVELER_DOOR_DB".SLW_RK_SP_1_RET_LS;
      A     L 0.0;
      A     "SLW_RK_SP_2_FWD_LS";
      =     "LEVELER_DOOR_DB".SLW_RK_SP_2_FWD_LS;
      A     L 0.0;
      A     "SLW_RK_SP_2_RET_LS";
      =     "LEVELER_DOOR_DB".SLW_RK_SP_2_RET_LS;
      A     L 0.0;
      A     "LEV_WN_FM_CR_UP_LS";
      =     "LEVELER_DOOR_DB".LEV_WN_CLR_UP_LS;
      A     L 0.0;
      A     "LEV_WN_FM_CR_DN_LS";
      =     "LEVELER_DOOR_DB".LEV_WN_CLR_DN_LS;
      A     L 0.0;
      A     "SMK_SLVE_FWD_LS";
      =     "LEVELER_DOOR_DB".SMK_SLVE_FWD_LS;
      A     L 0.0;
      A     "SMK_SLVE_SLOW_FWD_LS";
      =     "LEVELER_DOOR_DB".SMK_SLVE_SLOW_FWD_LS;
      A     L 0.0;
      A     "SMK_SLVE_REV_LS";
      =     "LEVELER_DOOR_DB".SMK_SLVE_REV_LS;
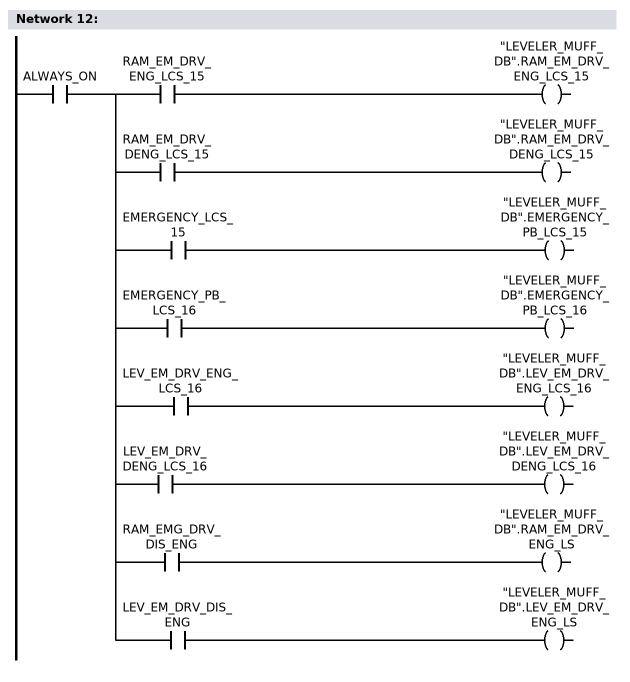
NETWORK
TITLE =
      A     "ALWAYS_ON";
      =     L 0.0;
      A     L 0.0;
      A     "RAM_EM_DRV_ENG_LCS_15";
      =     "LEVELER_MUFF_DB".RAM_EM_DRV_ENG_LCS_15;
      A     L 0.0;
      A     "RAM_EM_DRV_DENG_LCS_15";
      =     "LEVELER_MUFF_DB".RAM_EM_DRV_DENG_LCS_15;
      A     L 0.0;
      A     "EMERGENCY_LCS_15";
      =     "LEVELER_MUFF_DB".EMERGENCY_PB_LCS_15;
      A     L 0.0;
      A     "EMERGENCY_PB_LCS_16";
      =     "LEVELER_MUFF_DB".EMERGENCY_PB_LCS_16;
      A     L 0.0;
      A     "LEV_EM_DRV_ENG_LCS_16";
      =     "LEVELER_MUFF_DB".LEV_EM_DRV_ENG_LCS_16;
      A     L 0.0;
      A     "LEV_EM_DRV_DENG_LCS_16";
      =     "LEVELER_MUFF_DB".LEV_EM_DRV_DENG_LCS_16;
      A     L 0.0;
      A     "RAM_EMG_DRV_DIS_ENG";
      =     "LEVELER_MUFF_DB".RAM_EM_DRV_ENG_LS;
      A     L 0.0;
      A     "LEV_EM_DRV_DIS_ENG";
      =     "LEVELER_MUFF_DB".LEV_EM_DRV_ENG_LS;
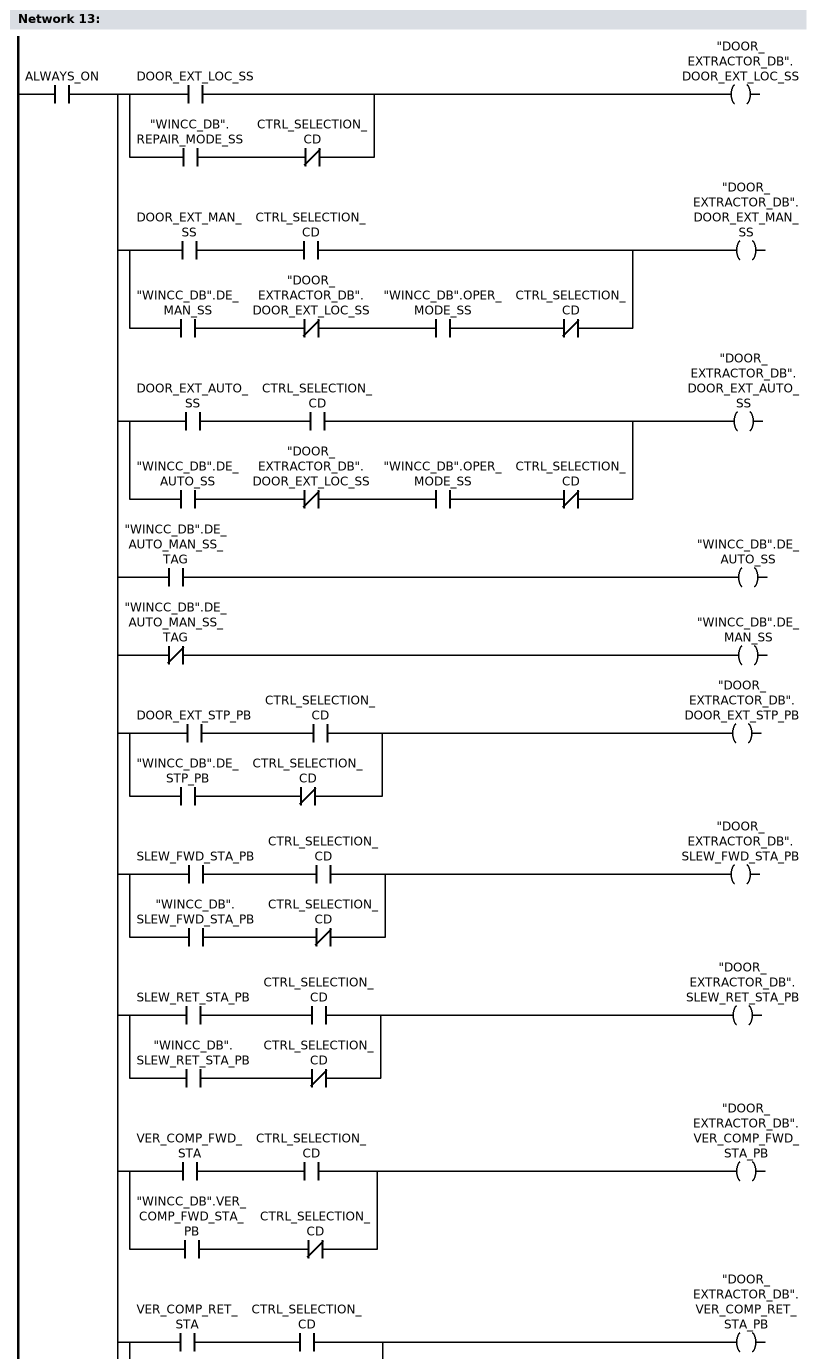
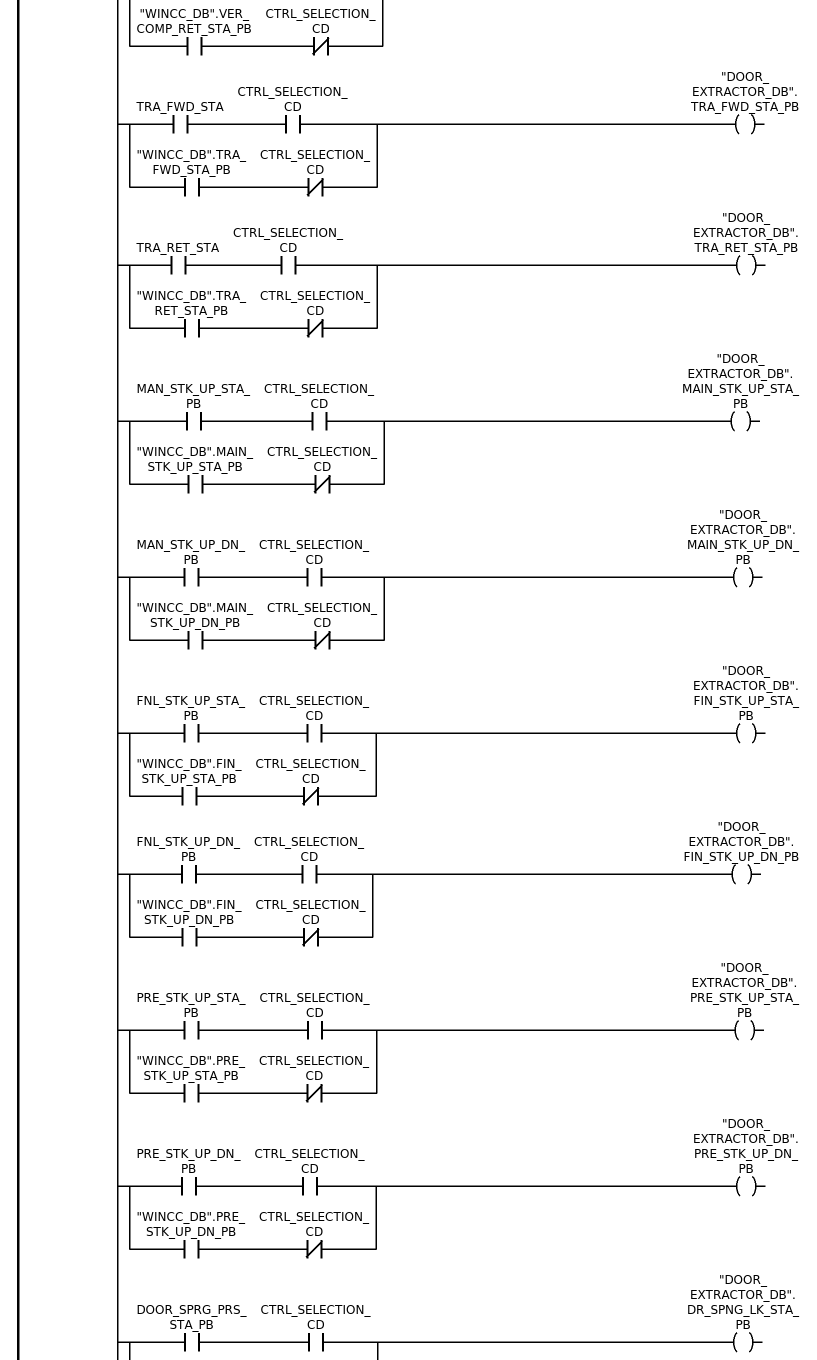
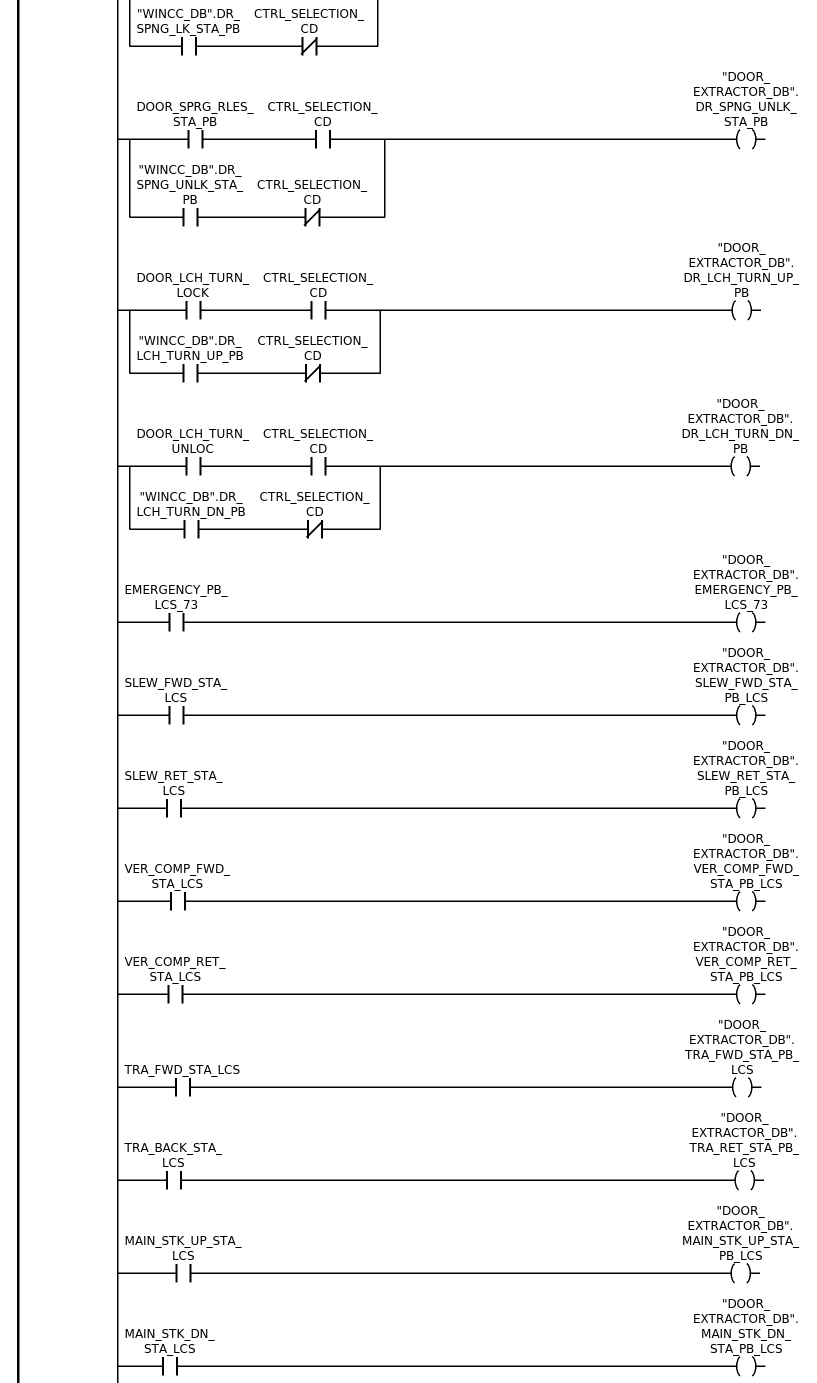
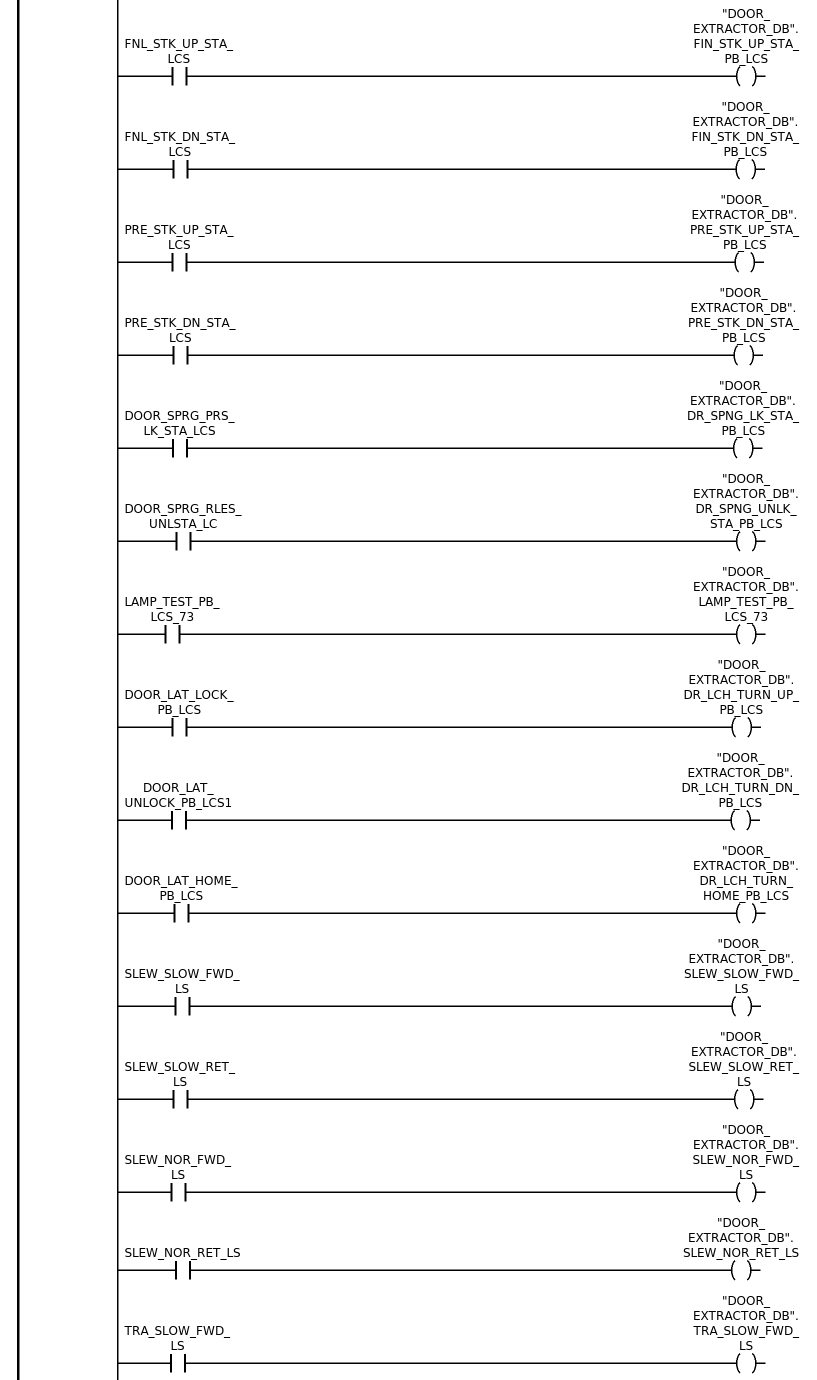
